Omron CX-Programmer project 新規ﾌﾟﾛｼﾞｪｸﾄ (CX-Programmer 9.20)

# PLC CP_14_0212: CJ2M CPU13
I/O table (CPU CJ2M-CPU13): rack 0 slot 0 CJ1W-ID262; rack 0 slot 1 CJ1W-OD263; rack 0 slot 2 CJ1W-ID262; rack 0 slot 3 CJ1W-OD211; rack 0 slot 4 CJ1W-ID211; rack 0 slot 5 CJ1W-OD211; rack 0 slot 6 CJ1W-CLK23

## Global symbols (name address type ; comment)
0.00 BOOL  ; SE:到着1_確認
0.01 BOOL  ; SE:到着2_確認
0.02 BOOL  ; SE:溜り_確認
0.03 BOOL  ; SE:ﾒｶｴｱｰ圧力
0.04 BOOL  ; SE:切出_引端
0.05 BOOL  ; SE:切出_出端
0.06 BOOL  ; SE:押え_動点
0.07 BOOL  ; SE:供給RBO_過負荷
0.08 BOOL  ; SE:ｽﾄｯﾊﾟｰ3_引端
0.09 BOOL  ; SE:ｽﾄｯﾊﾟｰ3_出端
0.10 BOOL  ; SE:ｽﾄｯﾊﾟｰ2_引端
0.11 BOOL  ; SE:ｽﾄｯﾊﾟｰ2_出端
0.12 BOOL  ; SE:ｽﾄｯﾊﾟｰ1_引端
0.13 BOOL  ; SE:ｽﾄｯﾊﾟｰ1_出端
0.14 BOOL  ; SE:ﾌﾟｯｼｬｰ3_引端
0.15 BOOL  ; SE:ﾌﾟｯｼｬｰ3_出端
1001 CHANNEL  ; 1CH_L_OV_SFT
1001.00 BOOL  ; 1CH_L_OV_SFT
1001.04 BOOL  ; 1CH_L_OV_SFT
1002 CHANNEL  ; 1CH_L_RV_SFT
1002.00 BOOL  ; 1CH_L_RV_SFT
1002.04 BOOL  ; 1CH_L_RV_SFT
1003 CHANNEL  ; 1CH_R_OV_SFT
1003.00 BOOL  ; 1CH_R_OV_SFT
1003.04 BOOL  ; 1CH_R_OV_SFT
1004 CHANNEL  ; 1CH_R_RV_SFT
1004.00 BOOL  ; 1CH_R_RV_SFT
1004.04 BOOL  ; 1CH_R_RV_SFT
1005 CHANNEL  ; 1CH_TSO_SFT
1005.00 BOOL  ; 1CH_TSO_SFT
1005.04 BOOL  ; 1CH_TSO_SFT
1006 CHANNEL  ; 1CH_
1006.00 BOOL  ; 1CH_OV/RV_NG_SFT_(CP1)
1006.04 BOOL  ; R_OV_Hi_(RT1)SFT
1007 CHANNEL  ; 1CH_
1007.00 BOOL  ; 1CH_OV/RV_NG_SFT_(取出)
1007.04 BOOL  ; R_RV_Low_(RT1)SFT
1008 CHANNEL  ; 1CH_
1008.04 BOOL  ; R_RV_Hi_(RT1)SFT
1009 CHANNEL  ; 1CH_
100.00 BOOL  ; PT:SW_全体1ｻｲｸﾙ
100.01 BOOL  ; 未使用
100.02 BOOL  ; 未使用
100.03 BOOL  ; 未使用
100.04 BOOL  ; 主軸_STEP_SW
100.05 BOOL  ; PT:SW_主軸1ｻｲｸﾙ
100.06 BOOL  ; PT:SW_主軸原点復帰
100.07 BOOL  ; PT:SW_全体原点復帰
100.08 BOOL  ; 手動:SW_1-9
100.09 BOOL  ; 手動:SW_1-10
100.10 BOOL  ; 手動:SW_1-11
100.11 BOOL  ; 手動:SW_1-12
100.12 BOOL  ; 手動:SW_1-13
100.13 BOOL  ; 手動:SW_1-14
100.14 BOOL  ; 手動:SW_1-15
100.15 BOOL  ; PT:FUN/RESET_SW
1011 CHANNEL  ; 2CH_L_OV_SFT
1011.01 BOOL  ; 2CH_L_OV_SFT
1011.04 BOOL  ; 2CH_L_OV_SFT
1012 CHANNEL  ; 2CH_L_RV_SFT
1012.01 BOOL  ; 2CH_L_RV_SFT
1012.04 BOOL  ; 2CH_L_RV_SFT
1013 CHANNEL  ; 2CH_R_OV_SFT
1013.01 BOOL  ; 2CH_R_OV_SFT
1013.04 BOOL  ; 2CH_R_OV_SFT
1014 CHANNEL  ; 2CH_R_RV_SFT
1014.01 BOOL  ; 2CH_R_RV_SFT
1014.04 BOOL  ; 2CH_R_RV_SFT
1015 CHANNEL  ; 2CH_TSO_SFT
1015.01 BOOL  ; 2CH_TSO_SFT
1015.04 BOOL  ; 2CH_TSO_SFT
1016 CHANNEL  ; 2CH
1016.00 BOOL  ; 2CH_OV/RV_NG_SFT_(CP2)
1016.04 BOOL  ; R_OV_Hi_(RT2)SFT
1017 CHANNEL  ; 2CH
1017.00 BOOL  ; 2CH_OV/RV_NG_SFT_(取出)
1017.04 BOOL  ; R_RV_Low_(RT2)SFT
1018 CHANNEL  ; 2CH
1018.04 BOOL  ; R_RV_Hi_(RT2)SFT
101.00 BOOL  ; PT:全体1ｻｲｸﾙ
101.01 BOOL  ; 未使用
101.02 BOOL  ; 未使用
101.03 BOOL  ; 未使用
101.04 BOOL  ; 未使用
101.05 BOOL  ; 未使用
101.06 BOOL  ; 主軸原点復帰
101.07 BOOL  ; 全体原点復帰
101.08 BOOL  ; 手動:LP_1-9
101.09 BOOL  ; 手動:LP_1-10
101.10 BOOL  ; 手動:LP_1-11
101.11 BOOL  ; 手動:LP_1-12
101.12 BOOL  ; 手動:LP_1-13
101.13 BOOL  ; 手動:LP_1-14
101.14 BOOL  ; 手動:LP_1-15
101.15 BOOL  ; 手動:LP_1-16
1021 CHANNEL  ; 3CH_L_OV_SFT
1021.03 BOOL  ; 3CH_L_OV_SFT
1021.04 BOOL  ; 3CH_L_OV_SFT
1022 CHANNEL  ; 3CH_L_RV_SFT
1022.03 BOOL  ; 3CH_L_RV_SFT
1022.04 BOOL  ; 3CH_L_RV_SFT
1023 CHANNEL  ; 3CH_R_OV_SFT
1023.03 BOOL  ; 3CH_L_RV_SFT
1023.04 BOOL  ; 3CH_R_OV_SFT
1024 CHANNEL  ; 3CH_R_RV_SFT
1024.03 BOOL  ; 3CH_R_RV_SFT
1024.04 BOOL  ; 3CH_R_RV_SFT
1025 CHANNEL  ; 3CH_TSO_SFT
1025.03 BOOL  ; 3CH_TSO_SFT
1025.04 BOOL  ; 3CH_TSO_SFT
1026 CHANNEL  ; 3CH
1026.00 BOOL  ; 3CH_OV/RN_NG_SFT_(CP3)
1026.04 BOOL  ; R_OV_Hi_(RT3)SFT
1027 CHANNEL  ; 3CH
1027.00 BOOL  ; 3CH_OV/RN_NG_SFT_(取出)
1027.04 BOOL  ; R_RV_Low_(RT3)SFT
1028 CHANNEL  ; 3CH
1028.04 BOOL  ; R_RV_Hi_(RT3)SFT
102.00 BOOL  ; PT:SW_切出1ｻｲｸﾙ
102.01 BOOL  ; PT:SW_供給1ｻｲｸﾙ
102.02 BOOL  ; 未使用
102.04 BOOL  ; PT:SW
102.05 BOOL  ; PT:SW
102.06 BOOL  ; 未使用
102.07 BOOL  ; PT:SW_供給RBO原点復帰
102.08 BOOL  ; 手動:SW_2-9
102.09 BOOL  ; 手動:SW_2-10
102.10 BOOL  ; 手動:SW_2-11
102.11 BOOL  ; 手動:SW_2-12
102.12 BOOL  ; 手動:SW_2-13
102.13 BOOL  ; 手動:SW_2-14
102.14 BOOL  ; 手動:SW_2-15
102.15 BOOL  ; 手動:SW_2-16
1031 CHANNEL  ; L_NO_(CP1)
1031.03 BOOL  ; L_acp_(CP1)
1032 CHANNEL  ; R_NO_(CP1)
1032.03 BOOL  ; R_acp_(CP1)
1033 CHANNEL  ; L_NC_(CP1)
1033.03 BOOL  ; L_bcp_(CP1)
1034 CHANNEL  ; R_NC_(CP1)
1034.03 BOOL  ; R_bcp_(CP1)
1035 CHANNEL  ; L_CG_(CP1)
1035.03 BOOL  ; L_Cg_(CP1)
1036 CHANNEL  ; R_CG_(CP1)
1036.02 BOOL  ; R_Cg_(CP2)
1036.03 BOOL  ; R_Cg_(CP1)
1037 CHANNEL  ; L_未測定_(CP1)
1037.03 BOOL  ; L_未測定_(CP1)
1038 CHANNEL  ; R_未測定_(CP1)
1038.03 BOOL  ; R_未測定_(CP1)
103.00 BOOL  ; 切出1ｻｲｸﾙ
103.01 BOOL  ; 供給1ｻｲｸﾙ
103.02 BOOL  ; 未使用
103.03 BOOL  ; M_供給ﾘﾆｱ
103.04 BOOL  ; :
103.05 BOOL  ; :
103.06 BOOL  ; 未使用
103.07 BOOL  ; 供給RBO_原点復帰
103.08 BOOL  ; 手動:LP_2-9
103.09 BOOL  ; 手動:LP_2-10
103.10 BOOL  ; 手動:LP_2-11
103.11 BOOL  ; 手動:LP_2-12
103.12 BOOL  ; 手動:LP_2-13
103.13 BOOL  ; 手動:LP_2-14
103.14 BOOL  ; 手動:LP_2-15
103.15 BOOL  ; 手動:LP_2-16
1041 CHANNEL  ; L_NO_(CP2)
1041.02 BOOL  ; L_acp_(CP2)
1042 CHANNEL  ; R_NO_(CP2)
1042.02 BOOL  ; R_acp_(CP2)
1043 CHANNEL  ; L_NC_(CP2)
1043.02 BOOL  ; L_bcp_(CP2)
1044 CHANNEL  ; R_NC_(CP2)
1044.02 BOOL  ; R_bcp_(CP2)
1045 CHANNEL  ; L_CG_(CP2)
1045.02 BOOL  ; L_Cg_(CP2)
1046 CHANNEL  ; R_CG_(CP2)
1047 CHANNEL  ; L_未測定_(CP2)
1047.02 BOOL  ; L_未測定_(CP2)
1048 CHANNEL  ; R_未測定_(CP2)
1048.02 BOOL  ; R_未測定_(CP2)
104.00 BOOL  ; PT:SW_RT1ｻｲｸﾙ
104.01 BOOL  ; :
104.02 BOOL  ; 未使用
104.03 BOOL  ; 未使用
104.04 BOOL  ; 洗浄_STEP_SW
104.05 BOOL  ; 未使用
104.06 BOOL  ; 未使用
104.07 BOOL  ; 未使用
104.08 BOOL  ; 手動:SW_3-9
104.09 BOOL  ; 手動:SW_3-10
104.10 BOOL  ; 手動:SW_3-11
104.11 BOOL  ; 手動:SW_3-12
104.12 BOOL  ; 手動:SW_3-13
104.13 BOOL  ; 手動:SW_3-14
104.14 BOOL  ; 手動:SW_3-15
104.15 BOOL  ; 手動:SW_3-16
1051 CHANNEL  ; L_NO_(CP3)
1051.00 BOOL  ; L_acp_(CP3)
1052 CHANNEL  ; R_NO_(CP3)
1052.00 BOOL  ; R_acp_(CP3)
1053 CHANNEL  ; L_NC_(CP3)
1053.00 BOOL  ; L_bcp_(CP3)
1054 CHANNEL  ; R_NC_(CP3)
1054.00 BOOL  ; R_bcp_(CP3)
1055 CHANNEL  ; L_CG_(CP3)
1055.00 BOOL  ; L_Cg_(CP3)
1056 CHANNEL  ; R_CG_(CP3)
1056.00 BOOL  ; R_Cg_(CP3)
1057 CHANNEL  ; L_未測定_(CP3)
1057.00 BOOL  ; L_未測定_(CP3)
1058 CHANNEL  ; R_未測定_(CP3)
1058.00 BOOL  ; R_未測定_(CP3)
105.00 BOOL  ; OV/RV1
105.01 BOOL  ; 未使用
105.02 BOOL  ; 未使用
105.03 BOOL  ; 未使用
105.04 BOOL  ; :
105.05 BOOL  ; 未使用
105.06 BOOL  ; 未使用
105.07 BOOL  ; 未使用
105.08 BOOL  ; 手動:LP_3-9
105.09 BOOL  ; 手動:LP_3-10
105.10 BOOL  ; 手動:LP_3-11
105.11 BOOL  ; 手動:LP_3-12
105.12 BOOL  ; 手動:LP_3-13
105.13 BOOL  ; 手動:LP_3-14
105.14 BOOL  ; 手動:LP_3-15
105.15 BOOL  ; 手動:LP_3-16
106.00 BOOL  ; PT:SW_RT_1ｻｲｸﾙ
106.01 BOOL  ; 未使用
106.02 BOOL  ; 未使用
106.03 BOOL  ; 未使用
106.04 BOOL  ; PT_SW:CP1原点復帰
106.05 BOOL  ; 未使用
106.06 BOOL  ; 未使用
106.07 BOOL  ; 未使用
106.08 BOOL  ; 手動:SW_4-9
106.09 BOOL  ; 手動:SW_4-10
106.10 BOOL  ; 手動:SW_4-11
106.11 BOOL  ; 手動:SW_4-12
106.12 BOOL  ; 手動:SW_4-13
106.13 BOOL  ; 手動:SW_4-14
106.14 BOOL  ; 手動:SW_4-15
106.15 BOOL  ; 手動:SW_4-16
107.00 BOOL  ; CP1_1ｻｲｸﾙ
107.01 BOOL  ; CP2_1ｻｲｸﾙ
107.02 BOOL  ; CP3_1ｻｲｸﾙ
107.03 BOOL  ; 未使用
107.04 BOOL  ; CP1原点復帰
107.05 BOOL  ; CP2原点復帰
107.06 BOOL  ; CP3原点復帰
107.07 BOOL  ; 未使用
107.08 BOOL  ; 手動:LP_4-9
107.09 BOOL  ; 手動:LP_4-10
107.10 BOOL  ; 手動:LP_4-11
107.11 BOOL  ; 手動:LP_4-12
107.12 BOOL  ; 手動:LP_4-13
107.13 BOOL  ; 手動:LP_4-14
107.14 BOOL  ; 手動:LP_4-15
107.15 BOOL  ; 手動:LP_4-16
108.00 BOOL  ; PT:SW_排出1ｻｲｸﾙ
108.01 BOOL  ; 未使用
108.02 BOOL  ; 未使用
108.03 BOOL  ; 未使用
108.04 BOOL  ; 未使用
108.05 BOOL  ; 未使用
108.06 BOOL  ; 未使用
108.07 BOOL  ; PT:SW_排出RBO原点復帰
108.08 BOOL  ; 手動:SW_5-9
108.09 BOOL  ; 手動:SW_5-10
108.10 BOOL  ; PT:SW
108.11 BOOL  ; :
108.12 BOOL  ; 手動:SW_5-13
108.13 BOOL  ; 手動:SW_5-14
108.14 BOOL  ; 手動:SW_5-15
108.15 BOOL  ; 手動:SW_5-16
109.00 BOOL  ; 排出1ｻｲｸﾙ
109.01 BOOL  ; 未使用
109.02 BOOL  ; 未使用
109.03 BOOL  ; CV_HOME
109.04 BOOL  ; CV_1ｻｲｸﾙ
109.05 BOOL  ; 未使用
109.06 BOOL  ; 未使用
109.07 BOOL  ; 排出RBO原点復帰
109.08 BOOL  ; 手動:LP_5-9
109.09 BOOL  ; 手動:LP_5-10
109.10 BOOL  ; :
109.11 BOOL  ; :
109.12 BOOL  ; 手動:LP_5-13
109.13 BOOL  ; 手動:LP_5-14
109.14 BOOL  ; 手動:LP_5-15
109.15 BOOL  ; 手動:LP_5-16
10.00 BOOL  ; CP2:安全位置
10.01 BOOL  ; CP3:ﾚﾃﾞｨｰ
10.02 BOOL  ; CP3:ｴﾗｰ
10.03 BOOL  ; CP3:HOME完了
10.04 BOOL  ; CP3:GO
10.05 BOOL  ; CP3:L_NOCP
10.06 BOOL  ; CP3:R_NOCP
10.07 BOOL  ; CP3:L_NCCP
10.08 BOOL  ; CP3:R_NCCP
10.09 BOOL  ; CP3:L_CG
10.10 BOOL  ; CP3:R_CG
10.11 BOOL  ; CP3:L_未測定
10.12 BOOL  ; CP3:R_未測定
10.13 BOOL  ; CP3:安全位置
10.14 BOOL  ; 次行程IF_下流満杯SE
1100 CHANNEL  ; OK_(RT1)_SFT
1100.00 BOOL  ; RT_OK(1CH)_SFT
1100.04 BOOL  ; OK_(OV/RV1)_SFT
1100.10 BOOL  ; 1CH_OK_OV/RV
1101 CHANNEL  ; OK_(RT2)_SFT
1101.01 BOOL  ; RT_OK(2CH)_SFT
1101.04 BOOL  ; OK_(RT2)_SFT
1101.10 BOOL  ; 2CH_OK_OV/RV
1102 CHANNEL  ; OK_(RT3)_SFT
1102.03 BOOL  ; RT_OK(3CH)_SFT
1102.04 BOOL  ; OK_(RT3)_SFT
1102.10 BOOL  ; 3CH_OK_OV/RV
110.00 BOOL  ; PT:SW_排出1ｻｲｸﾙ
110.01 BOOL  ; 未使用
110.02 BOOL  ; 未使用
110.03 BOOL  ; PT:SW_排出ﾘﾆｱ
110.04 BOOL  ; :
110.05 BOOL  ; 未使用
110.06 BOOL  ; :
110.07 BOOL  ; PT:SW_排出RBO原点復帰
110.08 BOOL  ; 手動:SW_6-9
110.09 BOOL  ; 手動:SW_6-10
110.10 BOOL  ; 手動:SW_6-11
110.11 BOOL  ; 手動:SW_6-12
110.12 BOOL  ; 手動:SW_6-13
110.13 BOOL  ; 手動:SW_6-14
110.14 BOOL  ; 手動:SW_6-15
110.15 BOOL  ; 手動:SW_6-16
1110 CHANNEL  ; OK_(CP1)_SFT
1110.03 BOOL  ; OK_(CP1)_SFT
1111 CHANNEL  ; OK_(CP2)_SFT
1111.02 BOOL  ; OK_(CP2)_SFT
1112 CHANNEL  ; OK_(CP3)_SFT
1112.00 BOOL  ; OK_(CP3)_SFT
111.00 BOOL  ; 排出1ｻｲｸﾙ
111.01 BOOL  ; 未使用
111.02 BOOL  ; 未使用
111.03 BOOL  ; M_排出ﾘﾆｱ
111.04 BOOL  ; :
111.05 BOOL  ; 未使用
111.06 BOOL  ; :
111.07 BOOL  ; 排出RBO原点復帰
111.08 BOOL  ; 手動:LP_6-9
111.09 BOOL  ; 手動:LP_6-10
111.10 BOOL  ; 手動:LP_6-11
111.11 BOOL  ; 手動:LP_6-12
111.12 BOOL  ; 手動:LP_6-13
111.13 BOOL  ; 手動:LP_6-14
111.14 BOOL  ; 手動:LP_6-15
111.15 BOOL  ; 手動:LP_6-16
112.00 BOOL  ; 手動:SW_7-1
112.01 BOOL  ; 手動:SW_7-2
112.02 BOOL  ; 手動:SW_7-3
112.03 BOOL  ; 手動:SW_7-4
112.04 BOOL  ; 手動:SW_7-5
112.05 BOOL  ; 手動:SW_7-6
112.06 BOOL  ; 手動:SW_7-7
112.07 BOOL  ; 手動:SW_7-8
11.00 BOOL  ; RB:HEND_供給
11.01 BOOL  ; RB:PEND_供給
11.02 BOOL  ; RB:ALM_供給
11.03 BOOL  ; RB:SV_供給
11.04 BOOL  ; RB:MOVE_供給
11.05 BOOL  ; SE:前後中間
11.09 BOOL  ; OV/RV:ﾕﾆｯﾄ2_RDY
11.10 BOOL  ; OV/RV:ﾕﾆｯﾄ2_ｴﾗｰ
11.11 BOOL  ; OV/RV_2:GO
11.12 BOOL  ; OV/RV_2:NG1
11.13 BOOL  ; OV/RV_2:NG2
11.14 BOOL  ; OV/RV_2:NG4
11.15 BOOL  ; OV/RV_2:NG8
120.00 BOOL  ; M_1-1SW
120.01 BOOL  ; M_1-2SW
120.02 BOOL  ; M_1-3SW
120.03 BOOL  ; M_1-4SW
120.04 BOOL  ; M_1-5SW
120.05 BOOL  ; M_1-6SW
120.06 BOOL  ; M_1-7SW
120.07 BOOL  ; M_1-8SW
120.08 BOOL  ; M_1-9SW
120.09 BOOL  ; M_1-10SW
120.10 BOOL  ; M_1-11SW
120.11 BOOL  ; M_1-12SW
120.12 BOOL  ; M_1-13SW
120.13 BOOL  ; M_1-14SW
120.14 BOOL  ; M_1-15SW
120.15 BOOL  ; M_1-16SW
121.00 BOOL  ; 単動:LP_搬送後退
121.01 BOOL  ; 単動:LP_搬送前進
121.02 BOOL  ; 単動:LP_搬送搬送
121.03 BOOL  ; 単動:LP_搬送戻り
121.04 BOOL  ; 単動:LP_
121.05 BOOL  ; 単動:LP_
121.06 BOOL  ; 単動:LP_1-7
121.07 BOOL  ; 単動:LP_1-8
121.08 BOOL  ; 単動:LP_押え上昇
121.09 BOOL  ; 単動:LP_押え下降
121.10 BOOL  ; 単動:LP_1-11
121.11 BOOL  ; 単動:LP_1-12
121.12 BOOL  ; 単動:LP_1-13_位置決前後
121.13 BOOL  ; 単動:LP_ﾌﾟﾛｰﾌﾞ昇降
121.14 BOOL  ; 単動:LP_1-15
121.15 BOOL  ; 単動:LP_1-16
122.00 BOOL  ; 単動:SW_2-1
122.01 BOOL  ; 単動:SW_2-2
122.02 BOOL  ; 単動:SW_2-3
122.03 BOOL  ; 単動:SW_2-4
122.04 BOOL  ; 単動:SW_2-5
122.05 BOOL  ; 単動:SW_2-6
122.06 BOOL  ; 単動:SW_2-7
122.07 BOOL  ; 単動:SW_2-8
122.08 BOOL  ; 単動:SW_2-9
122.09 BOOL  ; 単動:SW_2-10
122.10 BOOL  ; 単動:SW_2-11
122.11 BOOL  ; 単動:SW_2-12
122.12 BOOL  ; 単動:SW_2-13
122.13 BOOL  ; 単動:SW_2-14
122.14 BOOL  ; 単動:SW_2-15
122.15 BOOL  ; 単動:SW_2-16
123.00 BOOL  ; 単動:LP_切出
123.01 BOOL  ; 単動:LP_ｽﾄｯﾊﾟｰ
123.02 BOOL  ; 単動:LP_2-3
123.03 BOOL  ; 単動:LP_ﾘﾆｱ
123.04 BOOL  ; 単動:LP_ｽﾄｯﾊﾟｰ1
123.05 BOOL  ; 単動:LP_ｽﾄｯﾊﾟｰ2
123.06 BOOL  ; 単動:LP_ｽﾄｯﾊﾟｰ3
123.07 BOOL  ; 単動:LP_
123.08 BOOL  ; 単動:LP_ﾌﾟｯｼｬｰ1
123.09 BOOL  ; 単動:LP_ﾌﾟｯｼｬｰ2
123.10 BOOL  ; 単動:LP_ﾌﾟｯｼｬｰ3
123.11 BOOL  ; 単動:LP_2-12
123.12 BOOL  ; 単動:LP_
123.13 BOOL  ; 単動:LP_
123.14 BOOL  ; 単動:LP_RBO_移動
123.15 BOOL  ; 単動:LP_2-15
124.00 BOOL  ; 単動:SW_3-1
124.01 BOOL  ; 単動:SW_3-2
124.02 BOOL  ; 単動:SW_3-3
124.03 BOOL  ; 単動:SW_3-4
124.04 BOOL  ; 単動:SW_3-5
124.05 BOOL  ; 単動:SW_3-6
124.06 BOOL  ; 単動:SW_3-7
124.07 BOOL  ; 単動:SW_3-8
124.08 BOOL  ; 単動:SW_3-9
124.09 BOOL  ; 単動:SW_3-10
124.10 BOOL  ; 単動:SW_3-11
124.11 BOOL  ; 単動:SW_3-12
124.12 BOOL  ; 単動:SW_3-13
124.13 BOOL  ; 単動:SW_3-14
124.14 BOOL  ; 単動:SW_3-15
124.15 BOOL  ; 単動:SW_3-16
125.00 BOOL  ; OV/RVﾕﾆｯﾄ1
125.01 BOOL  ; OV/RVﾕﾆｯﾄ2
125.02 BOOL  ; OV/RVﾕﾆｯﾄ3
125.03 BOOL  ; M_切替3
125.04 BOOL  ; M_測定ﾕﾆｯﾄ
125.05 BOOL  ; M_
125.06 BOOL  ; 未使用
125.07 BOOL  ; 未使用
125.08 BOOL  ; M_
125.09 BOOL  ; M_
125.10 BOOL  ; M_
125.11 BOOL  ; M_
125.12 BOOL  ; M_
125.13 BOOL  ; M_
125.14 BOOL  ; M_
125.15 BOOL  ; 未使用
126.00 BOOL  ; 単動:SW_4-1
126.01 BOOL  ; 単動:SW_4-2
126.02 BOOL  ; 単動:SW_4-3
126.03 BOOL  ; 単動:SW_4-4
126.04 BOOL  ; 単動:SW_4-5
126.05 BOOL  ; 単動:SW_4-6
126.06 BOOL  ; 単動:SW_4-7
126.07 BOOL  ; 単動:SW_4-8
126.08 BOOL  ; 単動:SW_4-9
126.09 BOOL  ; 単動:SW_4-10
126.10 BOOL  ; 単動:SW_4-11
126.11 BOOL  ; 単動:SW_4-12
126.12 BOOL  ; 単動:SW_4-13
126.13 BOOL  ; 単動:SW_4-14
126.14 BOOL  ; 単動:SW_4-15
126.15 BOOL  ; 単動:SW_4-16
127.00 BOOL  ; 単動:CP1
127.01 BOOL  ; 単動:LP_
127.02 BOOL  ; 単動:LP_
127.03 BOOL  ; 単動:LP_
127.04 BOOL  ; 単動:LP_
127.05 BOOL  ; 単動:LP_
127.06 BOOL  ; 単動:LP_
127.07 BOOL  ; 単動:LP_
127.08 BOOL  ; 単動:LP_4-9
127.09 BOOL  ; 単動:LP_4-10
127.10 BOOL  ; 単動:LP_4-11
127.11 BOOL  ; 単動:LP_4-12
127.12 BOOL  ; 単動:LP_4-13
127.13 BOOL  ; 単動:LP_4-14
127.14 BOOL  ; 単動:LP_4-15
127.15 BOOL  ; 単動:LP_
128.00 BOOL  ; 単動:SW_5-1
128.01 BOOL  ; 単動:SW_5-2
128.02 BOOL  ; 単動:SW_5-3
128.03 BOOL  ; 単動:SW_5-4
128.04 BOOL  ; 単動:SW_5-5
128.05 BOOL  ; 単動:SW_5-6
128.06 BOOL  ; 単動:SW_5-7
128.07 BOOL  ; 単動:SW_5-8
128.08 BOOL  ; 単動:SW_5-9
128.09 BOOL  ; 単動:SW_5-10
128.10 BOOL  ; 単動:SW_5-11
128.11 BOOL  ; 単動:SW_5-12
128.12 BOOL  ; 単動:SW_5-13
128.13 BOOL  ; 単動:SW_5-14
128.14 BOOL  ; 単動:SW_5-15
128.15 BOOL  ; 単動:SW_5-16
129.00 BOOL  ; 単動:CP2
129.01 BOOL  ; 単動:LP_
129.02 BOOL  ; 単動:LP_5-3
129.03 BOOL  ; 単動:LP_5-4
129.04 BOOL  ; 単動:LP_5-5
129.05 BOOL  ; 単動:LP_5-6
129.06 BOOL  ; 単動:LP_5-7
129.07 BOOL  ; 単動:LP_5-8
129.08 BOOL  ; 単動:LP_5-9
129.09 BOOL  ; 単動:LP_5-10
129.10 BOOL  ; 単動:LP_5-11
129.11 BOOL  ; 単動:LP_5-12
129.12 BOOL  ; 単動:LP_5-13
129.13 BOOL  ; 単動:LP_5-14
129.14 BOOL  ; 単動:LP_5-15
129.15 BOOL  ; 単動:LP_5-16
12.00 BOOL  ; OV/RV1:ｽﾀｰﾄ
12.01 BOOL  ; OV/RV1:ﾘｾｯﾄ
12.02 BOOL  ; OV/RV:CODE1
12.03 BOOL  ; OV/RV:CODE2
12.04 BOOL  ; CP1:ｽﾀｰﾄ
12.05 BOOL  ; CP1:HOME
12.06 BOOL  ; CP2:ｽﾀｰﾄ
12.07 BOOL  ; CP2:HOME
12.08 BOOL  ; CP3:ｽﾀｰﾄ
12.09 BOOL  ; CP3:HOME
12.10 BOOL  ; CP:自動/手動
12.11 BOOL  ; CP:EMG
12.12 BOOL  ; SL:ｱｼｽﾄﾌﾞﾛｰ
130.00 BOOL  ; M_2-1SW
130.01 BOOL  ; M_2-2SW
130.02 BOOL  ; M_2-3SW
130.03 BOOL  ; M_2-4SW
130.04 BOOL  ; M_2-5SW
130.05 BOOL  ; M_2-6SW
130.06 BOOL  ; M_2-7SW
130.07 BOOL  ; M_2-8SW
130.08 BOOL  ; M_2-9SW
130.09 BOOL  ; M_2-10SW
130.10 BOOL  ; M_2-11SW
130.11 BOOL  ; M_2-12SW
130.12 BOOL  ; M_2-13SW
130.13 BOOL  ; M_2-14SW
130.14 BOOL  ; M_2-15SW
130.15 BOOL  ; M_2-16SW
131.00 BOOL  ; 単動:CP3
131.01 BOOL  ; 単動:LP_
131.02 BOOL  ; 単動:LP_
131.03 BOOL  ; 単動:LP_
131.04 BOOL  ; 単動:LP_
131.05 BOOL  ; 単動:LP_
131.06 BOOL  ; 単動:LP_
131.07 BOOL  ; 単動:LP_
131.08 BOOL  ; 単動:LP_
131.09 BOOL  ; 単動:LP_
131.10 BOOL  ; 単動:LP_6-11
131.11 BOOL  ; 単動:LP_6-12
131.12 BOOL  ; 単動:LP_6-13
131.13 BOOL  ; 単動:LP_6-14
131.14 BOOL  ; 単動:LP_6-15
131.15 BOOL  ; 単動:LP_ﾘﾆｱ(ｽﾄｯﾊﾟｰ)
132.00 BOOL  ; 単動:SW_7-1
132.01 BOOL  ; 単動:SW_7-2
132.02 BOOL  ; 単動:SW_7-3
132.03 BOOL  ; 単動:SW_7-4
132.04 BOOL  ; 単動:SW_7-5
132.05 BOOL  ; 単動:SW_7-6
132.06 BOOL  ; 単動:SW_7-7
132.07 BOOL  ; 単動:SW_7-8
132.08 BOOL  ; 単動:SW_7-9
132.09 BOOL  ; 単動:SW_7-10
132.10 BOOL  ; 単動:SW_7-11
132.11 BOOL  ; 単動:SW_7-12
132.12 BOOL  ; 単動:SW_7-13
132.13 BOOL  ; 単動:SW_7-14
132.14 BOOL  ; 単動:SW_7-15
132.15 BOOL  ; 単動:SW_7-16
133.00 BOOL  ; 単動:LP_上昇
133.01 BOOL  ; 単動:LP_下降
133.02 BOOL  ; 単動:LP_7-3
133.03 BOOL  ; 単動:LP_NGﾌﾟｯｼｬｰ
133.04 BOOL  ; 単動:排出C/V_START
133.05 BOOL  ; 単動:戻り
133.06 BOOL  ; 単動:排出
133.07 BOOL  ; 単動:払出
133.08 BOOL  ; 単動:LP_ﾁｬｯｸ1
133.09 BOOL  ; 単動:LP_ﾁｬｯｸ2
133.10 BOOL  ; 単動:LP_ﾁｬｯｸ3
133.11 BOOL  ; 単動:LP_7-12
133.12 BOOL  ; 単動:LP_7-13
133.13 BOOL  ; 単動:LP_7-14
133.14 BOOL  ; 単動:LP_RBO移動
133.15 BOOL  ; 単動:LP_7-16
135.00 BOOL  ; 単動動作中
135.01 BOOL  ; 単動1_動作中
135.02 BOOL  ; 単動2_動作中
135.03 BOOL  ; 単動3_動作中
135.04 BOOL  ; 単動4_動作中
135.05 BOOL  ; 単動5_動作中
135.06 BOOL  ; 単動6_動作中
135.07 BOOL  ; 単動7_動作中
135.10 BOOL  ; 単動動作中表示
135.11 BOOL  ; PT:SW_手動
136.00 BOOL  ; PT:No_100
136.01 BOOL  ; PT:No_101
136.02 BOOL  ; PT:No_102
136.03 BOOL  ; PT:No_103
136.04 BOOL  ; PT:No_104
136.05 BOOL  ; PT:No_105
136.06 BOOL  ; PT:No_106
136.10 BOOL  ; ｻｲｸﾙ画面中
137.00 BOOL  ; 動作中表示_1
137.01 BOOL  ; 動作中表示_2
137.02 BOOL  ; 動作中表示_3
137.03 BOOL  ; 動作中表示_4
137.04 BOOL  ; 動作中表示_5
137.05 BOOL  ; 動作中表示_6
137.06 BOOL  ; 動作中表示_7
138.00 BOOL  ; PT_No_110
138.06 BOOL  ; PT_No_116
13.00 BOOL  ; OV/RV:ﾕﾆｯﾄ3_RDY
13.01 BOOL  ; OV/RV:ﾖﾆｯﾄ3_ｴﾗｰ
13.02 BOOL  ; OV/RV3:GO
13.03 BOOL  ; OV/RV3:NG1
13.04 BOOL  ; OV/RV3:NG2
13.05 BOOL  ; OV/RV3:NG4
13.06 BOOL  ; OV/RV3:NG8
13.07 BOOL  ; 排出ﾓｰﾀ:READY/BUSY
13.08 BOOL  ; 排出ﾓｰﾀ:WARNING
13.09 BOOL  ; 排出ﾓｰﾀ:ERROR
13.10 BOOL  ; 排出ﾓｰﾀ原点ｾﾝｻ
13.11 BOOL  ; 排出ﾓｰﾀ動点ｾﾝｻ
13.12 BOOL  ; SE:CP2ﾌﾟﾛｰﾌﾞ下端
13.13 BOOL  ; SE:CP2ﾌﾟﾛｰﾌﾞ上端
13.14 BOOL  ; SE:CP3ﾌﾟﾛｰﾌﾞ下端
13.15 BOOL  ; SE:CP3ﾌﾟﾛｰﾌﾞ上端
140.08 BOOL  ; IL:搬送1ｻｲｸﾙ
14.00 BOOL  ; OV/RV3:ｽﾀｰﾄ
14.01 BOOL  ; OV/RV3:ﾘｾｯﾄ
14.02 BOOL  ; OV/RV3:CODE1
14.03 BOOL  ; OV/RV3:CODE2
14.04 BOOL  ; OV/RV3:CODE4
14.05 BOOL  ; OV/RV3:CODE8
14.06 BOOL  ; 排出ﾓｰﾀ:IN1
14.07 BOOL  ; 排出ﾓｰﾀ:IN2
14.08 BOOL  ; 排出ﾓｰﾀ:IN3
14.09 BOOL  ; 排出ﾓｰﾀ:START/STOP
14.10 BOOL  ; 排出ﾓｰﾀ:HOME
14.11 BOOL  ; 排出ﾓｰﾀ:ENABLE
14.12 BOOL  ; 排出ﾓｰﾀ:SENSOR1
14.13 BOOL  ; 排出ﾓｰﾀ:SENSOR2
14.14 BOOL  ; 排出ﾓｰﾀ:ORG_SENSOR
170.00 BOOL  ; 総合ERR
170.01 BOOL  ; 表示:ERR中
180.00 BOOL  ; ER:ﾒｲﾝ
181.00 BOOL  ; ER:ｴｱｰ圧力
182.00 BOOL  ; ER:PLC
182.01 BOOL  ; ER:電池異常
182.02 BOOL  ; ER:C/T_ｵｰﾊﾞｰ
182.03 BOOL  ; ER:I/O照合異常
182.04 BOOL  ; ER:ﾘﾓｰﾄI/O異常
183.00 BOOL  ; ER:ﾃﾞｰﾀ収集
183.01 BOOL  ; ﾃﾞｰﾀ収集_満杯
190.00 BOOL  ; ﾄｰﾀﾙｴﾗｰ
190.10 BOOL  ; ﾘｾｯﾄ
1.00 BOOL  ; SE:ﾌﾟｯｼｬｰ2_引端
1.01 BOOL  ; SE:ﾌﾟｯｼｬｰ2_出端
1.02 BOOL  ; SE:ﾌﾟｯｼｬｰ1_引端
1.03 BOOL  ; SE:ﾌﾟｯｼｬｰ1_出端
1.04 BOOL  ; SE:搬送後端
1.05 BOOL  ; SE:搬送前端
1.06 BOOL  ; RB:HEND_主軸
1.07 BOOL  ; RB:PEND_主軸
1.08 BOOL  ; RB:ALM_主軸
1.09 BOOL  ; RB:SV_主軸
1.10 BOOL  ; RB:MOVE_主軸
1.11 BOOL  ; SE:押え(OV/RV)_上端
1.12 BOOL  ; SE:押え(OV/RV)_下端
1.13 BOOL  ; SE:押え(CP1)_上端
1.14 BOOL  ; SE:押え(CP1)_下端
1.15 BOOL  ; SE:押え(CP2)_上端
201.00 BOOL  ; 搬送C/S_F(主軸)
201.01 BOOL  ; 前進_ON
201.02 BOOL  ; 位置決_解放
201.03 BOOL  ; 搬送_搬送位置_指示
201.04 BOOL  ; 搬送_搬送位置_GO_ON
201.05 BOOL  ; 搬送_搬送位置_GO_OFF
201.06 BOOL  ; 搬送_搬送位置_END
201.07 BOOL  ; 後退_ON
201.08 BOOL  ; 位置決_固定
201.09 BOOL  ; 固定確認
201.10 BOOL  ; 搬送_戻り位置_指示
201.11 BOOL  ; 搬送_戻り位置_GO_ON
201.12 BOOL  ; 搬送_戻り位置_GO_OFF
201.13 BOOL  ; 搬送_戻り位置_END
201.14 BOOL  ; 搬送C/E_F
202.00 BOOL  ; 搬送戻り_位置
202.01 BOOL  ; 搬送搬送_位置
203.00 BOOL  ; M_Pos2_指示
203.01 BOOL  ; M_Pos2_GO_ON
203.02 BOOL  ; M_Pos2_GO_OFF
203.03 BOOL  ; M_Pos2_END
203.04 BOOL  ; M_Pos2_C/E
204.00 BOOL  ; M_Pos1_指示
204.01 BOOL  ; M_Pos1_GO_ON
204.02 BOOL  ; M_Pos1_GO_OFF
204.03 BOOL  ; M_Pos1_END
204.04 BOOL  ; M_Poa1_C/E
205.00 BOOL  ; ER復帰_搬送後退_(主軸)
205.01 BOOL  ; ER復帰_位置決_(主軸)
205.02 BOOL  ; ER復帰_押え
205.03 BOOL  ; ER復帰終了_押え
206.00 BOOL  ; 復帰_搬送後退_(主軸)
206.01 BOOL  ; 復帰_押え
208.00 BOOL  ; ﾃﾞｰﾀ転送ﾄﾘｶﾞ
208.01 BOOL  ; ﾃﾞｰﾀｼﾌﾄ完了待ち
20.00 BOOL  ; DB
210.00 BOOL  ; 1CH有_保持
210.01 BOOL  ; 2CH有_保持
210.02 BOOL  ; 3CH有り_保持
211 CHANNEL  ; 1CH_供給SFT
211.00 BOOL  ; OV/RV_1CH_有り
211.01 BOOL  ; CP1_有り
211.05 BOOL  ; 排出_1CH_有り
212 CHANNEL  ; 2CH_供給SFT
212.00 BOOL  ; OV/RV_2CH_有り
212.02 BOOL  ; CP2_有り
212.05 BOOL  ; 排出_2CH_有り
213 CHANNEL  ; 3CH_供給SFT
213.00 BOOL  ; OV/RV_3CH_有り
213.04 BOOL  ; CP3_有り
213.05 BOOL  ; 排出_3CH_有り
215.00 BOOL  ; 供給ｼﾌﾄ_有
216 CHANNEL  ; 1CH_PASS_SFT
216.05 BOOL  ; 1CH_PASS_SFT
217 CHANNEL  ; 2CH_PASS_SFT
217.05 BOOL  ; 2CH_PASS_SFT
218 CHANNEL  ; 3CH_PASS_SFT
218.05 BOOL  ; 3CH_PASS_SFT
220.05 BOOL  ; 主軸_ﾓｰﾀ_ERR
250.00 BOOL  ; 主軸_ERR
250.01 BOOL  ; 主軸ER保持
250.05 BOOL  ; 前後ER_ｻｲｸﾙOFF
250.06 BOOL  ; 位置決ER_ｻｲｸﾙOFF
250.07 BOOL  ; 押えER_ｻｲｸﾙOFF
250.10 BOOL  ; 主軸部ER_ｻｲｸﾙOFF
251.00 BOOL  ; ER:搬送
251.01 BOOL  ; ER:搬送前後
251.02 BOOL  ; ER:押え1_(OV/RV)
251.03 BOOL  ; ER:押え2_(CP1)
251.04 BOOL  ; ER:押え3_(CP2)
251.05 BOOL  ; ER:押え4_(CP3)
251.06 BOOL  ; ER:位置決1
251.07 BOOL  ; ER:位置決2
252.00 BOOL  ; ER:主軸RB
252.01 BOOL  ; ER:主軸RBO_ALM
253.00 BOOL  ; ER:搬送過負荷
253.01 BOOL  ; ER:搬送過負荷
253.02 BOOL  ; 搬送過負荷_一時停止
2.00 BOOL  ; SE:押え(CP2)_下端
2.01 BOOL  ; SE:押え(CP3)_上端
2.02 BOOL  ; SE:押え(CP3)_下端
2.03 BOOL  ; SE:位置決1_出端
2.04 BOOL  ; SE:位置決1_引端
2.05 BOOL  ; SE:位置決2_出端
2.06 BOOL  ; SE:位置決2_引端
2.07 BOOL  ; SE:OV/RVﾌﾟﾛｰﾌﾞ1_下端
2.08 BOOL  ; SE:OV/RVﾌﾟﾛｰﾌﾞ1_上端
2.09 BOOL  ; SE:CP1ﾌﾟﾛｰﾌﾞ下端
2.10 BOOL  ; SE:CP1ﾌﾟﾛｰﾌﾞ上端
2.11 BOOL  ; RB:HEND_排出
2.12 BOOL  ; RB:PEND_排出
2.13 BOOL  ; RB:ALM_排出
2.14 BOOL  ; RB:SV_排出
2.15 BOOL  ; RB:MOVE_排出
300.00 BOOL  ; 上流不足_確認
300.01 BOOL  ; 溜り有_確認
300.05 BOOL  ; 下流満杯
300.06 BOOL  ; 下流満杯_警報
301.00 BOOL  ; 切出_C/S_F
301.01 BOOL  ; ｽﾄｯﾊﾟｰ_ON
301.02 BOOL  ; 切出_ON
301.03 BOOL  ; ｽﾄｯﾊﾟｰ_OFF
301.04 BOOL  ; 供給行き_指示
301.05 BOOL  ; GO_ON
301.06 BOOL  ; GO_OFF
301.07 BOOL  ; GO_END
301.08 BOOL  ; 押え_確認
301.09 BOOL  ; 供給戻り_指示
301.10 BOOL  ; GO_ON
301.11 BOOL  ; GO_OFF
301.12 BOOL  ; GO_END
301.13 BOOL  ; 供給戻り_確認
301.14 BOOL  ; 切出_OFF
301.15 BOOL  ; 切出_C/E
302.00 BOOL  ; 切出終了保持
302.05 BOOL  ; 供給行き_指示保持
303.03 BOOL  ; 切出し戻りC/E_F
304.00 BOOL  ; 切出戻りC/S_F
304.02 BOOL  ; ｽﾄｯﾊﾟｰOFF
305.00 BOOL  ; 供給(No_PASS)_C/S_F
305.01 BOOL  ; Pos2_指示
305.02 BOOL  ; Pos3_指示
305.03 BOOL  ; Pos4_指示
305.04 BOOL  ; :
305.05 BOOL  ; GO_END(3)
305.06 BOOL  ; 押え3_ON
305.07 BOOL  ; ｽﾄｯﾊﾟｰ2_ON
305.08 BOOL  ; 1_GO_ON(2)
305.09 BOOL  ; 1_GO_OFF(2)
305.10 BOOL  ; GO_END(2)
305.11 BOOL  ; 押え2_ON
305.12 BOOL  ; ｽﾄｯﾊﾟｰ1_ON
305.13 BOOL  ; 1_GO_ON(1)
305.14 BOOL  ; 1_GO_OFF(1)
305.15 BOOL  ; GO_END(1)
306.00 BOOL  ; 3_C/S_F
306.01 BOOL  ; ｽﾄｯﾊﾟｰ_ON
306.02 BOOL  ; 押え_ON
306.03 BOOL  ; 3_C/E
306.10 BOOL  ; PASS1_C/E
306.11 BOOL  ; PASS_1/3_C/E
307.00 BOOL  ; 2_C/S_F
307.01 BOOL  ; ｽﾄｯﾊﾟｰ_ON
307.02 BOOL  ; 押え_ON
307.03 BOOL  ; 2_C/E
308.00 BOOL  ; 1_C/S_F
308.01 BOOL  ; ｽﾄｯﾊﾟｰ_ON
308.02 BOOL  ; 押え_ON
308.03 BOOL  ; 1_C/E
308.04 BOOL  ; 2_GO_OFF(2)
308.05 BOOL  ; GO_END(2)
308.06 BOOL  ; 押え2_ON
308.07 BOOL  ; ｽﾄｯﾊﾟｰ1_ON
308.08 BOOL  ; 2_GO_ON(1)
308.09 BOOL  ; 2_GO_OFF(1)
308.10 BOOL  ; GO_END(1)
308.11 BOOL  ; 押え1_ON
308.12 BOOL  ; PASS3_C/E
308.15 BOOL  ; PASS1/3_C/E
309.00 BOOL  ; PASS3_供給終了保持
309.01 BOOL  ; PASS1/3_供給終了保持
310.00 BOOL  ; PASS_有
310.01 BOOL  ; PASS_指示
310.02 BOOL  ; 切出準備OK_3
310.03 BOOL  ; 3_GO_ON(1)
310.04 BOOL  ; 3_GO_OFF(1)
310.05 BOOL  ; GO_END(1)
310.06 BOOL  ; 押え1_ON
310.07 BOOL  ; PASS2/3_C/E
311.00 BOOL  ; PASS2/3_供給終了保持
315.00 BOOL  ; 供給RBO_戻り
316.00 BOOL  ; 供給戻り_C/S_F
316.01 BOOL  ; 戻り_Pos_指示
316.02 BOOL  ; 戻りGO_ON
316.03 BOOL  ; 戻りGO_OFF
316.04 BOOL  ; 戻りGO_END
316.05 BOOL  ; 供給戻り_C/E
317.00 BOOL  ; 供給戻り終了保持
320.00 BOOL  ; No_PASS_切出終了保持
320.01 BOOL  ; PASS1_切出終了保持
320.02 BOOL  ; PASS2_切出終了保持
320.03 BOOL  ; PASS1/2_切出終了保持
320.04 BOOL  ; PASS3_切出終了保持
320.05 BOOL  ; PASS1/3_切出終了保持
320.06 BOOL  ; PASS2/3_切出終了保持
323.00 BOOL  ; 切出終了保持
324.00 BOOL  ; 切出戻り_C/S_F
324.01 BOOL  ; 搬送前進端_確認
324.02 BOOL  ; ﾌﾟｯｼｬｰ/ｽﾄｯﾊﾟｰ_OFF
324.03 BOOL  ; 切出戻り_C/E
324.10 BOOL  ; 前進端保持
324.11 BOOL  ; 供給位置決_解放_保持
325.00 BOOL  ; Pos1_指示
325.01 BOOL  ; Pos2_指示
325.02 BOOL  ; Pos3_指示
325.03 BOOL  ; Pos4_指示
325.05 BOOL  ; 供給RBO_GO
350.00 BOOL  ; ER:供給部
350.01 BOOL  ; 供給ER保持
350.05 BOOL  ; 切出ER_ｻｲｸﾙOFF
350.10 BOOL  ; 供給ERｻｲｸﾙOFF
351.00 BOOL  ; ER:切出
351.01 BOOL  ; ER:切出
351.02 BOOL  ; ER:ｽﾄｯﾊﾟｰ
352.00 BOOL  ; ER:先頭未確認
352.01 BOOL  ; ER:先頭ﾜｰｸ未確認
352.02 BOOL  ; ER:二個目未確認
353.00 BOOL  ; ER:供給RBO
353.01 BOOL  ; ER:供給RBO_ALM
354.00 BOOL  ; ER:供給RBO_過負荷
354.01 BOOL  ; ER:供給RBO_過負荷
354.02 BOOL  ; 供給RBO_一時停止
355.00 BOOL  ; ER:ｽﾄｯﾊﾟｰ1
355.01 BOOL  ; ER:ｽﾄｯﾊﾟｰ1
355.02 BOOL  ; ER:ﾌﾟｯｼｬｰ1
356.00 BOOL  ; ER:ｽﾄｯﾊﾟｰ2
356.01 BOOL  ; ER:ｽﾄｯﾊﾟｰ2
356.02 BOOL  ; ER:ﾌﾟｯｼｬｰ2
357.00 BOOL  ; ER:ｽﾄｯﾊﾟｰ3
357.01 BOOL  ; ER:ｽﾄｯﾊﾟｰ3
357.02 BOOL  ; ER:ﾌﾟｯｼｬｰ3
3.00 BOOL  ; SE:ﾁｬｯｸ_上端
3.01 BOOL  ; SE:ﾁｬｯｸ_下端
3.02 BOOL  ; SE:ﾁｬｯｸ1_開
3.03 BOOL  ; SE:ﾁｬｯｸ1_閉
3.04 BOOL  ; SE:ﾁｬｯｸ2_開
3.05 BOOL  ; SE:ﾁｬｯｸ2_閉
3.06 BOOL  ; SE:ﾁｬｯｸ3_開
3.07 BOOL  ; SE:ﾁｬｯｸ3_閉
3.08 BOOL  ; NGﾌﾟｯｼｬｰ_出端
3.09 BOOL  ; NGﾌﾟｯｼｬｰ_引端
3.10 BOOL  ; SE:NG満杯
3.11 BOOL  ; SE:下流満杯
3.12 BOOL  ; SE:主軸搬送過負荷
400.00 BOOL  ; 測定動作必要
401.00 BOOL  ; 主軸_位置決終了
402.00 BOOL  ; 測定動作_C/S_F
402.01 BOOL  ; ﾌﾟﾛｰﾌﾞ上昇
402.02 BOOL  ; 測定終了
402.03 BOOL  ; ﾌﾟﾛｰﾌﾟ下降
402.04 BOOL  ; 測定動作_C/E
403.00 BOOL  ; 測定終了保持
405.00 BOOL  ; 治具洗浄動作指示
406.00 BOOL  ; 治具洗浄_C/S_F
410.00 BOOL  ; 洗浄部_ERR
4147.09 BOOL  ; CH1_PASS_ｼﾌﾄ_取出
4148.09 BOOL  ; CH2_PASS_ｼﾌﾄ_取出
4149.09 BOOL  ; CH3_PASS_ｼﾌﾄ_取出
4413.00 BOOL  ; ﾁｬｯｸ1_(閉)
4413.01 BOOL  ; ﾁｬｯｸ2_(閉)
4413.02 BOOL  ; ﾁｬｯｸ3_(閉)
450.00 BOOL  ; ER:測定部
451.00 BOOL  ; ER:ﾌﾟﾛｰﾌﾞ昇降
451.01 BOOL  ; ER:ﾌﾟﾛｰﾌﾞ昇降1
451.02 BOOL  ; ER:ﾌﾟﾛｰﾌﾞ昇降2
451.03 BOOL  ; ER:ﾌﾟﾛｰﾌﾞ昇降3
451.04 BOOL  ; ER:ﾌﾟﾛｰﾌﾞ昇降4
4.00 BOOL  ; ST:G
4.01 BOOL  ; ST:Y
4.02 BOOL  ; ST:R
4.03 BOOL  ; ST:BZ
4.04 BOOL  ; LF:供給
4.05 BOOL  ; SL:切出
4.06 BOOL  ; SL:ｽﾄｯﾊﾟｰ
4.07 BOOL  ; SL:ﾌﾟｯｼｬｰ3
4.08 BOOL  ; SL:ﾌﾟｯｼｬｰ2
4.09 BOOL  ; SL:ﾌﾟｯｼｬｰ1
4.10 BOOL  ; SL:ｽﾄｯﾊﾟｰ3
4.11 BOOL  ; SL:ｽﾄｯﾊﾟｰ2
4.12 BOOL  ; SL:ｽﾄｯﾊﾟｰ1
4.13 BOOL  ; SL:押え上昇
4.14 BOOL  ; SL:押え下降
4.15 BOOL  ; SL:搬送後退
500.00 BOOL  ; OV/RV_測定必要
501.00 BOOL  ; OV/RV_測定指示
502.00 BOOL  ; OV/RV1_C/S_F
502.01 BOOL  ; OV/RV1_ｽﾀｰﾄ
502.02 BOOL  ; OV/RV1_ｽﾄｯﾌﾟ
502.03 BOOL  ; OV/RV1_終了
502.04 BOOL  ; OV/RV1_C/E
502.05 BOOL  ; 2CH_ｽﾀｰﾄ_ON
502.06 BOOL  ; 2CH_ｽﾀｰﾄ_OFF
502.07 BOOL  ; 2CH_終了
502.08 BOOL  ; OV/RV1_C/E
503.00 BOOL  ; OV/RV1_終了保持
503.01 BOOL  ; 2CH_開始
503.02 BOOL  ; 2CH_終了
503.03 BOOL  ; 3CH_開始
503.04 BOOL  ; 3CH_終了
504.00 BOOL  ; OV/RV2_C/S_F
504.01 BOOL  ; OV/RV2_ｽﾀｰﾄ
504.02 BOOL  ; OV/RV2_ｽﾄｯﾌﾟ
504.03 BOOL  ; OV/RV2_終了
504.04 BOOL  ; OV/RV2_C/E
505.00 BOOL  ; OV/RV2_終了保持
505.04 BOOL  ; OV/RV3_C/E
505.05 BOOL  ; 3CH_PASS_C/E
506.00 BOOL  ; OV/RV3_C/S_F
506.01 BOOL  ; OV/RV3_ｽﾀｰﾄ
506.02 BOOL  ; OV/RV3_ｽﾄｯﾌﾟ
506.03 BOOL  ; OV/RV3_終了
506.04 BOOL  ; OV/RV3_C/E
507.00 BOOL  ; OV/RV3_終了保持
507.01 BOOL  ; 2CH_開始
507.02 BOOL  ; 2CH_終了
507.03 BOOL  ; 1/3CH_PASS_C/E
508.00 BOOL  ; 2/3CH_PASS_C/S_F
508.01 BOOL  ; 1CH_開始
508.02 BOOL  ; 1CH_終了
508.03 BOOL  ; 2/3CH_PAA_C/E
50.00 BOOL  ; PT:通常運転SW
50.01 BOOL  ; PT:空運転SW
50.02 BOOL  ; PT:終了運転SW
50.03 BOOL  ; PT:予備運転SW
50.04 BOOL  ; PT:ﾀﾞﾐｰ運転SW
50.10 BOOL  ; PT:RT_SW
50.11 BOOL  ; PT:CP_SW
510.00 BOOL  ; RT_終了保持
510.01 BOOL  ; RT_測定開始
511.00 BOOL  ; 1CH指示
511.01 BOOL  ; 2CH指示
511.02 BOOL  ; 3CH指示
514.00 BOOL  ; 測定開始指示
515.00 BOOL  ; RT測定_C/S_F
515.01 BOOL  ; 測定開始
515.02 BOOL  ; 測定中
515.03 BOOL  ; 測定終了
515.04 BOOL  ; RT測定_C/E
515.05 BOOL  ; 2CH_PASS_C/E
51.00 BOOL  ; PT:CH1_PASS_SW
51.01 BOOL  ; PT:PT:CH2_PASS_SW
51.02 BOOL  ; PT:CH3_PASS_SW
520.01 BOOL  ; ﾕﾆｯﾄ1:L_OV_(1)
520.02 BOOL  ; ﾕﾆｯﾄ1:L_RV_(2)
520.03 BOOL  ; ﾕﾆｯﾄ1:R_OV_(8)
520.04 BOOL  ; ﾕﾆｯﾄ1:R_RV_(9)
520.05 BOOL  ; ﾕﾆｯﾄ1:TSO_(3)
520.06 BOOL  ; R_OV_Hi(6)
520.07 BOOL  ; R_RV_Low(7)
520.08 BOOL  ; R_RV_Hi(8)
520.09 BOOL  ; 測定ER_(1)
521.05 BOOL  ; R_OV_Low
525.01 BOOL  ; ﾕﾆｯﾄ2:L_OV_(1)
525.02 BOOL  ; ﾕﾆｯﾄ2:L_RV_(2)
525.03 BOOL  ; ﾕﾆｯﾄ2:R_OV_(8)
525.04 BOOL  ; ﾕﾆｯﾄ2:R_RV_(9)
525.05 BOOL  ; ﾕﾆｯﾄ2:TSO_(3)
526.01 BOOL  ; L_OV_NG
526.02 BOOL  ; L_RV_NG
526.03 BOOL  ; R_OV_NG
526.04 BOOL  ; R_RV_NG
530.01 BOOL  ; ﾕﾆｯﾄ3:L_OV_(1)
530.02 BOOL  ; ﾕﾆｯﾄ3:L_RV_(2)
530.03 BOOL  ; ﾕﾆｯﾄ3:R_OV_(8)
530.04 BOOL  ; ﾕﾆｯﾄ3:R_RV_(9)
530.05 BOOL  ; ﾕﾆｯﾄ3:TSO_(3)
53.00 BOOL  ; PT:SW_原点ﾓﾆﾀ_1
53.01 BOOL  ; PT:SW_原点ﾓﾆﾀ_2
53.02 BOOL  ; PT:SW_原点ﾓﾆﾀ_3
53.03 BOOL  ; PT:SW_原点ﾓﾆﾀ_4
53.04 BOOL  ; PT:SW_原点ﾓﾆﾀ_5
53.05 BOOL  ; PT:SW_原点ﾓﾆﾀ_6
53.06 BOOL  ; PT:SW_原点ﾓﾆﾀ_7
550.00 BOOL  ; ER:ﾕﾆｯﾄ
551.00 BOOL  ; ER:OV/RV1
551.01 BOOL  ; ER:OV/RV1_ﾕﾆｯﾄ
551.02 BOOL  ; ER:OV/RV1_ｵｰﾊｰﾀｲﾑ
551.05 BOOL  ; OV/RV1_ERR保持
552.00 BOOL  ; ER:OV/RV2
552.01 BOOL  ; ER:OV/RV2_ﾕﾆｯﾄ
552.02 BOOL  ; ER:OV/RV2_ｵｰﾊﾞｰﾀｲﾑ
552.05 BOOL  ; OV/RV2_ERR保持
553.00 BOOL  ; ER:OV/RV3
553.01 BOOL  ; ER:OV/RV3_ﾕﾆｯﾄ
553.02 BOOL  ; ER:OV/RV3_ｵｰﾊﾞｰﾀｲﾑ
553.05 BOOL  ; OV/RV3_ERR保持
55.00 BOOL  ; 払出_開始_F
55.01 BOOL  ; 払出切替_F
55.02 BOOL  ; 通常切替_F
5.00 BOOL  ; SL:搬送前進
5.01 BOOL  ; RB:ｽﾀｰﾄ_主軸
5.02 BOOL  ; RB:一時停止_主軸
5.03 BOOL  ; RB:ﾘｾｯﾄ_主軸
5.04 BOOL  ; RB:ｻｰﾎﾞON_主軸
5.05 BOOL  ; RB:HOME_主軸
5.06 BOOL  ; RB:Pos1_主軸
5.07 BOOL  ; RB:Pos2_主軸
5.08 BOOL  ; SL:位置決
5.09 BOOL  ; SL:ﾌﾟﾛｰﾌﾞ上下
5.11 BOOL  ; RB:ｽﾀｰﾄ_排出
5.12 BOOL  ; RB:一時停止_排出
5.13 BOOL  ; RB:ﾘｾｯﾄ_排出
5.14 BOOL  ; RB:ｻｰﾎﾞON_排出
5.15 BOOL  ; RB:HOME_排出
600.00 BOOL  ; CP1_測定必要
601.00 BOOL  ; CP1_測定指示
602.00 BOOL  ; CP1_測定_C/S_F
602.01 BOOL  ; CP1_測定開始
602.02 BOOL  ; CP1_測定中
602.03 BOOL  ; CP1_測定終了
602.04 BOOL  ; CP1_測定_C/E
604.00 BOOL  ; CP1_測定終了保持
605.00 BOOL  ; CP2_測定必要
606.00 BOOL  ; CP2_測定指示
607.00 BOOL  ; CP2_測定_C/S_F
607.01 BOOL  ; CP2_測定開始
607.02 BOOL  ; CP2_測定中
607.03 BOOL  ; CP2_測定終了
607.04 BOOL  ; CP2_測定_C/E
609.00 BOOL  ; CP2_終了保持
60.00 BOOL  ; 主軸RBO_原点復帰指示
60.01 BOOL  ; 主軸RBO_原点復帰
60.02 BOOL  ; 主軸RB_原点復帰終了
60.03 BOOL  ; 主軸RB_Pos1指示
60.04 BOOL  ; 主軸RB_GO_ON
60.05 BOOL  ; 主軸RB_GO_OFF
60.06 BOOL  ; 主軸RB_Pos1_END
60.10 BOOL  ; 主軸RB_復帰終了保持
610.00 BOOL  ; CP3_測定必要
611.00 BOOL  ; CP3_測定指示
612.00 BOOL  ; CP3_測定_C/S_F
612.01 BOOL  ; CP3_測定開始
612.02 BOOL  ; CP3_測定中
612.03 BOOL  ; CP3_測定終了
612.04 BOOL  ; CP3_測定_C/E
614.00 BOOL  ; CP3_終了保持
61.00 BOOL  ; 排出RBO_原点復帰指示
61.01 BOOL  ; 排出RB_原点復帰
61.02 BOOL  ; 排出RB_原点復帰終了
61.03 BOOL  ; 排出RB_Pos1指示
61.04 BOOL  ; 排出RB_GO_ON
61.05 BOOL  ; 排出RB_GO_OFF
61.06 BOOL  ; 排出RB_Pos1_END
61.10 BOOL  ; 排出RB_復帰終了保持
620.00 BOOL  ; CP1_L_CG
620.01 BOOL  ; CP1_L_NOCP
620.02 BOOL  ; CP1_L_NCCP
620.03 BOOL  ; CP1_L_未測定
620.05 BOOL  ; CP1_R_CG
620.06 BOOL  ; CP1_R_NOCP
620.07 BOOL  ; CP1_R_NCCP
620.08 BOOL  ; CP1_R_未測定
620.10 BOOL  ; CP1_L_NG
620.11 BOOL  ; CP1_R_NG
621.00 BOOL  ; CP2_L_CG
621.01 BOOL  ; CP2_L_NOCP
621.02 BOOL  ; CP2_L_NCCP
621.03 BOOL  ; CP2_L_未測定
621.05 BOOL  ; CP2_R_CG
621.06 BOOL  ; CP2_R_NOCP
621.07 BOOL  ; CP2_R_NCCP
621.08 BOOL  ; CP2_R_未測定
621.10 BOOL  ; CP2_L_NG
621.11 BOOL  ; CP2_R_NG
622.00 BOOL  ; CP3_L_CG
622.01 BOOL  ; CP3_L_NOCP
622.02 BOOL  ; CP3_L_NCCP
622.03 BOOL  ; CP3_L_未測定
622.05 BOOL  ; CP3_R_CG
622.06 BOOL  ; CP3_R_NOCP
622.07 BOOL  ; CP3_R_NCCP
622.08 BOOL  ; CP3_R_未測定
622.10 BOOL  ; CP3_L_NG
622.11 BOOL  ; CP3_R_NG
62.00 BOOL  ; 原点復帰_搬送後退
62.01 BOOL  ; 原点復帰_押え上昇
62.02 BOOL  ; 原点復帰_ﾁｬｯｸ上昇
63.00 BOOL  ; 原点復帰_搬送後退
63.01 BOOL  ; 原点復帰_押え上昇
63.02 BOOL  ; 原点復帰_ﾁｬｯｸ上昇
64.00 BOOL  ; 供給RBO_原点復帰指示
64.01 BOOL  ; 供給RBO_原点復帰
64.02 BOOL  ; 供給RB_原点復帰終了
64.03 BOOL  ; 供給RB_Pos1指示
64.04 BOOL  ; 供給RB_GO_ON
64.05 BOOL  ; 供給RB_GO_OFF
64.06 BOOL  ; 供給RB_GO_END
64.10 BOOL  ; 供給RBO_原点復帰終了保持
650.00 BOOL  ; ER:CP
651.00 BOOL  ; ER:CP1
651.01 BOOL  ; ER:CP1ｵｰﾊﾞｰﾀｲﾑ
651.02 BOOL  ; ER:CP1ﾕﾆｯﾄER
652.00 BOOL  ; ER:CP2
652.01 BOOL  ; ER:CP2ｵｰﾊﾞｰﾀｲﾑ
652.02 BOOL  ; ER:CP2ﾕﾆｯﾄER
653.00 BOOL  ; ER:CP3
653.01 BOOL  ; ER:CP3ｵｰﾊﾞｰﾀｲﾑ
653.02 BOOL  ; ER:CP3ﾕﾆｯﾄER
654.00 BOOL  ; ER:EMG
65.00 BOOL  ; CP1_原点復帰指示
65.01 BOOL  ; CP1_原点復帰
65.02 BOOL  ; CP1_原点復帰終了
65.10 BOOL  ; CP1_原点復帰終了保持
66.00 BOOL  ; CP2_原点復帰指示
66.01 BOOL  ; CP2_原点復帰
66.02 BOOL  ; CP2_原点復帰終了
66.10 BOOL  ; CP2_原点復帰終了保持
67.00 BOOL  ; CP3_原点復帰指示
67.01 BOOL  ; CP3_:原点復帰
67.02 BOOL  ; CP3_原点復帰終了
67.10 BOOL  ; CP3_原点復帰終了保持
68.00 BOOL  ; 排出M_復帰指示
68.01 BOOL  ; 排出ﾓｰﾀ_原点復帰
68.02 BOOL  ; 排出ﾓｰﾀ_復帰終了
68.10 BOOL  ; 排出ﾓｰﾀ_復帰終了保持
6.00 BOOL  ; RB:Pos1_排出
6.01 BOOL  ; RB:Pos2_排出
6.02 BOOL  ; RB:Pos4_排出
6.03 BOOL  ; RB:Pos8_排出
6.04 BOOL  ; SL:取出ﾁｬｯｸ上昇
6.05 BOOL  ; SL:取出ﾁｬｯｸ下降
6.06 BOOL  ; SL:取出ﾁｬｯｸ3
6.07 BOOL  ; SL:取出ﾁｬｯｸ2
6.08 BOOL  ; SL:取出ﾁｬｯｸ1
6.09 BOOL  ; SL:NGﾌﾟｯｼｬｰ
6.11 BOOL  ; LF:排出
6.12 BOOL  ; RY:OV/RV切替1
6.13 BOOL  ; RY:OV/RV切替2
6.14 BOOL  ; RY:OV/RV切替3
700.00 BOOL  ; 1CH_ﾃﾞｰﾀ取込
700.01 BOOL  ; 2CH_ﾃﾞｰﾀ取込
700.02 BOOL  ; 3CH_ﾃﾞｰﾀ取込
700.05 BOOL  ; CP1_ﾃﾞｰﾀ取込
700.06 BOOL  ; CP2_ﾃﾞｰﾀ取込
700.07 BOOL  ; CP3_ﾃﾞｰﾀ取込
701.00 BOOL  ; ﾃﾞｰﾀ_ｼﾌﾄ
701.01 BOOL  ; ﾃﾞｰﾀ_OFF
701.05 BOOL  ; ｼﾌﾄﾃﾞｰﾀ_ｸﾘｱ
70.00 BOOL  ; ORG:TTL
710.01 BOOL  ; 1CH_L_OV_保持
710.02 BOOL  ; 1CH_L_RV_保持
710.03 BOOL  ; 1CH_R_OV_保持
710.04 BOOL  ; 1CH_R_RV_保持
710.05 BOOL  ; 1CH_TSO_保持
710.06 BOOL  ; 1CH_
710.07 BOOL  ; 1CH_
710.08 BOOL  ; 1CH_
710.09 BOOL  ; 1CH_
711.01 BOOL  ; 2CH_L_OV_保持
711.02 BOOL  ; 2CH_L_RV_保持
711.03 BOOL  ; 2CH_R_OV_保持
711.04 BOOL  ; 2CH_R_RV_保持
711.05 BOOL  ; 2CH_TSO_保持
711.06 BOOL  ; 2CH_
711.07 BOOL  ; 2CH_
711.08 BOOL  ; 2CH__
712.01 BOOL  ; 3CH_L_OV_保持
712.02 BOOL  ; 3CH_L_RV_保持
712.03 BOOL  ; 3CH_R_OV_保持
712.04 BOOL  ; 3CH_R_RV_保持
712.05 BOOL  ; 3CH_TSO保持
712.06 BOOL  ; 3CH_
712.07 BOOL  ; 3CH_
712.08 BOOL  ; 3CH_
715.00 BOOL  ; 1CH_OV/RV_OK
716.00 BOOL  ; 2CH_OV/RV_OK
717.00 BOOL  ; 3CH_OV/RV_OK保持
71.00 BOOL  ; ORG:主軸
71.01 BOOL  ; ORG:搬送
71.02 BOOL  ; ORG:位置決
71.03 BOOL  ; ORG:ﾌﾟﾛｰﾌﾞ昇降
71.04 BOOL  ; ORG:押え
71.05 BOOL  ; 押え_動点
71.06 BOOL  ; 押え_動点↓
71.07 BOOL  ; 押え_原点
71.08 BOOL  ; 押え:原点↓
720.01 BOOL  ; 1CH_L_NO_(CP1)
720.02 BOOL  ; 1CH_R_NO_(CP1)
720.03 BOOL  ; 1CH_L_NC_(CP1)
720.04 BOOL  ; 1CH_R_NC_(CP1)
720.05 BOOL  ; 1CH_L_CG_(CP1)
720.06 BOOL  ; 1CH_R_CG_(CP1)
720.07 BOOL  ; 1CH_L_未測定_(CP1)
720.08 BOOL  ; 1CH_R_未測定_(CP1)
721.01 BOOL  ; 2CH_L_NO_(CP2)
721.02 BOOL  ; 2CH_R_NO_(CP2)
721.03 BOOL  ; 2CH_L_NC_(CP2)
721.04 BOOL  ; 2CH_R_NC_(CP2)
721.05 BOOL  ; 2CH_L_CG_(CP2)
721.06 BOOL  ; 2CH_R_CG_(CP2)
721.07 BOOL  ; 2CH_L_未測定_(CP2)
721.08 BOOL  ; 2CH_R_未測定_(CP2)
722.01 BOOL  ; 3CH_L_NO_(CP3)
722.02 BOOL  ; 3CH_R_NO_(CP3)
722.03 BOOL  ; 3CH_L_NC_(CP3)
722.04 BOOL  ; 3CH_R_NC_(CP3)
722.05 BOOL  ; 3CH_L_CG_(CP3)
722.06 BOOL  ; 3CH_R_CG_(CP3)
722.07 BOOL  ; 3CH_L_未測定_(CP3)
722.08 BOOL  ; 3CH_R_未測定_(CP3)
725.00 BOOL  ; 1CH_OK_(CP1)
726.00 BOOL  ; 2CH_OK_(CP2)
727.00 BOOL  ; 3CH_OK_(CP3)
72.00 BOOL  ; ORG:供給
72.01 BOOL  ; ORG:切出
72.02 BOOL  ; 切出中
72.05 BOOL  ; ORG:ｴｽｹｰﾌﾟ
72.06 BOOL  ; ORG:ｽﾄｯﾊﾟｰ
72.08 BOOL  ; ORG:ﾌﾟｯｼｬｰ
730.00 BOOL  ; 1CH_排出ﾃﾞｰﾀ_取込
730.01 BOOL  ; 2CH_ﾃﾞｰﾀ取込
730.02 BOOL  ; 3CH_ﾃﾞｰﾀ取込
730.05 BOOL  ; 1CH_排出ﾃﾞｰﾀ_ｸﾘｱ
730.06 BOOL  ; 2CH_排出ﾃﾞｰﾀ_ｸﾘｱ
730.07 BOOL  ; 3CH_排出ﾃﾞｰﾀ_ｸﾘｱ
731.01 BOOL  ; ER:ｽﾄｯﾊﾟｰ
731.02 BOOL  ; ER:反転
731.03 BOOL  ; ER:ﾌﾟｯｼﾔｰ
735.00 BOOL  ; OK_(1CH)
735.01 BOOL  ; OK_(2CH)
735.02 BOOL  ; OK_(3CH)
736.03 BOOL  ; NGﾚｰﾝ1_(1CH)
736.04 BOOL  ; NGﾚｰﾝ2_(1CH)
736.05 BOOL  ; NGﾚｰﾝ3_(1CH)
736.06 BOOL  ; NGﾚｰﾝ4_(1CH)
736.07 BOOL  ; NGﾚｰﾝ5_(1CH)
736.08 BOOL  ; NGﾚｰﾝ6_(1CH)
736.09 BOOL  ; NGﾚｰﾝ7_(1CH)
736.10 BOOL  ; 1CH_NG排出ﾜｰｸ_有り
737.03 BOOL  ; 未検査1_(2CH)
737.04 BOOL  ; NGﾚｰﾝ2_(2CH)
737.05 BOOL  ; NGﾚｰﾝ3_(2CH)
737.06 BOOL  ; NGﾚｰﾝ4_(2CH)
737.07 BOOL  ; NGﾚｰﾝ5_(2CH)
737.08 BOOL  ; NGﾚｰﾝ6_(2CH)
737.09 BOOL  ; NGﾚｰﾝ7_(2CH)
737.10 BOOL  ; 2CH_NG排出ﾜｰｸ_有り
738.03 BOOL  ; 未検査1_(3CH)
738.04 BOOL  ; NGﾚｰﾝ2_(3CH)
738.05 BOOL  ; NGﾚｰﾝ3_(3CH)
738.06 BOOL  ; NGﾚｰﾝ4_(3CH)
738.07 BOOL  ; NGﾚｰﾝ5_(3CH)
738.08 BOOL  ; NGﾚｰﾝ6_(3CH)
738.09 BOOL  ; NGﾚｰﾝ7_(3CH)
738.10 BOOL  ; 3CH_NG排出ﾜｰｸ_有り
73.00 BOOL  ; ORG:OV/RV
740.01 BOOL  ; 排出先_1ヶ所
740.02 BOOL  ; 排出先_2ヶ所
740.03 BOOL  ; 排出先_3ヶ所
74.00 BOOL  ; ORG:CP測定
74.01 BOOL  ; ORG:CP1
74.02 BOOL  ; ORG:CP2
74.03 BOOL  ; ORG:CP3
750.00 BOOL  ; ﾃﾞｰﾀ_有
751.00 BOOL  ; 1CH_L_OV/RV_OK
751.01 BOOL  ; 1CH_L_OV/RV_NG
751.02 BOOL  ; 1CH_L_OV/RV_未測定
751.03 BOOL  ; 1CH_R_OV/RV_OK
751.04 BOOL  ; 1CH_R_OV/RV_NG
751.05 BOOL  ; 1CH_R_OV/RV_未測定
751.06 BOOL  ; 1CH_L_CP_OK
751.07 BOOL  ; 1CH_L_CP_NO
751.08 BOOL  ; 1CH_L_CP_NC
751.09 BOOL  ; 1CH_L_CP_CG
751.10 BOOL  ; 1CH_L_CP_未測定
751.11 BOOL  ; 1CH_R_CP_OK
751.12 BOOL  ; 1CH_R_CP_NO
751.13 BOOL  ; 1CH_R_CP_NC
751.14 BOOL  ; 1CH_R_CP_CG
751.15 BOOL  ; 1CH_R_CP_未測定
752.00 BOOL  ; 2CH_L_OV_OK
752.01 BOOL  ; 2CH_L_OV_NG
752.02 BOOL  ; 2CH_L_OV_未測定
752.03 BOOL  ; 2CH_R_OV_OK
752.04 BOOL  ; 2CH_R_OV_NG
752.05 BOOL  ; 2CH_R_OV_未測定
752.06 BOOL  ; 2CH_L_CP_OK
752.07 BOOL  ; 2CH_L_CP_NO
752.08 BOOL  ; 2CH_L_CP_NC
752.09 BOOL  ; 2CH_L_CP_CG
752.10 BOOL  ; 2CH_L_CP_未測定
752.11 BOOL  ; 2CH_R_CP_OK
752.12 BOOL  ; 2CH_R_CP_NO
752.13 BOOL  ; 2CH_R_CP_NC
752.14 BOOL  ; 2CH_R_CP_CG
752.15 BOOL  ; 2CH_R_CP_未測定
753.00 BOOL  ; 3CH_L_OV_OK
753.01 BOOL  ; 3CH_L_OV_NG
753.02 BOOL  ; 3CH_L_OV_未測定
753.03 BOOL  ; 3CH_R_OV_OK
753.04 BOOL  ; 3CH_R_OV_NG
753.05 BOOL  ; 3CH_R_OV_未測定
753.06 BOOL  ; 3CH_L_CP_OK
753.07 BOOL  ; 3CH_L_CP_NO
753.08 BOOL  ; 3CH_L_CP_NC
753.09 BOOL  ; 3CH_L_CP_CG
753.10 BOOL  ; 3CH_L_CP_未測定
753.11 BOOL  ; 3CH_R_CP_OK
753.12 BOOL  ; 3CH_R_CP_NO
753.13 BOOL  ; 3CH_R_CP_NC
753.14 BOOL  ; 3CH_R_CP_CG
753.15 BOOL  ; 3CH_R_CP_未測定
75.00 BOOL  ; ORG:排出
75.01 BOOL  ; 排出:ORG
75.05 BOOL  ; ORG:排出ｺﾝﾍﾞｱ
76.00 BOOL  ; ORG:ﾃﾞｰﾀ収集
76.01 BOOL  ; RDY:ﾃﾞｰﾀ収集
7.00 BOOL  ; RB:ｽﾀｰﾄ_供給
7.01 BOOL  ; RB:一時停止_供給
7.02 BOOL  ; RB:ﾘｾｯﾄ_供給
7.03 BOOL  ; RB:ｻｰﾎﾞON_供給
7.04 BOOL  ; RB:HOME_供給
7.05 BOOL  ; RB:Pos1_供給
7.06 BOOL  ; RB:Pos2_供給
7.07 BOOL  ; RB:Pos4_供給
7.10 BOOL  ; OV/RV2:ｽﾀｰﾄ
7.11 BOOL  ; OV/RV2:ﾘｾｯﾄ
7.12 BOOL  ; OV/RV2:CODE1
7.13 BOOL  ; OV/RV2:CODE2
7.14 BOOL  ; OV/RV2:CODE4
7.15 BOOL  ; OV/RV2:CODE8
800.00 BOOL  ; 排出必要
800.02 BOOL  ; 排出必要_予約
801.00 BOOL  ; DB_SW:仮
805.00 BOOL  ; 排出C/S_F
805.01 BOOL  ; 下降_ON
805.02 BOOL  ; ﾁｬｯｸ_閉
805.03 BOOL  ; 上昇_ON
805.04 BOOL  ; 排出1_GO_ON
805.05 BOOL  ; 排出1_GO_OFF
805.06 BOOL  ; 排出1_GO_END
805.07 BOOL  ; 下降_ON
805.08 BOOL  ; ﾁｬｯｸ_開
805.09 BOOL  ; 上昇_ON
805.10 BOOL  ; 排出2_GO_ON
805.11 BOOL  ; 排出2_GO_OFF
805.12 BOOL  ; 排出2_GO_END
805.13 BOOL  ; 下降_ON
805.14 BOOL  ; ﾁｬｯｸ_開
805.15 BOOL  ; 上昇_ON
806.00 BOOL  ; 排出3_GO_ON
806.01 BOOL  ; 排出3_GO_OFF
806.02 BOOL  ; 排出3_GO_END
806.03 BOOL  ; 下降_ON
806.04 BOOL  ; ﾁｬｯｸ_開
806.05 BOOL  ; 上昇_ON
807.00 BOOL  ; 排出戻り_Pos_指示
807.01 BOOL  ; 排出戻り_GO_ON
807.02 BOOL  ; 排出戻り_GO_OFF
807.03 BOOL  ; 排出戻り_GO_END
807.04 BOOL  ; ﾁｬｯｸ開ﾁｪｯｸ
807.05 BOOL  ; 排出C/E_F
808.00 BOOL  ; DB_排出
80.00 BOOL  ; PT:運転SW
80.05 BOOL  ; PT:停止SW
810.00 BOOL  ; 排出済_搬送許可
815.01 BOOL  ; 排出_Pos1
815.02 BOOL  ; 排出_Pos2
815.03 BOOL  ; 排出_Pos3
815.04 BOOL  ; 排出_Pos4
815.05 BOOL  ; 排出_Pos5
815.06 BOOL  ; 排出_Pos6
815.07 BOOL  ; 排出_Pos7
815.08 BOOL  ; 排出_Pos8
815.09 BOOL  ; 排出_Pos9
816.00 BOOL  ; 排出RBO_Pos指示
816.01 BOOL  ; 排出RBO_GO
816.02 BOOL  ; 排出RBO_Pos1
816.03 BOOL  ; 排出RBO_Pos2
816.04 BOOL  ; 排出RBO_Pos4
816.05 BOOL  ; 排出RBO_Pos8
816.10 BOOL  ; ﾁｬｯｸ開_ﾀｲﾐﾝｸﾞ
817.01 BOOL  ; 取出_位置
817.02 BOOL  ; OK_位置
817.03 BOOL  ; NGﾚｰﾝ1
817.04 BOOL  ; NGﾚｰﾝ2
817.05 BOOL  ; NGﾚｰﾝ3
817.06 BOOL  ; NGｹｰﾝ4
817.07 BOOL  ; NGﾚｰﾝ5
817.08 BOOL  ; NGﾚｰﾝ6
817.09 BOOL  ; NGﾚｰﾝ7
817.10 BOOL  ; 移動禁止
818.01 BOOL  ; ﾁｬｯｸ1_閉
818.02 BOOL  ; ﾁｬｯｸ2_閉
818.03 BOOL  ; ﾁｬｯｸ3_閉
819.01 BOOL  ; ﾁｬｯｸ1_開
819.02 BOOL  ; ﾁｬｯｸ2_開
819.03 BOOL  ; ﾁｬｯｸ3_開
819.10 BOOL  ; ﾁｬｯｸ1_開確認
81.00 BOOL  ; 運転_F
81.05 BOOL  ; 運転連絡
820.00 BOOL  ; NG_排出ﾜｰｸ有
821.00 BOOL  ; NG_排出C/S_F
821.01 BOOL  ; ﾌﾟｯｼｬｰ_ON
821.02 BOOL  ; ﾌﾟｯｼｬｰ_OFF
821.03 BOOL  ; NG排出_C/E
822.00 BOOL  ; NGﾌﾟｯｼｬｰ_ON
823.00 BOOL  ; CP_測定中
823.01 BOOL  ; CP_RDY
825.00 BOOL  ; ER復帰_上昇
825.01 BOOL  ; ER復帰_ﾁｬｯｸ
826.00 BOOL  ; 復帰_上昇
826.01 BOOL  ; 復帰_ﾁｬｯｸ
82.00 BOOL  ; 停止_F
82.05 BOOL  ; 停止ﾗﾝﾌﾟ
830.00 BOOL  ; 排出_必要
831.00 BOOL  ; 排出ｺﾝﾍﾞｱ_C/S_F
831.01 BOOL  ; 排出_指示
831.02 BOOL  ; 搬送_ON
831.03 BOOL  ; 搬送_END
831.04 BOOL  ; 戻り_指示
831.05 BOOL  ; 戻り_ON
831.06 BOOL  ; 戻り_END
831.07 BOOL  ; 原点確認
831.08 BOOL  ; 排出ｺﾝﾍﾞｱ_C/E
831.10 BOOL  ; 払出_指示
831.11 BOOL  ; 払出_ON
831.12 BOOL  ; 払出_END
831.13 BOOL  ; 次行程IF_脱磁停止
83.00 BOOL  ; ﾄｰﾀﾙ_C/S_F
84.00 BOOL  ; ﾄｰﾀﾙ_待機ﾌﾗｸﾞ
84.01 BOOL  ; ﾊﾟｰﾂ情報_1
84.02 BOOL  ; ﾊﾟｰﾂ情報_2
84.03 BOOL  ; ﾊﾟｰﾂ情報_3
84.04 BOOL  ; ﾊﾟｰﾂ情報_4
84.05 BOOL  ; ﾊﾟｰﾂ情報_5
84.06 BOOL  ; ﾊﾟｰﾂ情報_6
84.07 BOOL  ; ﾊﾟｰﾂ情報_7
850.00 BOOL  ; 排出部_ER:排出部
850.01 BOOL  ; 排出ER保持
850.05 BOOL  ; 昇降ER_ｻｲｸﾙOFF
850.06 BOOL  ; ﾁｬｯｸ_1ER_ｻｲｸﾙOFF
850.07 BOOL  ; ﾁｬｯｸ_2ER_ｻｲｸﾙOFF
850.08 BOOL  ; ﾁｬｯｸ_3ER_ｻｲｸﾙOFF
850.10 BOOL  ; 排出部ER_ｻｲｸﾙOFF
851.00 BOOL  ; ER:排出RBO
851.01 BOOL  ; ER:排出RBO_ALM
851.02 BOOL  ; ER:排出RBO_ｵｰﾊﾞｰﾀｲﾑ
852.00 BOOL  ; ER:排出
852.01 BOOL  ; ER:排出昇降
852.02 BOOL  ; ER:NGﾌﾟｯｼｬｰ
853.00 BOOL  ; ER:ﾁｬｯｸ1
853.01 BOOL  ; ER:ﾁｬｯｸ1
854.00 BOOL  ; ER:ﾁｬｯｸ2
854.01 BOOL  ; ER:ﾁｬｯｸ2
855.00 BOOL  ; ER:ﾁｬｯｸ3
855.01 BOOL  ; ER:ﾁｬｯｸ3
856.00 BOOL  ; 排出NG満杯
856.01 BOOL  ; 排出NG満杯
857.00 BOOL  ; ER:排出ﾓｰﾀ
857.01 BOOL  ; ER:RDY_OFF
857.02 BOOL  ; ER:WARNING
857.03 BOOL  ; ER:ERROR
857.04 BOOL  ; ER:ｵｰﾊﾞｰﾀｲﾑ
85.00 BOOL  ; ﾄｰﾀﾙ_警報ﾌﾗｸﾞ
85.01 BOOL  ; 警報_1
85.02 BOOL  ; 警報_2
85.03 BOOL  ; 警報_3
85.04 BOOL  ; 警報_4
85.05 BOOL  ; 警報_5
85.06 BOOL  ; 警報_6
86.00 BOOL  ; PT:SW_ﾌﾞｻﾞｰｵﾌ
86.05 BOOL  ; ﾌﾞｻﾞｰｵﾌ
87.00 BOOL  ; 手動
87.01 BOOL  ; MAIN
87.05 BOOL  ; 手動
87.06 BOOL  ; 単動
87.10 BOOL  ; MAIN_指示
87.11 BOOL  ; MAIN_指示保持
88.00 BOOL  ; ﾁｮｺ停CNT_CLR_SW
88.05 BOOL  ; 生産ｶｳﾝﾄ_CLR_SW
88.10 BOOL  ; ｻｲｸﾙﾀｲﾑｵｰﾊﾞｰ
89.00 BOOL  ; ERR_CNT条件
89.05 BOOL  ; PT:SW_ERR_CNT_CLR
89.06 BOOL  ; PT:SW_ERR_ST
89.07 BOOL  ; PT:SW_NGｶｳﾝﾄ
89.09 BOOL  ; DB:SW_ER無効
89.10 BOOL  ; ｴﾗｰ検出条件
8.00 BOOL  ; OV/RV:ﾕﾆｯﾄ1_RDY
8.01 BOOL  ; OV/RV:ﾕﾆｯﾄ1_ｴﾗｰ
8.02 BOOL  ; OV/RV_1:GO
8.03 BOOL  ; OV/RV_1:NG1
8.04 BOOL  ; OV/RV_1:NG2
8.05 BOOL  ; OV/RV_1:NG4
8.06 BOOL  ; OV/RV_1:NG8
8.07 BOOL  ; CP1:ﾚﾃﾞｨｰ
8.08 BOOL  ; CP1:ｴﾗｰ
8.09 BOOL  ; CP1:HOME完了
8.10 BOOL  ; CP1:GO
8.11 BOOL  ; CP1:L_NOCP
8.12 BOOL  ; CP1:R_NOCP
8.13 BOOL  ; CP1:L_NCCP
8.14 BOOL  ; CP1:R_NCCP
8.15 BOOL  ; CP1:L_CG
90.00 BOOL  ; IL:全体1ｻｲｸﾙ
90.01 BOOL  ; IL:
90.02 BOOL  ; IL:
90.03 BOOL  ; IL:
90.04 BOOL  ; IL:
90.05 BOOL  ; IL:
90.06 BOOL  ; IL:主軸RBO原点復帰
90.07 BOOL  ; IL:全体原点復帰
90.08 BOOL  ; IL:切出1ｻｲｸﾙ
90.09 BOOL  ; IL:供給1ｻｲｸﾙ
90.10 BOOL  ; IL:
90.11 BOOL  ; IL:ﾘﾆｱ_ｵﾌ
90.12 BOOL  ; IL:
90.13 BOOL  ; IL:
90.14 BOOL  ; IL:
90.15 BOOL  ; IL:供給RBO_HOME
91.00 BOOL  ; IL:OV/RV_1ｻｲｸﾙ
91.01 BOOL  ; IL:
91.02 BOOL  ; IL:
91.03 BOOL  ; IL:
91.04 BOOL  ; IL:
91.05 BOOL  ; IL:
91.06 BOOL  ; IL:
91.07 BOOL  ; IL:
91.08 BOOL  ; IL:CP1_1ｻｲｸﾙ
91.09 BOOL  ; IL:CP2_1ｻｲｸﾙ
91.10 BOOL  ; IL:CP3_1ｻｲｸﾙ
91.11 BOOL  ; IL:
91.12 BOOL  ; IL:CP1原点復帰
91.13 BOOL  ; IL:CP2原点復帰
91.14 BOOL  ; IL:CP3原点復帰
91.15 BOOL  ; IL:
92.00 BOOL  ; IL:排出1ｻｲｸﾙ
92.01 BOOL  ; IL:
92.02 BOOL  ; IL:
92.03 BOOL  ; IL:C/V_HOME
92.04 BOOL  ; IL:
92.05 BOOL  ; IL:
92.06 BOOL  ; IL:
92.07 BOOL  ; IL:排出ROB原点復帰
93.00 BOOL  ; IL:搬送後退
93.01 BOOL  ; IL:搬送前進
93.02 BOOL  ; IL:搬送搬送
93.03 BOOL  ; IL:搬送戻り
93.04 BOOL  ; IL:
93.05 BOOL  ; IL:
93.06 BOOL  ; IL:
93.07 BOOL  ; IL:
93.08 BOOL  ; IL:押え上昇
93.09 BOOL  ; IL:押え下降
93.12 BOOL  ; IL:位置決前後
93.13 BOOL  ; IL:ﾌﾟﾛｰﾌﾞ上下
93.14 BOOL  ; IL:
93.15 BOOL  ; IL:
94.00 BOOL  ; IL:切出
94.01 BOOL  ; IL:ｽﾄｯﾊﾟｰ
94.02 BOOL  ; IL:ｽﾄｯﾊﾟｰ1
94.03 BOOL  ; IL:
94.04 BOOL  ; IL:ｽﾄｯﾊﾟｰ1
94.05 BOOL  ; IL:ｽﾄｯﾊﾟｰ2
94.06 BOOL  ; IL:ｽﾄｯﾊﾟｰ6
94.07 BOOL  ; IL:
94.08 BOOL  ; IL:ﾌﾟｯｼｬｰ1
94.09 BOOL  ; IL:ﾌﾟｯｼｬｰ2
94.10 BOOL  ; IL:ﾌﾟｯｼｬｰ3
94.11 BOOL  ; IL:
94.12 BOOL  ; IL:
94.13 BOOL  ; IL:
94.14 BOOL  ; IL:供給RBO
94.15 BOOL  ; IL:
95.00 BOOL  ; IL:ﾕﾆｯﾄ1_(OV/RV)
95.01 BOOL  ; IL:ﾕﾆｯﾄ2_(OV/RV)
95.02 BOOL  ; IL:ﾕﾆｯﾄ3_(OV/RV)
95.03 BOOL  ; IL:
95.04 BOOL  ; IL:
96.00 BOOL  ; IL:CP1
97.00 BOOL  ; IL:CP2
98.00 BOOL  ; IL:CP3
99.00 BOOL  ; IL:上昇
99.01 BOOL  ; IL:下降
99.02 BOOL  ; IL:
99.03 BOOL  ; IL:NGﾌﾟｯｼｬｰ
99.04 BOOL  ; IL:排出CV_START
99.05 BOOL  ; IL:戻り
99.06 BOOL  ; IL:排出
99.07 BOOL  ; IL:払出
99.08 BOOL  ; IL:ﾁｬｯｸ1
99.09 BOOL  ; IL:ﾁｬｯｸ2
99.10 BOOL  ; IL:ﾁｬｯｸ3
99.11 BOOL  ; IL:
99.12 BOOL  ; IL:
99.13 BOOL  ; IL:
99.14 BOOL  ; IL:排出RBO移動
99.15 BOOL  ; IL:
9.00 BOOL  ; CP1:R_CG
9.01 BOOL  ; CP1:L_未測定
9.02 BOOL  ; CP1:R_未測定
9.03 BOOL  ; CP1:安全位置
9.04 BOOL  ; CP2:ﾚﾃﾞｨｰ
9.05 BOOL  ; CP2:ｴﾗｰ
9.06 BOOL  ; CP2:HOME完了
9.07 BOOL  ; CP2:GO
9.08 BOOL  ; CP2:L_NOCP
9.09 BOOL  ; CP2:R_NOCP
9.10 BOOL  ; CP2:L_NCCP
9.11 BOOL  ; CP2:R_NCCP
9.12 BOOL  ; CP2:L_CG
9.13 BOOL  ; CP2:R_CG
9.14 BOOL  ; CP2:L_未測定
9.15 BOOL  ; CP2:R_未測定
A402.05 BOOL  ; ﾘﾓｰﾄI/O異常
C0010 BOOL  ; 6sec
D10 CHANNEL  ; PT:画面切替
D1000 CHANNEL  ; 長押し_時間
D10000.00 BOOL  ; 収集PLCﾄﾘｶﾞ
D10000.03 BOOL  ; 払出運転
D10001.00 BOOL  ; 収集RT1検査ﾌﾗｸﾞ
D10001.01 BOOL  ; 収集RT2検査ﾌﾗｸﾞ
D10001.02 BOOL  ; 収集RT3検査ﾌﾗｸﾞ
D10001.03 BOOL  ; 収集CP1検査ﾌﾗｸﾞ
D10001.04 BOOL  ; 収集CP2検査ﾌﾗｸﾞ
D10001.05 BOOL  ; 収集CP3検査ﾌﾗｸﾞ
D10002.00 BOOL  ; 収集検査開始ﾄﾘｶﾞ
D10007 CHANNEL  ; 1st：ﾜｰｸ有り
D10008 CHANNEL  ; 2st：ﾜｰｸ有り
D10009 CHANNEL  ; 3st：ﾜｰｸ有り
D10010 CHANNEL  ; 1CH_OV_L
D10011 CHANNEL  ; 1CH_OV_R
D10012 CHANNEL  ; 1CH_RV_L
D10013 CHANNEL  ; 1CH_RV_R
D10014 CHANNEL  ; 1CH_TS_L
D10015 CHANNEL  ; 1CH_TS_R
D10016 CHANNEL  ; 2CH_OV_L
D10017 CHANNEL  ; 2CH_OV_R
D10018 CHANNEL  ; 2CH_RV_L
D10019 CHANNEL  ; 2CH_RV_R
D10020 CHANNEL  ; 2CH_TS_L
D10021 CHANNEL  ; 2CH_TS_R
D10022 CHANNEL  ; 3CH_OV_L
D10023 CHANNEL  ; 3CH_OV_R
D10024 CHANNEL  ; 3CH_RV_L
D10025 CHANNEL  ; 3CH_RV_R
D10026 CHANNEL  ; 3CH_TS_L
D10027 CHANNEL  ; 3CH_TS_R
D10028 CHANNEL  ; 1CH_NO_L
D10029 CHANNEL  ; 1CH_NO_R
D10030 CHANNEL  ; 1CH_NC_L
D10031 CHANNEL  ; 1CH_NC_R
D10032 CHANNEL  ; 1CH_CG_L
D10033 CHANNEL  ; 1CH_CG_R
D10034 CHANNEL  ; 2CH_NO_L
D10035 CHANNEL  ; 2CH_NO_R
D10036 CHANNEL  ; 2CH_NC_L
D10037 CHANNEL  ; 2CH_NC_R
D10038 CHANNEL  ; 2CH_CG_L
D10039 CHANNEL  ; 2CH_CG_R
D10040 CHANNEL  ; 3CH_NO_L
D10041 CHANNEL  ; 3CH_NO_R
D10042 CHANNEL  ; 3CH_NC_L
D10043 CHANNEL  ; 3CH_NC_R
D10044 CHANNEL  ; 3CH_CG_L
D10045 CHANNEL  ; 3CH_CG_R
D10050 CHANNEL  ; 3CH_L_OV_Low
D10051 CHANNEL  ; 3CH_L_OV_Hi
D10052 CHANNEL  ; 3CH_R_OV_Low
D10053 CHANNEL  ; 3CH_R_OV_Hi
D10054 CHANNEL  ; 3CH_L_RV_Low
D10055 CHANNEL  ; 3CH_L_RV_Hi
D10056 CHANNEL  ; 3CH_R_RV_Low
D10057 CHANNEL  ; 3CH_R_RV_Hi
D10058 CHANNEL  ; 3CH_L_acp
D10059 CHANNEL  ; 3CH_R_acp
D10060 CHANNEL  ; 3CH_L_bcp
D10061 CHANNEL  ; 3CH_R_bcp
D10062 CHANNEL  ; 3CH_L_cg
D10063 CHANNEL  ; 3CH_R_cg
D1010 CHANNEL  ; PT:画面No.
D10990 CHANNEL  ; NGｺｰﾄﾞ
D10991 CHANNEL  ; OKｺｰﾄﾞ
D10992 CHANNEL  ; 未側ｺｰﾄﾞ
D11994.00 BOOL  ; ﾃﾞｰﾀ収集Busy
D11997 CHANNEL  ; RDY:ﾃﾞｰﾀ収集
D11997.00 BOOL  ; RDY:ﾃﾞｰﾀ収集
D1600 CHANNEL  ; 1CH_排出先ﾃﾞｰﾀ
D1610 CHANNEL  ; 2CH_排出先ﾃﾞｰﾀ
D1620 CHANNEL  ; 3CH_排出先ﾃﾞｰﾀ
D1650 CHANNEL  ; 排出RBO_現在位置
D202 CHANNEL  ; 投入数
D204 CHANNEL  ; 生産数
D206 CHANNEL  ; 不良数
D208 CHANNEL  ; 歩留り
D210 CHANNEL  ; 稼働率
D220 CHANNEL  ; 全体_C/T
D221 CHANNEL  ; 主軸_C/T
D222 CHANNEL  ; 切出_C/T
D223 CHANNEL  ; 測定_C/T
D224 CHANNEL  ; RT_C/T
D225 CHANNEL  ; CP1_C/T
D226 CHANNEL  ; CP2_C/T
D227 CHANNEL  ; CP3_C/T
D228 CHANNEL  ; 排出_C/T
D240 CHANNEL  ; ERR:MAIN
D241 CHANNEL  ; ERR:主軸部
D242 CHANNEL  ; ERR:ﾍﾞｰｽ供給部
D243 CHANNEL  ; ERR:測定部
D244 CHANNEL  ; ERR:RT
D245 CHANNEL  ; ERR:CP1
D246 CHANNEL  ; ERR:CP2
D247 CHANNEL  ; ERR:CP3
D248 CHANNEL  ; ERR:排出部
D250 CHANNEL  ; 生産数×1000
D260 CHANNEL  ; 生産数×1000
D3000 CHANNEL  ; 指示Pos_CNT
D400 CHANNEL  ; 1CH_L_OV
D401 CHANNEL  ; 1CH_L_RV
D402 CHANNEL  ; 1CH_TSO
D403 CHANNEL  ; 1CH_L_RV_Hi
D404 CHANNEL  ; 1CH_R_OV
D405 CHANNEL  ; 1CH_R_RV
D406 CHANNEL  ; 1CH_R_TSO
D407 CHANNEL  ; 1CH_R_RV_Hi
D408 CHANNEL  ; 1CH_L_NO
D409 CHANNEL  ; 1CH_L_NC
D410 CHANNEL  ; 1CH_L_CG
D411 CHANNEL  ; 1CH_L_未測定
D412 CHANNEL  ; 1CH_R_NO
D413 CHANNEL  ; 1CH_R_NC
D414 CHANNEL  ; 1CH_R_CG
D415 CHANNEL  ; 1CH_R_未測定
D420 CHANNEL  ; 2CH_L_OV
D421 CHANNEL  ; 2CH_L_RV
D422 CHANNEL  ; 2CH_TSO
D423 CHANNEL  ; 2CH_L_RV_Hi
D424 CHANNEL  ; 2CH_R_OV
D425 CHANNEL  ; 2CH_R_RV
D426 CHANNEL  ; 2CH_R_RV_Low
D427 CHANNEL  ; 2CH_R_RV_Hi
D428 CHANNEL  ; 2CH_L_NO
D429 CHANNEL  ; 2CH_L_NC
D430 CHANNEL  ; 2CH_L_CG
D431 CHANNEL  ; 2CH_L_未測定
D432 CHANNEL  ; 2CH_R_NO
D433 CHANNEL  ; 2CH_R_NC
D434 CHANNEL  ; 2CH_R_CG
D435 CHANNEL  ; 2CH_R_未測定
D440 CHANNEL  ; 3CH_L_OV
D441 CHANNEL  ; 3CH_L_RV
D442 CHANNEL  ; 3CH_TSO
D443 CHANNEL  ; 3CH_L_RV_Hi
D444 CHANNEL  ; 3CH_R_OV
D445 CHANNEL  ; 3CH_R_RV
D446 CHANNEL  ; 3CH_R_RV_Low
D447 CHANNEL  ; 3CH_R_RV_Hi
D448 CHANNEL  ; 3CH_L_NO
D449 CHANNEL  ; 3CH_L_NC
D450 CHANNEL  ; 3CH_L_CG
D451 CHANNEL  ; 3CH_L_未測定
D452 CHANNEL  ; 3CH_R_NO
D453 CHANNEL  ; 3CH_R_NC
D454 CHANNEL  ; 3CH_R_CG
D455 CHANNEL  ; 3CH_R_未測定
D601 CHANNEL  ; C/T_比較値
D92 CHANNEL  ; MODE
H10.00 BOOL  ; 通常運転
H10.01 BOOL  ; 終了運転
H10.02 BOOL  ; 払出運転
H10.03 BOOL  ; 予備運転
H10.04 BOOL  ; ﾀﾞﾐｰ運転
H10.05 BOOL  ; 指定無し
H10.10 BOOL  ; RT_選択
H10.11 BOOL  ; CP_選択
H11.00 BOOL  ; CH1_PASS
H11.01 BOOL  ; CH2_PASS
H11.02 BOOL  ; CH3_PASS
H11.05 BOOL  ; CH1_PASSﾌﾞﾛｯｸ
H11.06 BOOL  ; CH2_PASS_ﾌﾞﾛｯｸ
H11.07 BOOL  ; CH3_PASS_ﾌﾞﾛｯｸ
H12.00 BOOL  ; 1_PASS
H12.01 BOOL  ; 2_PASS
H12.02 BOOL  ; 3_PASS
H12.03 BOOL  ; 1/2_PASS
H12.04 BOOL  ; 1/3_PASS
H12.05 BOOL  ; 2/3_PASS
H12.15 BOOL  ; NO_PASS
H90.04 BOOL  ; DB:TTL_OK
H90.08 BOOL  ; DB:ﾃﾞｰﾀ収集無効
T0000 BOOL  ; 電源ON DRY
T0001 BOOL  ; 主軸RB_ｻｰﾎﾞON
T0002 BOOL  ; 主軸RB_HOME
T0003 BOOL  ; 排出RB_ｻｰﾎﾞON
T0004 BOOL  ; 排出RB_HOME
T0005 BOOL  ; 供給RB_ｻｰﾎﾞON
T0006 BOOL  ; 供給RB_HOME
T0042 BOOL  ; 供給RBO_復帰確認
T0060 BOOL  ; SW:ｽﾀｰﾄUP↑
T0081 BOOL  ; ERR_CNT_CLR
T0175 BOOL  ; 総合ERR_遅延
T0180 BOOL  ; :
T0201 BOOL  ; 位置決解放_確認
T0202 BOOL  ; 搬送前端_確認
T0203 BOOL  ; 搬送_Pos2指示
T0206 BOOL  ; 位置決固定確認
T0300 BOOL  ; 先頭_有確認
T0302 BOOL  ; 二個目_有確認
T0304 BOOL  ; 上流有り_確認
T0306 BOOL  ; 上流無し_確認
T0314 BOOL  ; GO_END_確認
T0316 BOOL  ; :
T0317 BOOL  ; :
T0319 BOOL  ; :
T0320 BOOL  ; :
T0323 BOOL  ; :
T0330 BOOL  ; 供給ﾘﾆｱ
T0340 BOOL  ; 供給ﾜｰｸ無確認
T0345 BOOL  ; 先頭未確認
T0346 BOOL  ; 二個目未確認
T0400 BOOL  ; :
T0401 BOOL  ; :
T0402 BOOL  ; :
T0500 BOOL  ; :
T0501 BOOL  ; :
T0502 BOOL  ; :
T0505 BOOL  ; :
T0816 BOOL  ; 排出1_上端確認
T0820 BOOL  ; 排出2_上端確認
T0825 BOOL  ; 排出3_上端確認
T0845 BOOL  ; 排出ﾘﾆｱ
T0861 BOOL  ; :
T1000 BOOL  ; 遅延_1-1
T1001 BOOL  ; 遅延_1-2
T1002 BOOL  ; 遅延_1-3
T1003 BOOL  ; 遅延_1-4
T1004 BOOL  ; 遅延_1-5
T1005 BOOL  ; 遅延_1-6
T1006 BOOL  ; 遅延_1-7
T1007 BOOL  ; 遅延_1-8
T1010 BOOL  ; 遅延_2-1
T1011 BOOL  ; 遅延_2-2
T1012 BOOL  ; 遅延_2-3
T1013 BOOL  ; 遅延_2-4
T1014 BOOL  ; 遅延_2-5
T1015 BOOL  ; 遅延_2-6
T1016 BOOL  ; 遅延_2-7
T1017 BOOL  ; 遅延_2-8
T1020 BOOL  ; 遅延_3-1
T1021 BOOL  ; 遅延_3-2
T1022 BOOL  ; 遅延_3-3
T1023 BOOL  ; 遅延_3-4
T1024 BOOL  ; 遅延_3-5
T1025 BOOL  ; 遅延_3-6
T1026 BOOL  ; 遅延_3-7
T1027 BOOL  ; 遅延_3-8
T1030 BOOL  ; 遅延_4-1
T1031 BOOL  ; 遅延_4-2
T1032 BOOL  ; 遅延_4-3
T1033 BOOL  ; 遅延_4-4
T1034 BOOL  ; 遅延_4-5
T1035 BOOL  ; 遅延_4-6
T1036 BOOL  ; 遅延_4-7
T1037 BOOL  ; 遅延_4-8
T1040 BOOL  ; 遅延_5-1
T1041 BOOL  ; 遅延_5-2
T1042 BOOL  ; 遅延_5-3
T1043 BOOL  ; 遅延_5-4
T1044 BOOL  ; 遅延_5-5
T1045 BOOL  ; 遅延_5-6
T1046 BOOL  ; 遅延_5-7
T1047 BOOL  ; 遅延_5-8
T1050 BOOL  ; 遅延_6-1
T1051 BOOL  ; 遅延_6-2
T1052 BOOL  ; 遅延_6-3
T1053 BOOL  ; 遅延_6-4
T1054 BOOL  ; 遅延_6-5
T1055 BOOL  ; 遅延_6-6
T1056 BOOL  ; 遅延_6-7
T1057 BOOL  ; 遅延_6-8
T1060 BOOL  ; 遅延_7-1
T1061 BOOL  ; 遅延_7-2
T1062 BOOL  ; 遅延_7-3
T1063 BOOL  ; 遅延_7-4
T1064 BOOL  ; 遅延_7-5
T1065 BOOL  ; 遅延_7-6
T1066 BOOL  ; 遅延_7-7
T1067 BOOL  ; 遅延_7-8
T1309 BOOL  ; 1CH_未検査排出判定
T2000 BOOL  ; 収集PLCﾄﾘｶﾞON時間
T2001 BOOL  ; ﾃﾞｰﾀｼﾌﾄ待ち時間
T72 CHANNEL  ; :
W147 CHANNEL  ; 1st：ﾜｰｸ有り
W148 CHANNEL  ; 2st：ﾜｰｸ有り
W149 CHANNEL  ; 3st：ﾜｰｸ有り
W50.00 BOOL  ; PT:SW_#80
W50.01 BOOL  ; PT:SW_#81
W50.02 BOOL  ; PT:SW_#82
W50.03 BOOL  ; PT:SW_#83
W50.04 BOOL  ; PT:SW_#84
W50.05 BOOL  ; PT:SW_#90
W50.06 BOOL  ; PT:SW_#85
W50.07 BOOL  ; PT:SW_#86
W511.09 BOOL  ; DEBUG_EM1_2nd_ﾁｬｯｸ開確認
W511.10 BOOL  ; DEBUG
W511.11 BOOL  ; DEBUG_EM1_2nd_次行程満杯
W511.12 BOOL  ; DEBUG_EM1_2nd_未検査判定ﾀｲﾐﾝｸﾞ変更
W511.13 BOOL  ; DEBUG_EM1_2nd_先頭ﾜｰｸ未確認ER変更
W511.14 BOOL  ; DEBUG_EM1_2nd_排出CV
W511.15 BOOL  ; DEBUG_EM1_2nd_排出順番変更

## Program MAIN (cyclic task 0)

### Section MAIN

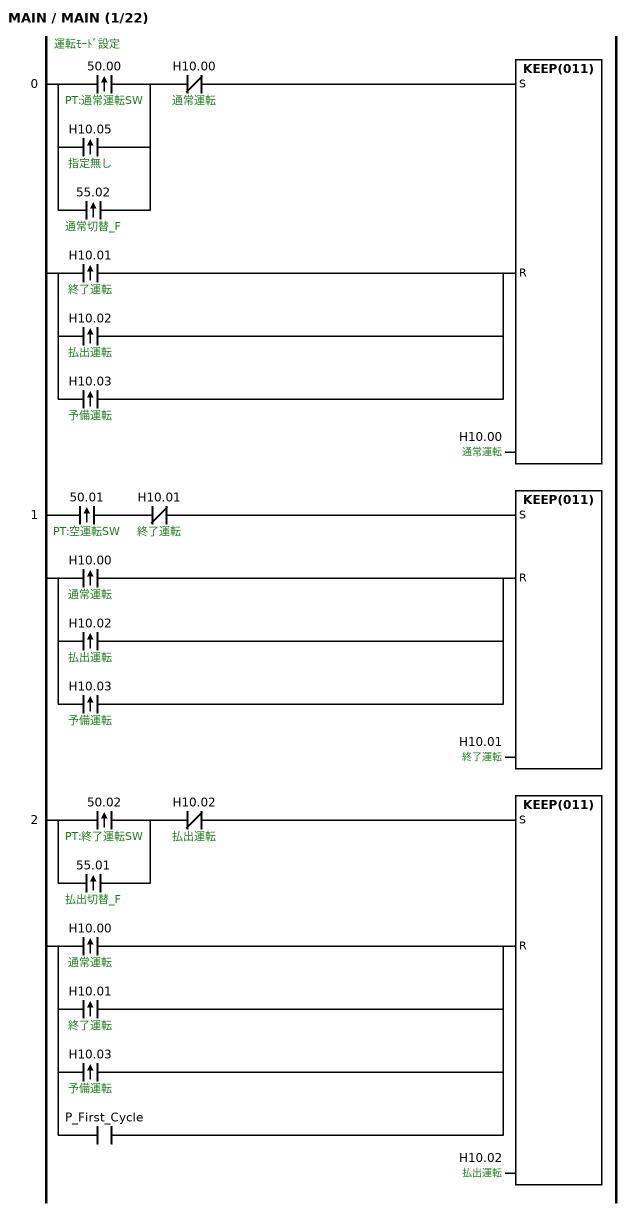
; rung 0: 運転ﾓｰﾄﾞ設定
@LD 50.00  ; PT:通常運転SW
@OR H10.05  ; 指定無し
@OR 55.02  ; 通常切替_F
ANDNOT H10.00  ; 通常運転
@LD H10.01  ; 終了運転
@OR H10.02  ; 払出運転
@OR H10.03  ; 予備運転
KEEP(011) H10.00  ; 通常運転
; rung 1
@LD 50.01  ; PT:空運転SW
ANDNOT H10.01  ; 終了運転
@LD H10.00  ; 通常運転
@OR H10.02  ; 払出運転
@OR H10.03  ; 予備運転
KEEP(011) H10.01  ; 終了運転
; rung 2
@LD 50.02  ; PT:終了運転SW
@OR 55.01  ; 払出切替_F
ANDNOT H10.02  ; 払出運転
@LD H10.00  ; 通常運転
@OR H10.01  ; 終了運転
@OR H10.03  ; 予備運転
OR P_First_Cycle
KEEP(011) H10.02  ; 払出運転

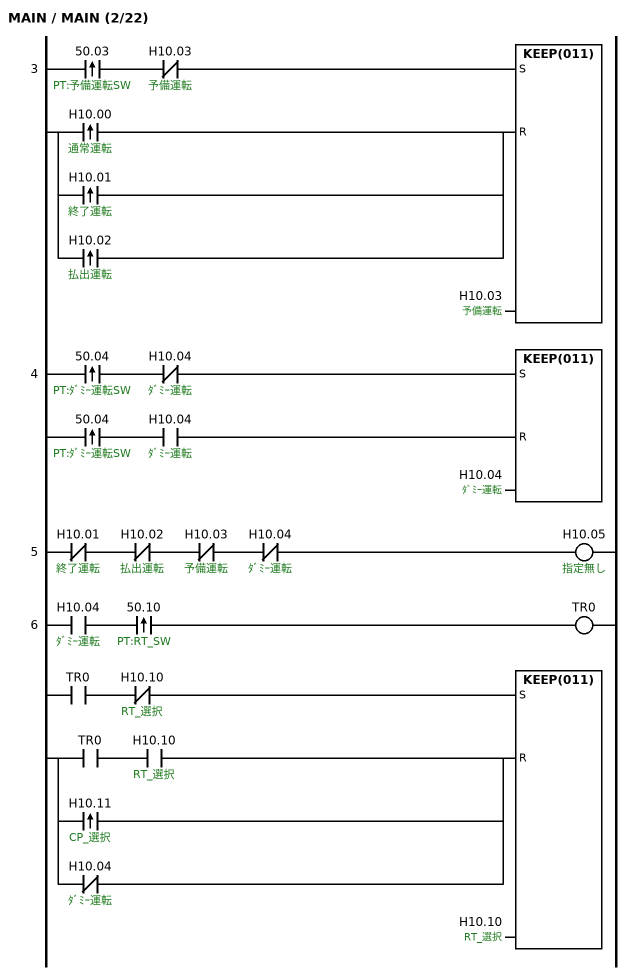
; rung 3
@LD 50.03  ; PT:予備運転SW
ANDNOT H10.03  ; 予備運転
@LD H10.00  ; 通常運転
@OR H10.01  ; 終了運転
@OR H10.02  ; 払出運転
KEEP(011) H10.03  ; 予備運転
; rung 4
@LD 50.04  ; PT:ﾀﾞﾐｰ運転SW
ANDNOT H10.04  ; ﾀﾞﾐｰ運転
@LD 50.04  ; PT:ﾀﾞﾐｰ運転SW
AND H10.04  ; ﾀﾞﾐｰ運転
KEEP(011) H10.04  ; ﾀﾞﾐｰ運転
; rung 5
LDNOT H10.01  ; 終了運転
ANDNOT H10.02  ; 払出運転
ANDNOT H10.03  ; 予備運転
ANDNOT H10.04  ; ﾀﾞﾐｰ運転
OUT H10.05  ; 指定無し
; rung 6
LD H10.04  ; ﾀﾞﾐｰ運転
@AND 50.10  ; PT:RT_SW
OUT TR0
ANDNOT H10.10  ; RT_選択
LD TR0
AND H10.10  ; RT_選択
@LD H10.11  ; CP_選択
ORNOT H10.04  ; ﾀﾞﾐｰ運転
ORLD
KEEP(011) H10.10  ; RT_選択

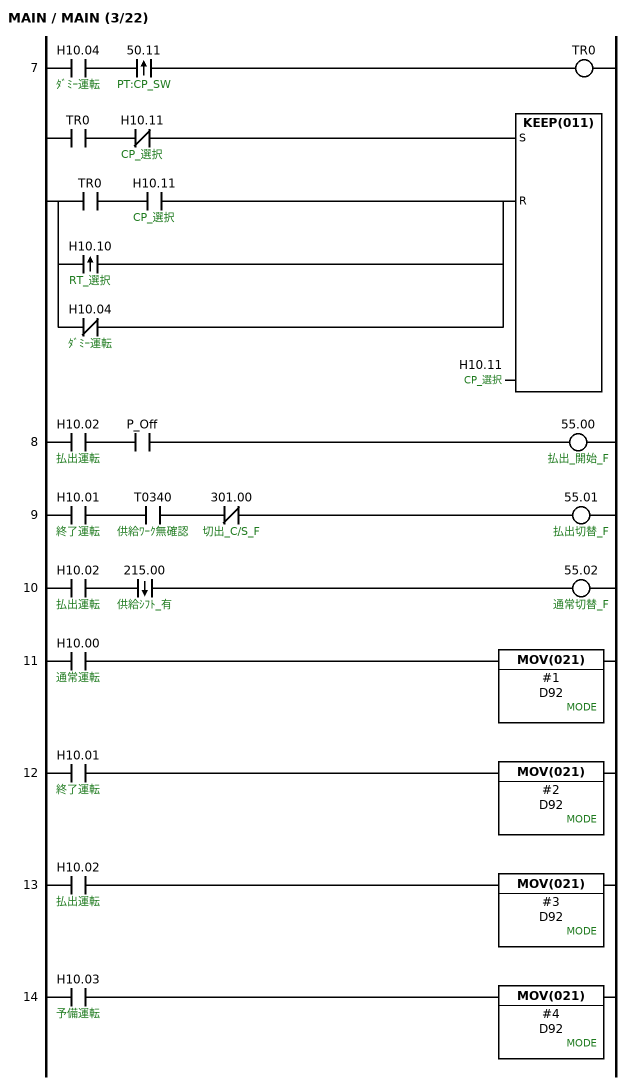
; rung 7
LD H10.04  ; ﾀﾞﾐｰ運転
@AND 50.11  ; PT:CP_SW
OUT TR0
ANDNOT H10.11  ; CP_選択
LD TR0
AND H10.11  ; CP_選択
@LD H10.10  ; RT_選択
ORNOT H10.04  ; ﾀﾞﾐｰ運転
ORLD
KEEP(011) H10.11  ; CP_選択
; rung 8
LD H10.02  ; 払出運転
AND P_Off
OUT 55.00  ; 払出_開始_F
; rung 9
LD H10.01  ; 終了運転
AND T0340  ; 供給ﾜｰｸ無確認
ANDNOT 301.00  ; 切出_C/S_F
OUT 55.01  ; 払出切替_F
; rung 10
LD H10.02  ; 払出運転
%AND 215.00  ; 供給ｼﾌﾄ_有
OUT 55.02  ; 通常切替_F
; rung 11
LD H10.00  ; 通常運転
MOV(021) #1 D92  ; MODE
; rung 12
LD H10.01  ; 終了運転
MOV(021) #2 D92  ; MODE
; rung 13
LD H10.02  ; 払出運転
MOV(021) #3 D92  ; MODE
; rung 14
LD H10.03  ; 予備運転
MOV(021) #4 D92  ; MODE

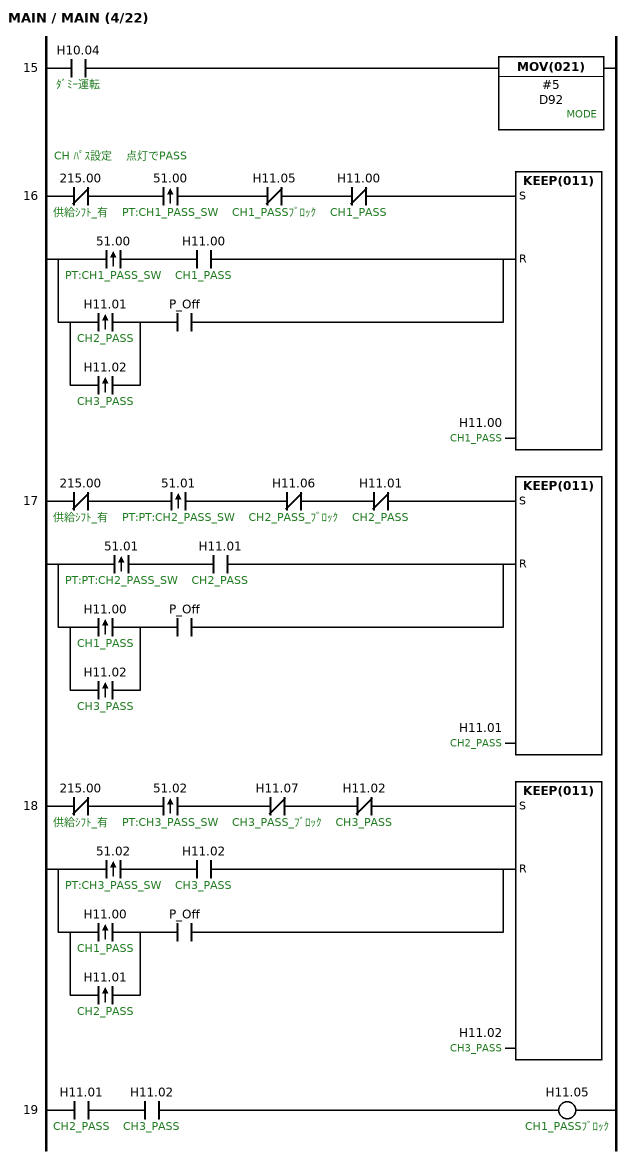
; rung 15
LD H10.04  ; ﾀﾞﾐｰ運転
MOV(021) #5 D92  ; MODE
; rung 16: CH ﾊﾟｽ設定    点灯でPASS
LDNOT 215.00  ; 供給ｼﾌﾄ_有
@AND 51.00  ; PT:CH1_PASS_SW
ANDNOT H11.05  ; CH1_PASSﾌﾞﾛｯｸ
ANDNOT H11.00  ; CH1_PASS
@LD 51.00  ; PT:CH1_PASS_SW
AND H11.00  ; CH1_PASS
@LD H11.01  ; CH2_PASS
@OR H11.02  ; CH3_PASS
AND P_Off
ORLD
KEEP(011) H11.00  ; CH1_PASS
; rung 17
LDNOT 215.00  ; 供給ｼﾌﾄ_有
@AND 51.01  ; PT:PT:CH2_PASS_SW
ANDNOT H11.06  ; CH2_PASS_ﾌﾞﾛｯｸ
ANDNOT H11.01  ; CH2_PASS
@LD 51.01  ; PT:PT:CH2_PASS_SW
AND H11.01  ; CH2_PASS
@LD H11.00  ; CH1_PASS
@OR H11.02  ; CH3_PASS
AND P_Off
ORLD
KEEP(011) H11.01  ; CH2_PASS
; rung 18
LDNOT 215.00  ; 供給ｼﾌﾄ_有
@AND 51.02  ; PT:CH3_PASS_SW
ANDNOT H11.07  ; CH3_PASS_ﾌﾞﾛｯｸ
ANDNOT H11.02  ; CH3_PASS
@LD 51.02  ; PT:CH3_PASS_SW
AND H11.02  ; CH3_PASS
@LD H11.00  ; CH1_PASS
@OR H11.01  ; CH2_PASS
AND P_Off
ORLD
KEEP(011) H11.02  ; CH3_PASS
; rung 19
LD H11.01  ; CH2_PASS
AND H11.02  ; CH3_PASS
OUT H11.05  ; CH1_PASSﾌﾞﾛｯｸ

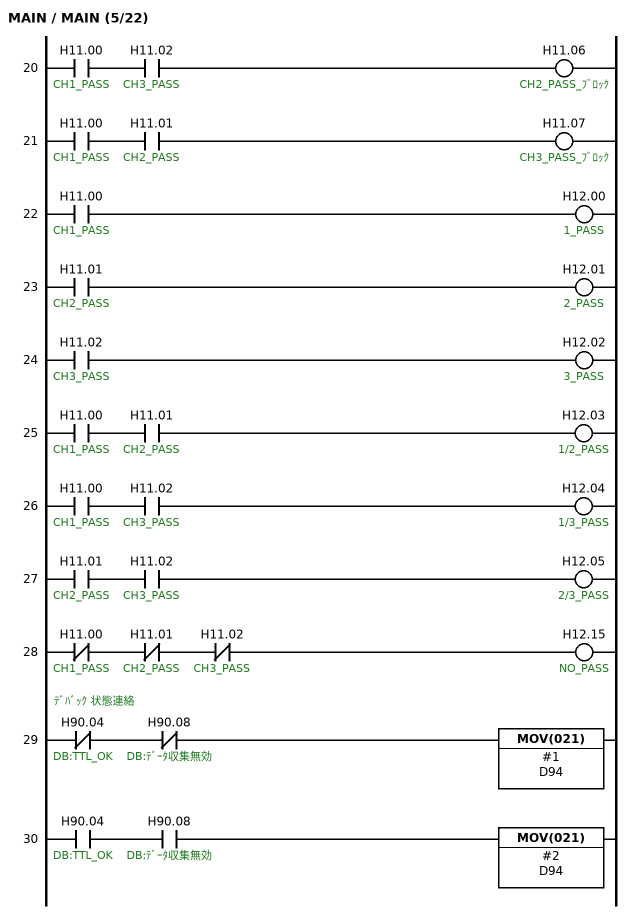
; rung 20
LD H11.00  ; CH1_PASS
AND H11.02  ; CH3_PASS
OUT H11.06  ; CH2_PASS_ﾌﾞﾛｯｸ
; rung 21
LD H11.00  ; CH1_PASS
AND H11.01  ; CH2_PASS
OUT H11.07  ; CH3_PASS_ﾌﾞﾛｯｸ
; rung 22
LD H11.00  ; CH1_PASS
OUT H12.00  ; 1_PASS
; rung 23
LD H11.01  ; CH2_PASS
OUT H12.01  ; 2_PASS
; rung 24
LD H11.02  ; CH3_PASS
OUT H12.02  ; 3_PASS
; rung 25
LD H11.00  ; CH1_PASS
AND H11.01  ; CH2_PASS
OUT H12.03  ; 1/2_PASS
; rung 26
LD H11.00  ; CH1_PASS
AND H11.02  ; CH3_PASS
OUT H12.04  ; 1/3_PASS
; rung 27
LD H11.01  ; CH2_PASS
AND H11.02  ; CH3_PASS
OUT H12.05  ; 2/3_PASS
; rung 28
LDNOT H11.00  ; CH1_PASS
ANDNOT H11.01  ; CH2_PASS
ANDNOT H11.02  ; CH3_PASS
OUT H12.15  ; NO_PASS
; rung 29: ﾃﾞﾊﾞｯｸ 状態連絡
LDNOT H90.04  ; DB:TTL_OK
ANDNOT H90.08  ; DB:ﾃﾞｰﾀ収集無効
MOV(021) #1 D94
; rung 30
LD H90.04  ; DB:TTL_OK
AND H90.08  ; DB:ﾃﾞｰﾀ収集無効
MOV(021) #2 D94

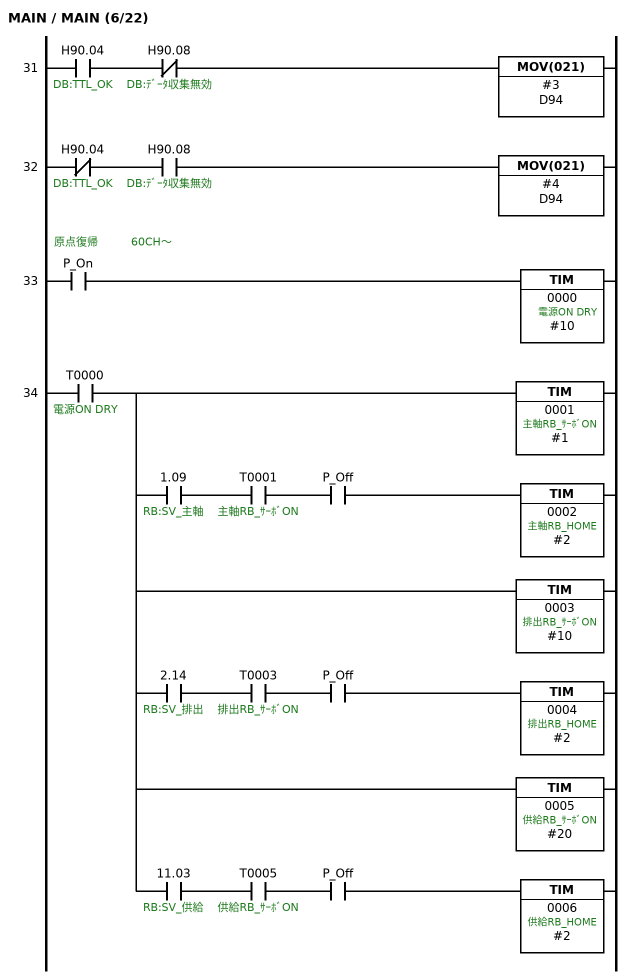
; rung 31
LD H90.04  ; DB:TTL_OK
ANDNOT H90.08  ; DB:ﾃﾞｰﾀ収集無効
MOV(021) #3 D94
; rung 32
LDNOT H90.04  ; DB:TTL_OK
AND H90.08  ; DB:ﾃﾞｰﾀ収集無効
MOV(021) #4 D94
; rung 33: 原点復帰　　　60CH～
LD P_On
TIM 0000 #10  ; 電源ON DRY
; rung 34
LD T0000  ; 電源ON DRY
OUT TR0
TIM 0001 #1  ; 主軸RB_ｻｰﾎﾞON
AND 1.09  ; RB:SV_主軸
AND T0001  ; 主軸RB_ｻｰﾎﾞON
AND P_Off
TIM 0002 #2  ; 主軸RB_HOME
LD TR0
TIM 0003 #10  ; 排出RB_ｻｰﾎﾞON
AND 2.14  ; RB:SV_排出
AND T0003  ; 排出RB_ｻｰﾎﾞON
AND P_Off
TIM 0004 #2  ; 排出RB_HOME
LD TR0
TIM 0005 #20  ; 供給RB_ｻｰﾎﾞON
AND 11.03  ; RB:SV_供給
AND T0005  ; 供給RB_ｻｰﾎﾞON
AND P_Off
TIM 0006 #2  ; 供給RB_HOME

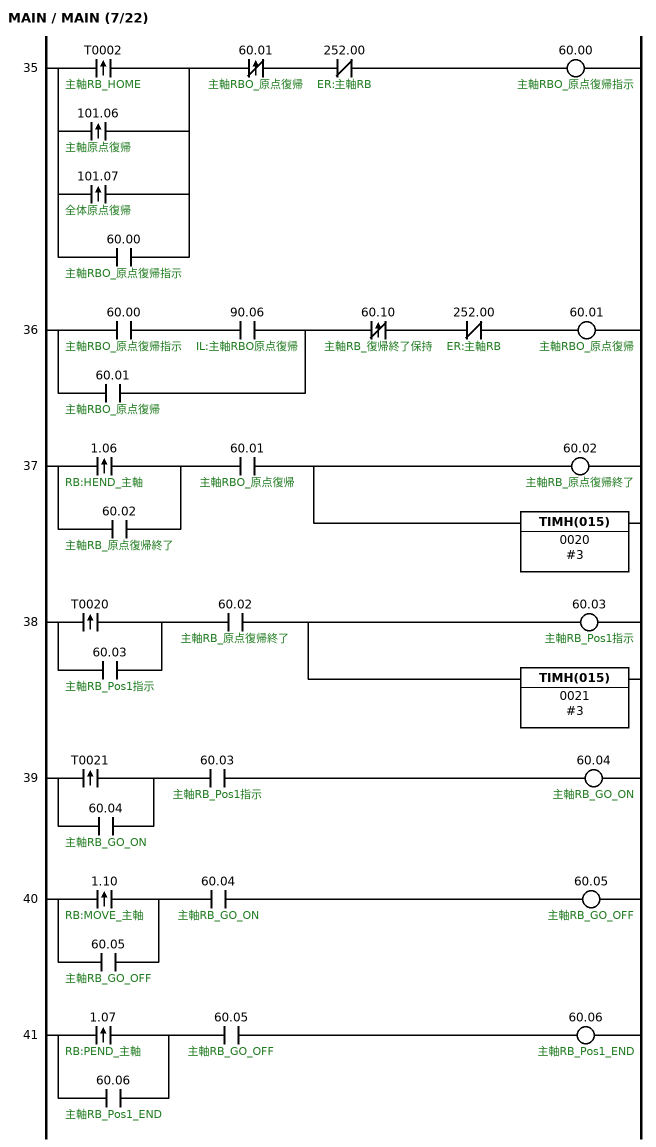
; rung 35
@LD T0002  ; 主軸RB_HOME
@OR 101.06  ; 主軸原点復帰
@OR 101.07  ; 全体原点復帰
OR 60.00  ; 主軸RBO_原点復帰指示
@ANDNOT 60.01  ; 主軸RBO_原点復帰
ANDNOT 252.00  ; ER:主軸RB
OUT 60.00  ; 主軸RBO_原点復帰指示
; rung 36
LD 60.00  ; 主軸RBO_原点復帰指示
AND 90.06  ; IL:主軸RBO原点復帰
OR 60.01  ; 主軸RBO_原点復帰
@ANDNOT 60.10  ; 主軸RB_復帰終了保持
ANDNOT 252.00  ; ER:主軸RB
OUT 60.01  ; 主軸RBO_原点復帰
; rung 37
@LD 1.06  ; RB:HEND_主軸
OR 60.02  ; 主軸RB_原点復帰終了
AND 60.01  ; 主軸RBO_原点復帰
OUT 60.02  ; 主軸RB_原点復帰終了
TIMH(015) 0020 #3
; rung 38
@LD T0020
OR 60.03  ; 主軸RB_Pos1指示
AND 60.02  ; 主軸RB_原点復帰終了
OUT 60.03  ; 主軸RB_Pos1指示
TIMH(015) 0021 #3
; rung 39
@LD T0021
OR 60.04  ; 主軸RB_GO_ON
AND 60.03  ; 主軸RB_Pos1指示
OUT 60.04  ; 主軸RB_GO_ON
; rung 40
@LD 1.10  ; RB:MOVE_主軸
OR 60.05  ; 主軸RB_GO_OFF
AND 60.04  ; 主軸RB_GO_ON
OUT 60.05  ; 主軸RB_GO_OFF
; rung 41
@LD 1.07  ; RB:PEND_主軸
OR 60.06  ; 主軸RB_Pos1_END
AND 60.05  ; 主軸RB_GO_OFF
OUT 60.06  ; 主軸RB_Pos1_END

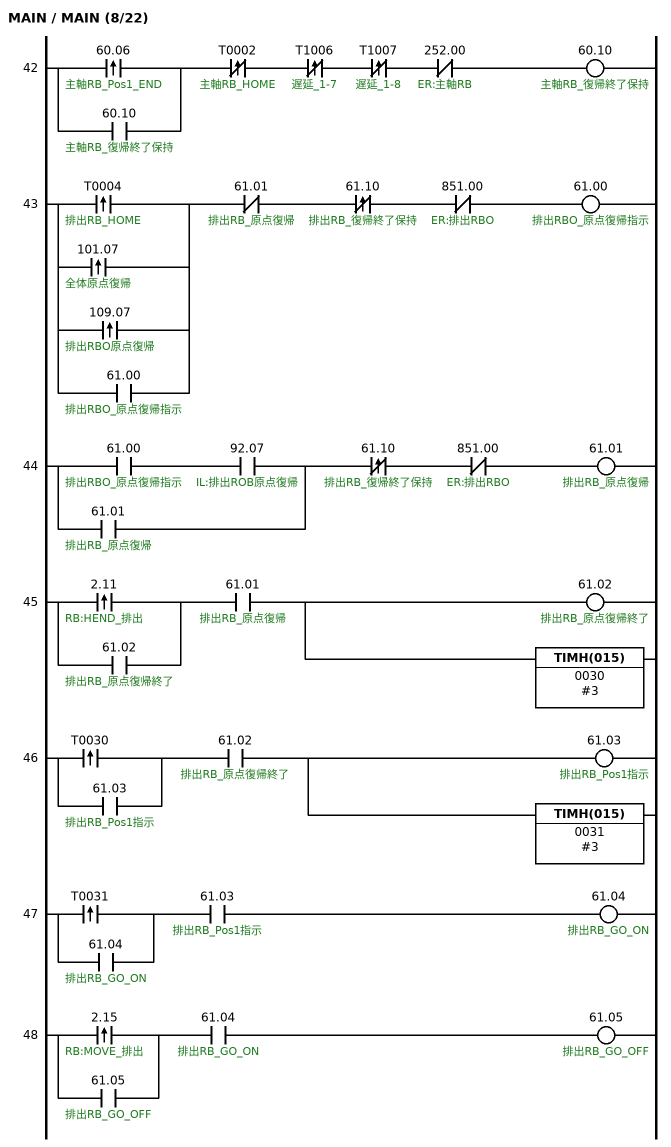
; rung 42
@LD 60.06  ; 主軸RB_Pos1_END
OR 60.10  ; 主軸RB_復帰終了保持
@ANDNOT T0002  ; 主軸RB_HOME
@ANDNOT T1006  ; 遅延_1-7
@ANDNOT T1007  ; 遅延_1-8
ANDNOT 252.00  ; ER:主軸RB
OUT 60.10  ; 主軸RB_復帰終了保持
; rung 43
@LD T0004  ; 排出RB_HOME
@OR 101.07  ; 全体原点復帰
@OR 109.07  ; 排出RBO原点復帰
OR 61.00  ; 排出RBO_原点復帰指示
ANDNOT 61.01  ; 排出RB_原点復帰
@ANDNOT 61.10  ; 排出RB_復帰終了保持
ANDNOT 851.00  ; ER:排出RBO
OUT 61.00  ; 排出RBO_原点復帰指示
; rung 44
LD 61.00  ; 排出RBO_原点復帰指示
AND 92.07  ; IL:排出ROB原点復帰
OR 61.01  ; 排出RB_原点復帰
@ANDNOT 61.10  ; 排出RB_復帰終了保持
ANDNOT 851.00  ; ER:排出RBO
OUT 61.01  ; 排出RB_原点復帰
; rung 45
@LD 2.11  ; RB:HEND_排出
OR 61.02  ; 排出RB_原点復帰終了
AND 61.01  ; 排出RB_原点復帰
OUT 61.02  ; 排出RB_原点復帰終了
TIMH(015) 0030 #3
; rung 46
@LD T0030
OR 61.03  ; 排出RB_Pos1指示
AND 61.02  ; 排出RB_原点復帰終了
OUT 61.03  ; 排出RB_Pos1指示
TIMH(015) 0031 #3
; rung 47
@LD T0031
OR 61.04  ; 排出RB_GO_ON
AND 61.03  ; 排出RB_Pos1指示
OUT 61.04  ; 排出RB_GO_ON
; rung 48
@LD 2.15  ; RB:MOVE_排出
OR 61.05  ; 排出RB_GO_OFF
AND 61.04  ; 排出RB_GO_ON
OUT 61.05  ; 排出RB_GO_OFF

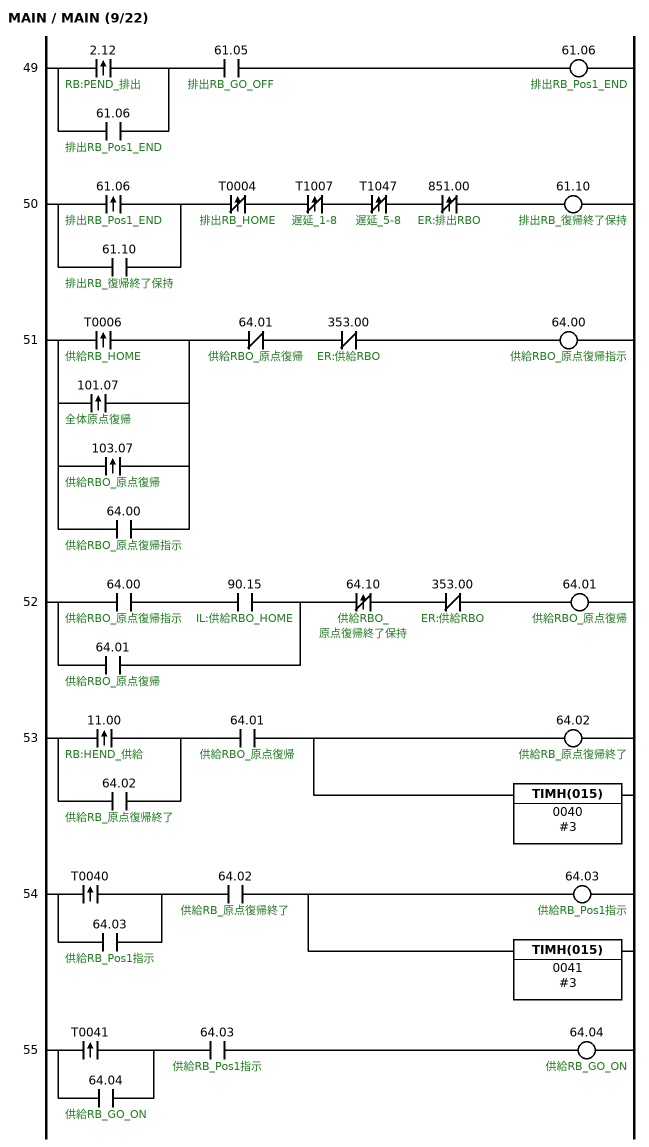
; rung 49
@LD 2.12  ; RB:PEND_排出
OR 61.06  ; 排出RB_Pos1_END
AND 61.05  ; 排出RB_GO_OFF
OUT 61.06  ; 排出RB_Pos1_END
; rung 50
@LD 61.06  ; 排出RB_Pos1_END
OR 61.10  ; 排出RB_復帰終了保持
@ANDNOT T0004  ; 排出RB_HOME
@ANDNOT T1007  ; 遅延_1-8
@ANDNOT T1047  ; 遅延_5-8
@ANDNOT 851.00  ; ER:排出RBO
OUT 61.10  ; 排出RB_復帰終了保持
; rung 51
@LD T0006  ; 供給RB_HOME
@OR 101.07  ; 全体原点復帰
@OR 103.07  ; 供給RBO_原点復帰
OR 64.00  ; 供給RBO_原点復帰指示
ANDNOT 64.01  ; 供給RBO_原点復帰
ANDNOT 353.00  ; ER:供給RBO
OUT 64.00  ; 供給RBO_原点復帰指示
; rung 52
LD 64.00  ; 供給RBO_原点復帰指示
AND 90.15  ; IL:供給RBO_HOME
OR 64.01  ; 供給RBO_原点復帰
@ANDNOT 64.10  ; 供給RBO_原点復帰終了保持
ANDNOT 353.00  ; ER:供給RBO
OUT 64.01  ; 供給RBO_原点復帰
; rung 53
@LD 11.00  ; RB:HEND_供給
OR 64.02  ; 供給RB_原点復帰終了
AND 64.01  ; 供給RBO_原点復帰
OUT 64.02  ; 供給RB_原点復帰終了
TIMH(015) 0040 #3
; rung 54
@LD T0040
OR 64.03  ; 供給RB_Pos1指示
AND 64.02  ; 供給RB_原点復帰終了
OUT 64.03  ; 供給RB_Pos1指示
TIMH(015) 0041 #3
; rung 55
@LD T0041
OR 64.04  ; 供給RB_GO_ON
AND 64.03  ; 供給RB_Pos1指示
OUT 64.04  ; 供給RB_GO_ON

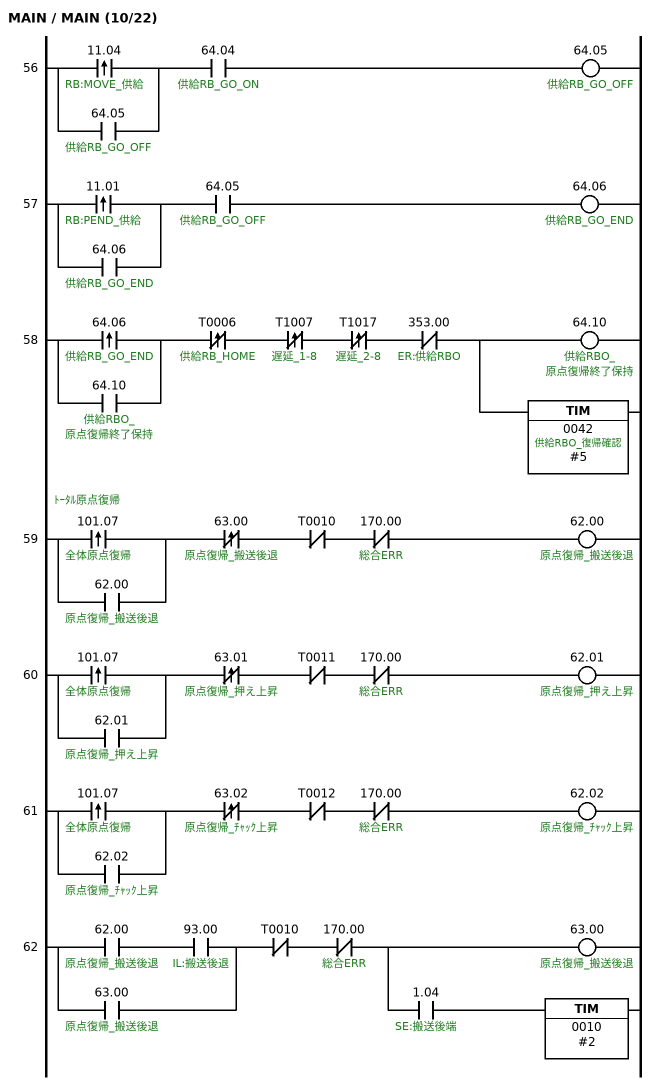
; rung 56
@LD 11.04  ; RB:MOVE_供給
OR 64.05  ; 供給RB_GO_OFF
AND 64.04  ; 供給RB_GO_ON
OUT 64.05  ; 供給RB_GO_OFF
; rung 57
@LD 11.01  ; RB:PEND_供給
OR 64.06  ; 供給RB_GO_END
AND 64.05  ; 供給RB_GO_OFF
OUT 64.06  ; 供給RB_GO_END
; rung 58
@LD 64.06  ; 供給RB_GO_END
OR 64.10  ; 供給RBO_原点復帰終了保持
@ANDNOT T0006  ; 供給RB_HOME
@ANDNOT T1007  ; 遅延_1-8
@ANDNOT T1017  ; 遅延_2-8
ANDNOT 353.00  ; ER:供給RBO
OUT 64.10  ; 供給RBO_原点復帰終了保持
TIM 0042 #5  ; 供給RBO_復帰確認
; rung 59: ﾄｰﾀﾙ原点復帰
@LD 101.07  ; 全体原点復帰
OR 62.00  ; 原点復帰_搬送後退
@ANDNOT 63.00  ; 原点復帰_搬送後退
ANDNOT T0010
ANDNOT 170.00  ; 総合ERR
OUT 62.00  ; 原点復帰_搬送後退
; rung 60
@LD 101.07  ; 全体原点復帰
OR 62.01  ; 原点復帰_押え上昇
@ANDNOT 63.01  ; 原点復帰_押え上昇
ANDNOT T0011
ANDNOT 170.00  ; 総合ERR
OUT 62.01  ; 原点復帰_押え上昇
; rung 61
@LD 101.07  ; 全体原点復帰
OR 62.02  ; 原点復帰_ﾁｬｯｸ上昇
@ANDNOT 63.02  ; 原点復帰_ﾁｬｯｸ上昇
ANDNOT T0012
ANDNOT 170.00  ; 総合ERR
OUT 62.02  ; 原点復帰_ﾁｬｯｸ上昇
; rung 62
LD 62.00  ; 原点復帰_搬送後退
AND 93.00  ; IL:搬送後退
OR 63.00  ; 原点復帰_搬送後退
ANDNOT T0010
ANDNOT 170.00  ; 総合ERR
OUT 63.00  ; 原点復帰_搬送後退
AND 1.04  ; SE:搬送後端
TIM 0010 #2

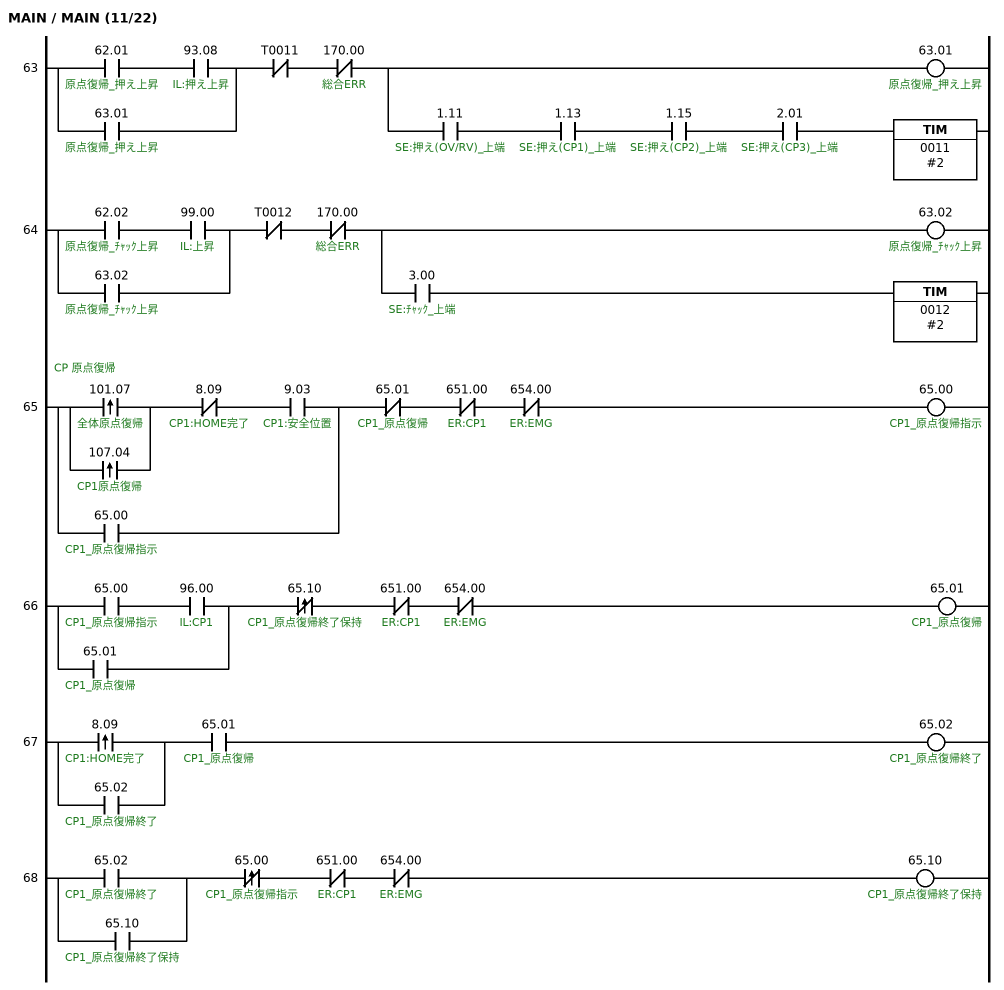
; rung 63
LD 62.01  ; 原点復帰_押え上昇
AND 93.08  ; IL:押え上昇
OR 63.01  ; 原点復帰_押え上昇
ANDNOT T0011
ANDNOT 170.00  ; 総合ERR
OUT 63.01  ; 原点復帰_押え上昇
AND 1.11  ; SE:押え(OV/RV)_上端
AND 1.13  ; SE:押え(CP1)_上端
AND 1.15  ; SE:押え(CP2)_上端
AND 2.01  ; SE:押え(CP3)_上端
TIM 0011 #2
; rung 64
LD 62.02  ; 原点復帰_ﾁｬｯｸ上昇
AND 99.00  ; IL:上昇
OR 63.02  ; 原点復帰_ﾁｬｯｸ上昇
ANDNOT T0012
ANDNOT 170.00  ; 総合ERR
OUT 63.02  ; 原点復帰_ﾁｬｯｸ上昇
AND 3.00  ; SE:ﾁｬｯｸ_上端
TIM 0012 #2
; rung 65: CP 原点復帰
@LD 101.07  ; 全体原点復帰
@OR 107.04  ; CP1原点復帰
ANDNOT 8.09  ; CP1:HOME完了
AND 9.03  ; CP1:安全位置
OR 65.00  ; CP1_原点復帰指示
ANDNOT 65.01  ; CP1_原点復帰
ANDNOT 651.00  ; ER:CP1
ANDNOT 654.00  ; ER:EMG
OUT 65.00  ; CP1_原点復帰指示
; rung 66
LD 65.00  ; CP1_原点復帰指示
AND 96.00  ; IL:CP1
OR 65.01  ; CP1_原点復帰
@ANDNOT 65.10  ; CP1_原点復帰終了保持
ANDNOT 651.00  ; ER:CP1
ANDNOT 654.00  ; ER:EMG
OUT 65.01  ; CP1_原点復帰
; rung 67
@LD 8.09  ; CP1:HOME完了
OR 65.02  ; CP1_原点復帰終了
AND 65.01  ; CP1_原点復帰
OUT 65.02  ; CP1_原点復帰終了
; rung 68
LD 65.02  ; CP1_原点復帰終了
OR 65.10  ; CP1_原点復帰終了保持
@ANDNOT 65.00  ; CP1_原点復帰指示
ANDNOT 651.00  ; ER:CP1
ANDNOT 654.00  ; ER:EMG
OUT 65.10  ; CP1_原点復帰終了保持

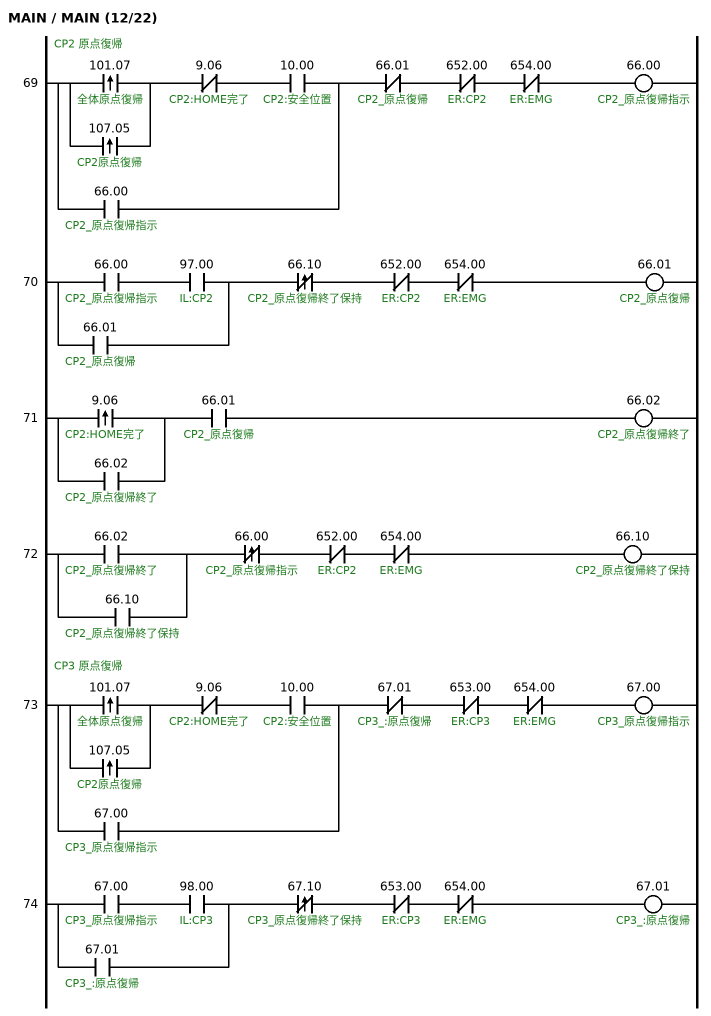
; rung 69: CP2 原点復帰
@LD 101.07  ; 全体原点復帰
@OR 107.05  ; CP2原点復帰
ANDNOT 9.06  ; CP2:HOME完了
AND 10.00  ; CP2:安全位置
OR 66.00  ; CP2_原点復帰指示
ANDNOT 66.01  ; CP2_原点復帰
ANDNOT 652.00  ; ER:CP2
ANDNOT 654.00  ; ER:EMG
OUT 66.00  ; CP2_原点復帰指示
; rung 70
LD 66.00  ; CP2_原点復帰指示
AND 97.00  ; IL:CP2
OR 66.01  ; CP2_原点復帰
@ANDNOT 66.10  ; CP2_原点復帰終了保持
ANDNOT 652.00  ; ER:CP2
ANDNOT 654.00  ; ER:EMG
OUT 66.01  ; CP2_原点復帰
; rung 71
@LD 9.06  ; CP2:HOME完了
OR 66.02  ; CP2_原点復帰終了
AND 66.01  ; CP2_原点復帰
OUT 66.02  ; CP2_原点復帰終了
; rung 72
LD 66.02  ; CP2_原点復帰終了
OR 66.10  ; CP2_原点復帰終了保持
@ANDNOT 66.00  ; CP2_原点復帰指示
ANDNOT 652.00  ; ER:CP2
ANDNOT 654.00  ; ER:EMG
OUT 66.10  ; CP2_原点復帰終了保持
; rung 73: CP3 原点復帰
@LD 101.07  ; 全体原点復帰
@OR 107.05  ; CP2原点復帰
ANDNOT 9.06  ; CP2:HOME完了
AND 10.00  ; CP2:安全位置
OR 67.00  ; CP3_原点復帰指示
ANDNOT 67.01  ; CP3_:原点復帰
ANDNOT 653.00  ; ER:CP3
ANDNOT 654.00  ; ER:EMG
OUT 67.00  ; CP3_原点復帰指示
; rung 74
LD 67.00  ; CP3_原点復帰指示
AND 98.00  ; IL:CP3
OR 67.01  ; CP3_:原点復帰
@ANDNOT 67.10  ; CP3_原点復帰終了保持
ANDNOT 653.00  ; ER:CP3
ANDNOT 654.00  ; ER:EMG
OUT 67.01  ; CP3_:原点復帰

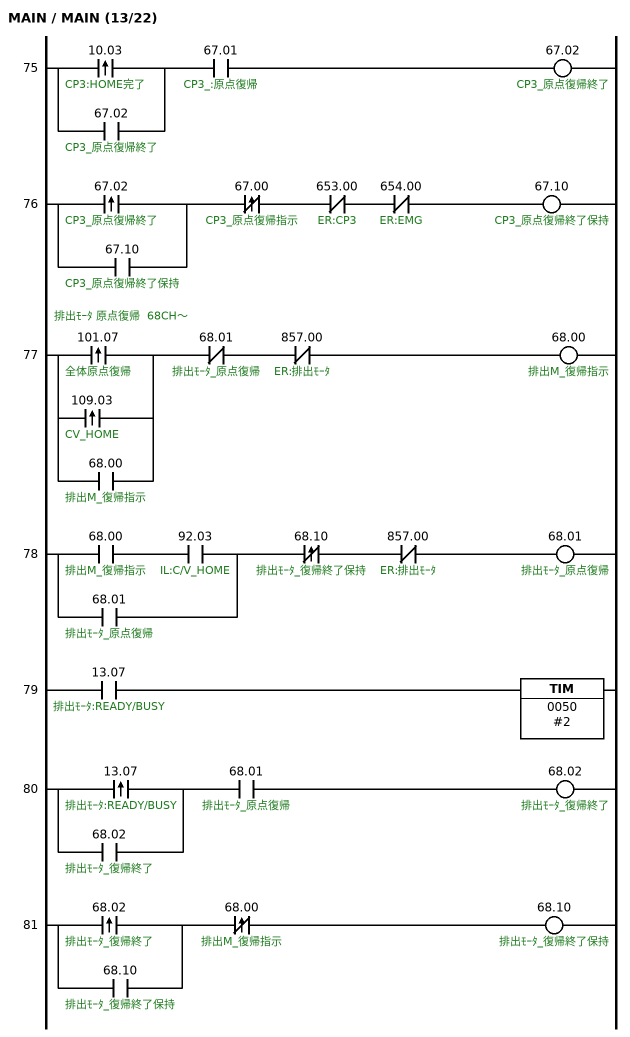
; rung 75
@LD 10.03  ; CP3:HOME完了
OR 67.02  ; CP3_原点復帰終了
AND 67.01  ; CP3_:原点復帰
OUT 67.02  ; CP3_原点復帰終了
; rung 76
@LD 67.02  ; CP3_原点復帰終了
OR 67.10  ; CP3_原点復帰終了保持
@ANDNOT 67.00  ; CP3_原点復帰指示
ANDNOT 653.00  ; ER:CP3
ANDNOT 654.00  ; ER:EMG
OUT 67.10  ; CP3_原点復帰終了保持
; rung 77: 排出ﾓｰﾀ 原点復帰  68CH～
@LD 101.07  ; 全体原点復帰
@OR 109.03  ; CV_HOME
OR 68.00  ; 排出M_復帰指示
ANDNOT 68.01  ; 排出ﾓｰﾀ_原点復帰
ANDNOT 857.00  ; ER:排出ﾓｰﾀ
OUT 68.00  ; 排出M_復帰指示
; rung 78
LD 68.00  ; 排出M_復帰指示
AND 92.03  ; IL:C/V_HOME
OR 68.01  ; 排出ﾓｰﾀ_原点復帰
@ANDNOT 68.10  ; 排出ﾓｰﾀ_復帰終了保持
ANDNOT 857.00  ; ER:排出ﾓｰﾀ
OUT 68.01  ; 排出ﾓｰﾀ_原点復帰
; rung 79
LD 13.07  ; 排出ﾓｰﾀ:READY/BUSY
TIM 0050 #2
; rung 80
@LD 13.07  ; 排出ﾓｰﾀ:READY/BUSY
OR 68.02  ; 排出ﾓｰﾀ_復帰終了
AND 68.01  ; 排出ﾓｰﾀ_原点復帰
OUT 68.02  ; 排出ﾓｰﾀ_復帰終了
; rung 81
@LD 68.02  ; 排出ﾓｰﾀ_復帰終了
OR 68.10  ; 排出ﾓｰﾀ_復帰終了保持
@ANDNOT 68.00  ; 排出M_復帰指示
OUT 68.10  ; 排出ﾓｰﾀ_復帰終了保持

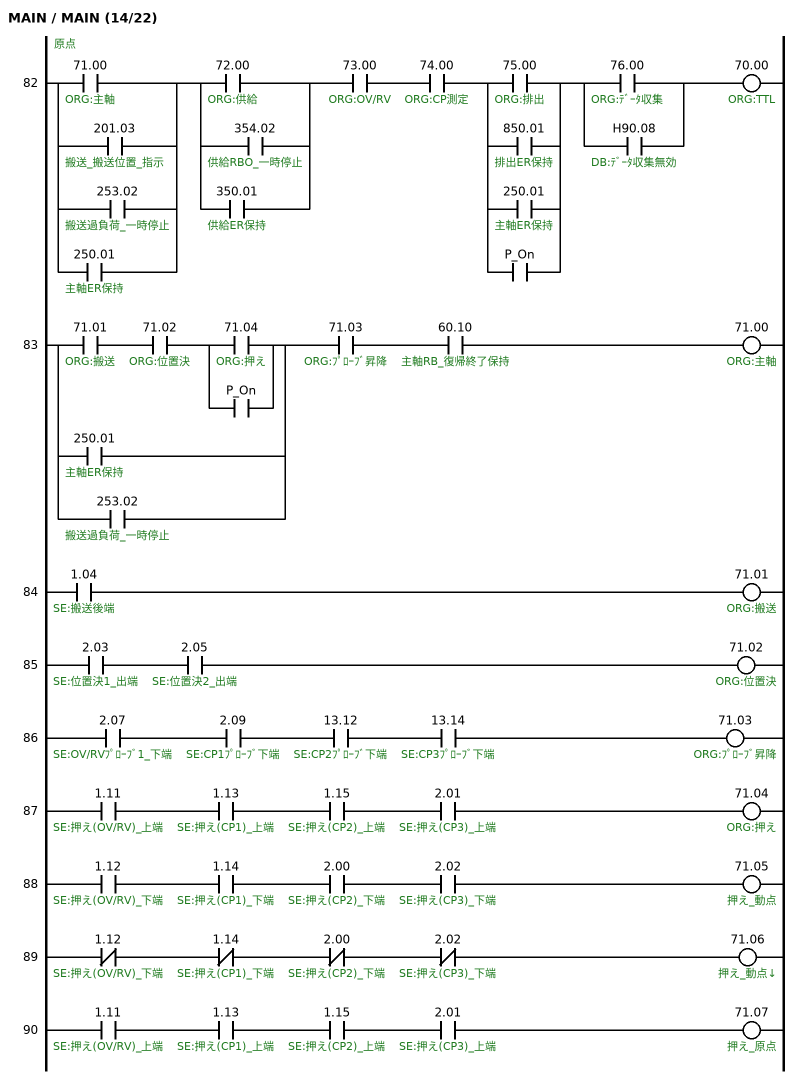
; rung 82: 原点
LD 71.00  ; ORG:主軸
OR 201.03  ; 搬送_搬送位置_指示
OR 253.02  ; 搬送過負荷_一時停止
OR 250.01  ; 主軸ER保持
LD 72.00  ; ORG:供給
OR 354.02  ; 供給RBO_一時停止
OR 350.01  ; 供給ER保持
ANDLD
AND 73.00  ; ORG:OV/RV
AND 74.00  ; ORG:CP測定
LD 75.00  ; ORG:排出
OR 850.01  ; 排出ER保持
OR 250.01  ; 主軸ER保持
OR P_On
ANDLD
LD 76.00  ; ORG:ﾃﾞｰﾀ収集
OR H90.08  ; DB:ﾃﾞｰﾀ収集無効
ANDLD
OUT 70.00  ; ORG:TTL
; rung 83
LD 71.01  ; ORG:搬送
AND 71.02  ; ORG:位置決
LD 71.04  ; ORG:押え
OR P_On
ANDLD
OR 250.01  ; 主軸ER保持
OR 253.02  ; 搬送過負荷_一時停止
AND 71.03  ; ORG:ﾌﾟﾛｰﾌﾞ昇降
AND 60.10  ; 主軸RB_復帰終了保持
OUT 71.00  ; ORG:主軸
; rung 84
LD 1.04  ; SE:搬送後端
OUT 71.01  ; ORG:搬送
; rung 85
LD 2.03  ; SE:位置決1_出端
AND 2.05  ; SE:位置決2_出端
OUT 71.02  ; ORG:位置決
; rung 86
LD 2.07  ; SE:OV/RVﾌﾟﾛｰﾌﾞ1_下端
AND 2.09  ; SE:CP1ﾌﾟﾛｰﾌﾞ下端
AND 13.12  ; SE:CP2ﾌﾟﾛｰﾌﾞ下端
AND 13.14  ; SE:CP3ﾌﾟﾛｰﾌﾞ下端
OUT 71.03  ; ORG:ﾌﾟﾛｰﾌﾞ昇降
; rung 87
LD 1.11  ; SE:押え(OV/RV)_上端
AND 1.13  ; SE:押え(CP1)_上端
AND 1.15  ; SE:押え(CP2)_上端
AND 2.01  ; SE:押え(CP3)_上端
OUT 71.04  ; ORG:押え
; rung 88
LD 1.12  ; SE:押え(OV/RV)_下端
AND 1.14  ; SE:押え(CP1)_下端
AND 2.00  ; SE:押え(CP2)_下端
AND 2.02  ; SE:押え(CP3)_下端
OUT 71.05  ; 押え_動点
; rung 89
LDNOT 1.12  ; SE:押え(OV/RV)_下端
ANDNOT 1.14  ; SE:押え(CP1)_下端
ANDNOT 2.00  ; SE:押え(CP2)_下端
ANDNOT 2.02  ; SE:押え(CP3)_下端
OUT 71.06  ; 押え_動点↓
; rung 90
LD 1.11  ; SE:押え(OV/RV)_上端
AND 1.13  ; SE:押え(CP1)_上端
AND 1.15  ; SE:押え(CP2)_上端
AND 2.01  ; SE:押え(CP3)_上端
OUT 71.07  ; 押え_原点

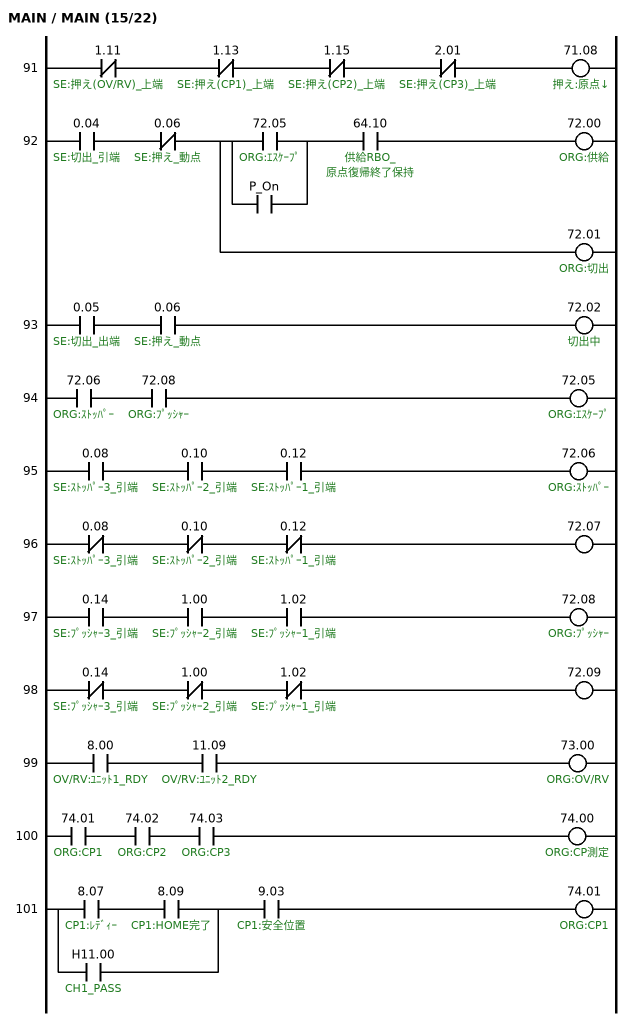
; rung 91
LDNOT 1.11  ; SE:押え(OV/RV)_上端
ANDNOT 1.13  ; SE:押え(CP1)_上端
ANDNOT 1.15  ; SE:押え(CP2)_上端
ANDNOT 2.01  ; SE:押え(CP3)_上端
OUT 71.08  ; 押え:原点↓
; rung 92
LD 0.04  ; SE:切出_引端
ANDNOT 0.06  ; SE:押え_動点
OUT TR0
LD 72.05  ; ORG:ｴｽｹｰﾌﾟ
OR P_On
ANDLD
AND 64.10  ; 供給RBO_原点復帰終了保持
OUT 72.00  ; ORG:供給
LD TR0
OUT 72.01  ; ORG:切出
; rung 93
LD 0.05  ; SE:切出_出端
AND 0.06  ; SE:押え_動点
OUT 72.02  ; 切出中
; rung 94
LD 72.06  ; ORG:ｽﾄｯﾊﾟｰ
AND 72.08  ; ORG:ﾌﾟｯｼｬｰ
OUT 72.05  ; ORG:ｴｽｹｰﾌﾟ
; rung 95
LD 0.08  ; SE:ｽﾄｯﾊﾟｰ3_引端
AND 0.10  ; SE:ｽﾄｯﾊﾟｰ2_引端
AND 0.12  ; SE:ｽﾄｯﾊﾟｰ1_引端
OUT 72.06  ; ORG:ｽﾄｯﾊﾟｰ
; rung 96
LDNOT 0.08  ; SE:ｽﾄｯﾊﾟｰ3_引端
ANDNOT 0.10  ; SE:ｽﾄｯﾊﾟｰ2_引端
ANDNOT 0.12  ; SE:ｽﾄｯﾊﾟｰ1_引端
OUT 72.07
; rung 97
LD 0.14  ; SE:ﾌﾟｯｼｬｰ3_引端
AND 1.00  ; SE:ﾌﾟｯｼｬｰ2_引端
AND 1.02  ; SE:ﾌﾟｯｼｬｰ1_引端
OUT 72.08  ; ORG:ﾌﾟｯｼｬｰ
; rung 98
LDNOT 0.14  ; SE:ﾌﾟｯｼｬｰ3_引端
ANDNOT 1.00  ; SE:ﾌﾟｯｼｬｰ2_引端
ANDNOT 1.02  ; SE:ﾌﾟｯｼｬｰ1_引端
OUT 72.09
; rung 99
LD 8.00  ; OV/RV:ﾕﾆｯﾄ1_RDY
AND 11.09  ; OV/RV:ﾕﾆｯﾄ2_RDY
OUT 73.00  ; ORG:OV/RV
; rung 100
LD 74.01  ; ORG:CP1
AND 74.02  ; ORG:CP2
AND 74.03  ; ORG:CP3
OUT 74.00  ; ORG:CP測定
; rung 101
LD 8.07  ; CP1:ﾚﾃﾞｨｰ
AND 8.09  ; CP1:HOME完了
OR H11.00  ; CH1_PASS
AND 9.03  ; CP1:安全位置
OUT 74.01  ; ORG:CP1

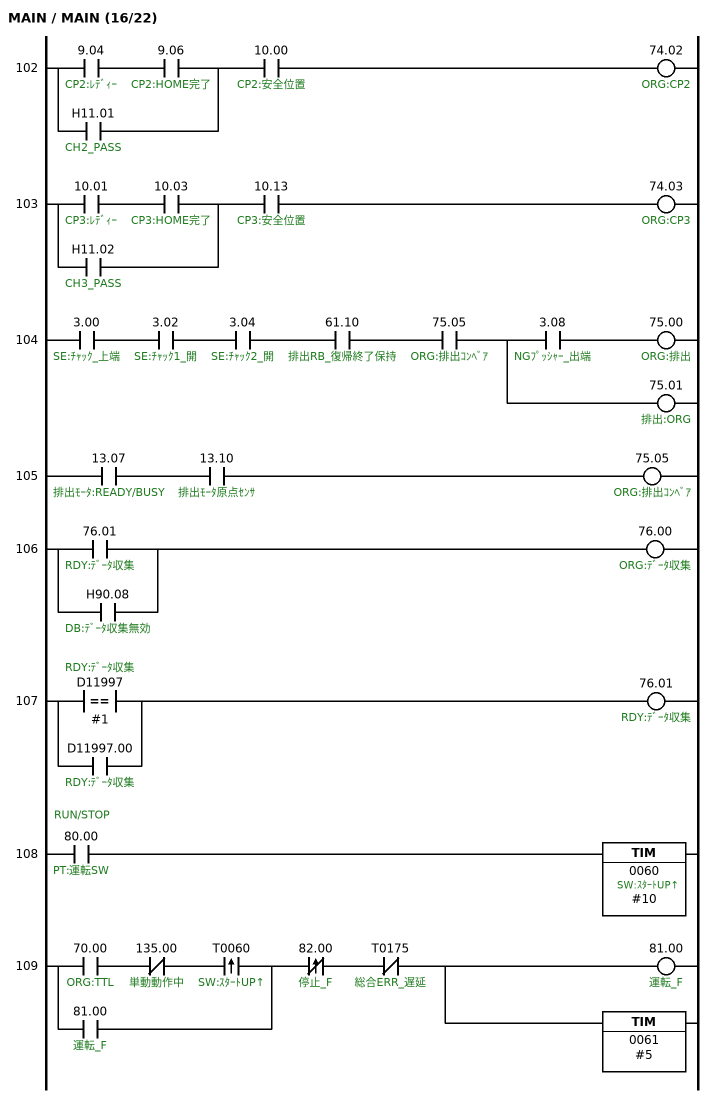
; rung 102
LD 9.04  ; CP2:ﾚﾃﾞｨｰ
AND 9.06  ; CP2:HOME完了
OR H11.01  ; CH2_PASS
AND 10.00  ; CP2:安全位置
OUT 74.02  ; ORG:CP2
; rung 103
LD 10.01  ; CP3:ﾚﾃﾞｨｰ
AND 10.03  ; CP3:HOME完了
OR H11.02  ; CH3_PASS
AND 10.13  ; CP3:安全位置
OUT 74.03  ; ORG:CP3
; rung 104
LD 3.00  ; SE:ﾁｬｯｸ_上端
AND 3.02  ; SE:ﾁｬｯｸ1_開
AND 3.04  ; SE:ﾁｬｯｸ2_開
AND 61.10  ; 排出RB_復帰終了保持
AND 75.05  ; ORG:排出ｺﾝﾍﾞｱ
OUT TR0
AND 3.08  ; NGﾌﾟｯｼｬｰ_出端
OUT 75.00  ; ORG:排出
LD TR0
OUT 75.01  ; 排出:ORG
; rung 105
LD 13.07  ; 排出ﾓｰﾀ:READY/BUSY
AND 13.10  ; 排出ﾓｰﾀ原点ｾﾝｻ
OUT 75.05  ; ORG:排出ｺﾝﾍﾞｱ
; rung 106
LD 76.01  ; RDY:ﾃﾞｰﾀ収集
OR H90.08  ; DB:ﾃﾞｰﾀ収集無効
OUT 76.00  ; ORG:ﾃﾞｰﾀ収集
; rung 107
LD=(300) D11997 #1  ; RDY:ﾃﾞｰﾀ収集
OR D11997.00  ; RDY:ﾃﾞｰﾀ収集
OUT 76.01  ; RDY:ﾃﾞｰﾀ収集
; rung 108: RUN/STOP
LD 80.00  ; PT:運転SW
TIM 0060 #10  ; SW:ｽﾀｰﾄUP↑
; rung 109
LD 70.00  ; ORG:TTL
ANDNOT 135.00  ; 単動動作中
@AND T0060  ; SW:ｽﾀｰﾄUP↑
OR 81.00  ; 運転_F
@ANDNOT 82.00  ; 停止_F
ANDNOT T0175  ; 総合ERR_遅延
OUT 81.00  ; 運転_F
TIM 0061 #5

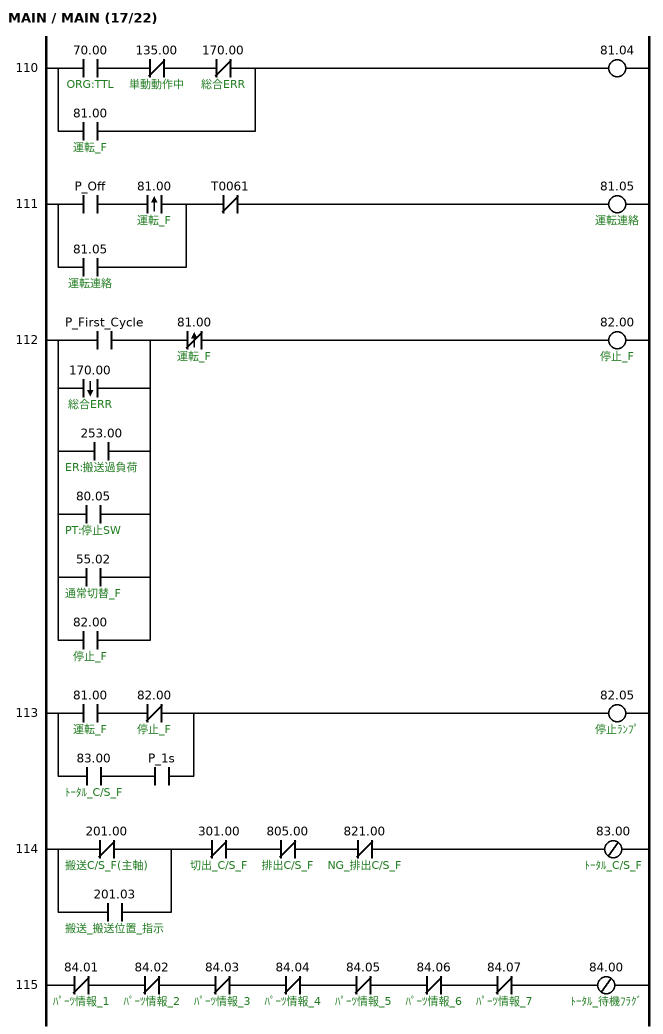
; rung 110
LD 70.00  ; ORG:TTL
ANDNOT 135.00  ; 単動動作中
ANDNOT 170.00  ; 総合ERR
OR 81.00  ; 運転_F
OUT 81.04
; rung 111
LD P_Off
@AND 81.00  ; 運転_F
OR 81.05  ; 運転連絡
ANDNOT T0061
OUT 81.05  ; 運転連絡
; rung 112
LD P_First_Cycle
%OR 170.00  ; 総合ERR
OR 253.00  ; ER:搬送過負荷
OR 80.05  ; PT:停止SW
OR 55.02  ; 通常切替_F
OR 82.00  ; 停止_F
@ANDNOT 81.00  ; 運転_F
OUT 82.00  ; 停止_F
; rung 113
LD 81.00  ; 運転_F
ANDNOT 82.00  ; 停止_F
LD 83.00  ; ﾄｰﾀﾙ_C/S_F
AND P_1s
ORLD
OUT 82.05  ; 停止ﾗﾝﾌﾟ
; rung 114
LDNOT 201.00  ; 搬送C/S_F(主軸)
OR 201.03  ; 搬送_搬送位置_指示
ANDNOT 301.00  ; 切出_C/S_F
ANDNOT 805.00  ; 排出C/S_F
ANDNOT 821.00  ; NG_排出C/S_F
OUTNOT 83.00  ; ﾄｰﾀﾙ_C/S_F
; rung 115
LDNOT 84.01  ; ﾊﾟｰﾂ情報_1
ANDNOT 84.02  ; ﾊﾟｰﾂ情報_2
ANDNOT 84.03  ; ﾊﾟｰﾂ情報_3
ANDNOT 84.04  ; ﾊﾟｰﾂ情報_4
ANDNOT 84.05  ; ﾊﾟｰﾂ情報_5
ANDNOT 84.06  ; ﾊﾟｰﾂ情報_6
ANDNOT 84.07  ; ﾊﾟｰﾂ情報_7
OUTNOT 84.00  ; ﾄｰﾀﾙ_待機ﾌﾗｸﾞ

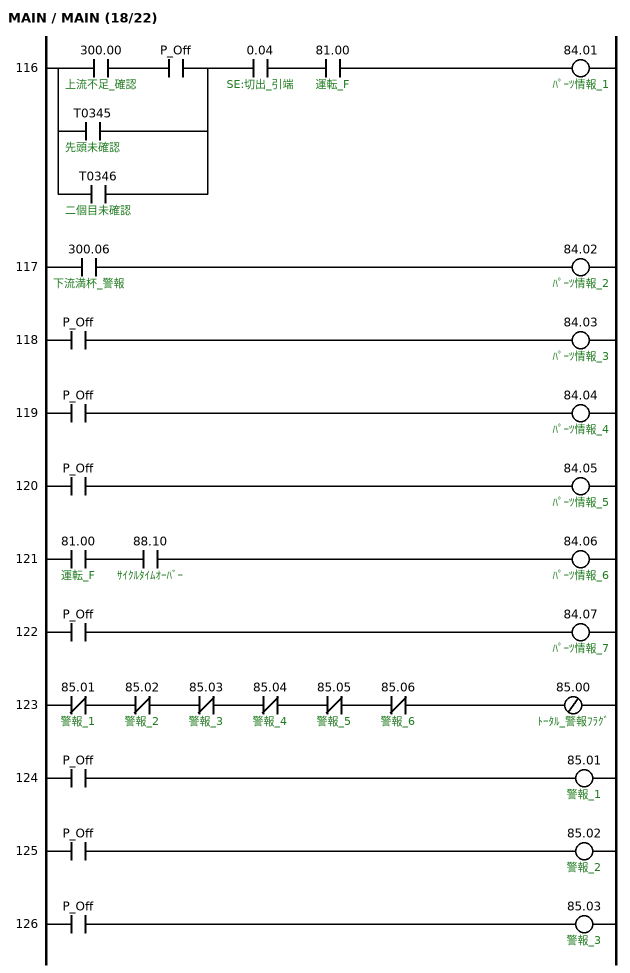
; rung 116
LD 300.00  ; 上流不足_確認
AND P_Off
OR T0345  ; 先頭未確認
OR T0346  ; 二個目未確認
AND 0.04  ; SE:切出_引端
AND 81.00  ; 運転_F
OUT 84.01  ; ﾊﾟｰﾂ情報_1
; rung 117
LD 300.06  ; 下流満杯_警報
OUT 84.02  ; ﾊﾟｰﾂ情報_2
; rung 118
LD P_Off
OUT 84.03  ; ﾊﾟｰﾂ情報_3
; rung 119
LD P_Off
OUT 84.04  ; ﾊﾟｰﾂ情報_4
; rung 120
LD P_Off
OUT 84.05  ; ﾊﾟｰﾂ情報_5
; rung 121
LD 81.00  ; 運転_F
AND 88.10  ; ｻｲｸﾙﾀｲﾑｵｰﾊﾞｰ
OUT 84.06  ; ﾊﾟｰﾂ情報_6
; rung 122
LD P_Off
OUT 84.07  ; ﾊﾟｰﾂ情報_7
; rung 123
LDNOT 85.01  ; 警報_1
ANDNOT 85.02  ; 警報_2
ANDNOT 85.03  ; 警報_3
ANDNOT 85.04  ; 警報_4
ANDNOT 85.05  ; 警報_5
ANDNOT 85.06  ; 警報_6
OUTNOT 85.00  ; ﾄｰﾀﾙ_警報ﾌﾗｸﾞ
; rung 124
LD P_Off
OUT 85.01  ; 警報_1
; rung 125
LD P_Off
OUT 85.02  ; 警報_2
; rung 126
LD P_Off
OUT 85.03  ; 警報_3

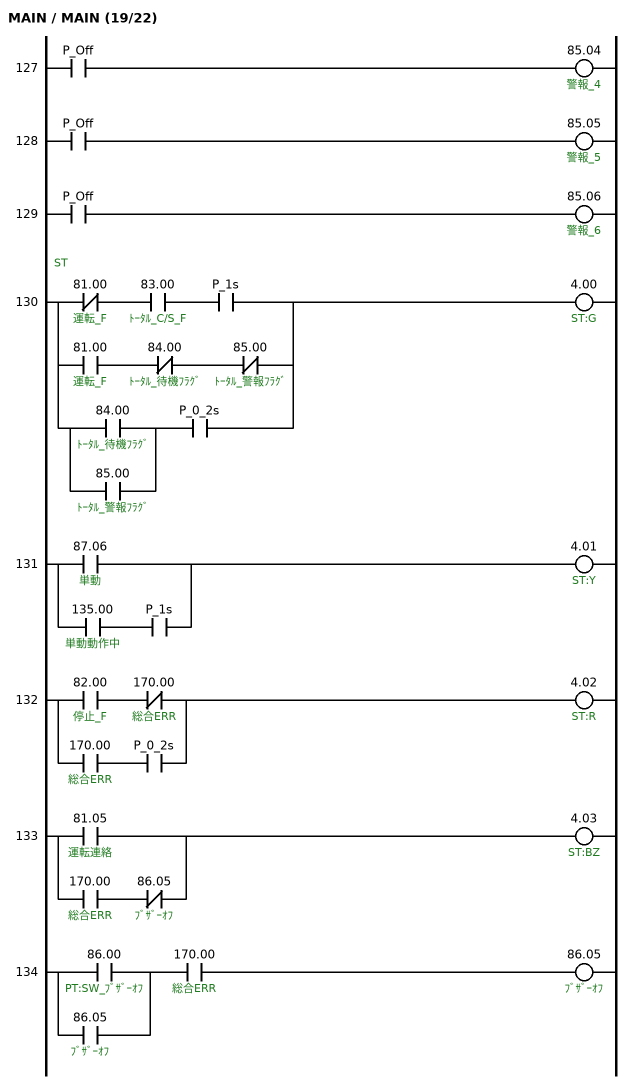
; rung 127
LD P_Off
OUT 85.04  ; 警報_4
; rung 128
LD P_Off
OUT 85.05  ; 警報_5
; rung 129
LD P_Off
OUT 85.06  ; 警報_6
; rung 130: ST
LDNOT 81.00  ; 運転_F
AND 83.00  ; ﾄｰﾀﾙ_C/S_F
AND P_1s
LD 81.00  ; 運転_F
ANDNOT 84.00  ; ﾄｰﾀﾙ_待機ﾌﾗｸﾞ
ANDNOT 85.00  ; ﾄｰﾀﾙ_警報ﾌﾗｸﾞ
ORLD
LD 84.00  ; ﾄｰﾀﾙ_待機ﾌﾗｸﾞ
OR 85.00  ; ﾄｰﾀﾙ_警報ﾌﾗｸﾞ
AND P_0_2s
ORLD
OUT 4.00  ; ST:G
; rung 131
LD 87.06  ; 単動
LD 135.00  ; 単動動作中
AND P_1s
ORLD
OUT 4.01  ; ST:Y
; rung 132
LD 82.00  ; 停止_F
ANDNOT 170.00  ; 総合ERR
LD 170.00  ; 総合ERR
AND P_0_2s
ORLD
OUT 4.02  ; ST:R
; rung 133
LD 81.05  ; 運転連絡
LD 170.00  ; 総合ERR
ANDNOT 86.05  ; ﾌﾞｻﾞｰｵﾌ
ORLD
OUT 4.03  ; ST:BZ
; rung 134
LD 86.00  ; PT:SW_ﾌﾞｻﾞｰｵﾌ
OR 86.05  ; ﾌﾞｻﾞｰｵﾌ
AND 170.00  ; 総合ERR
OUT 86.05  ; ﾌﾞｻﾞｰｵﾌ

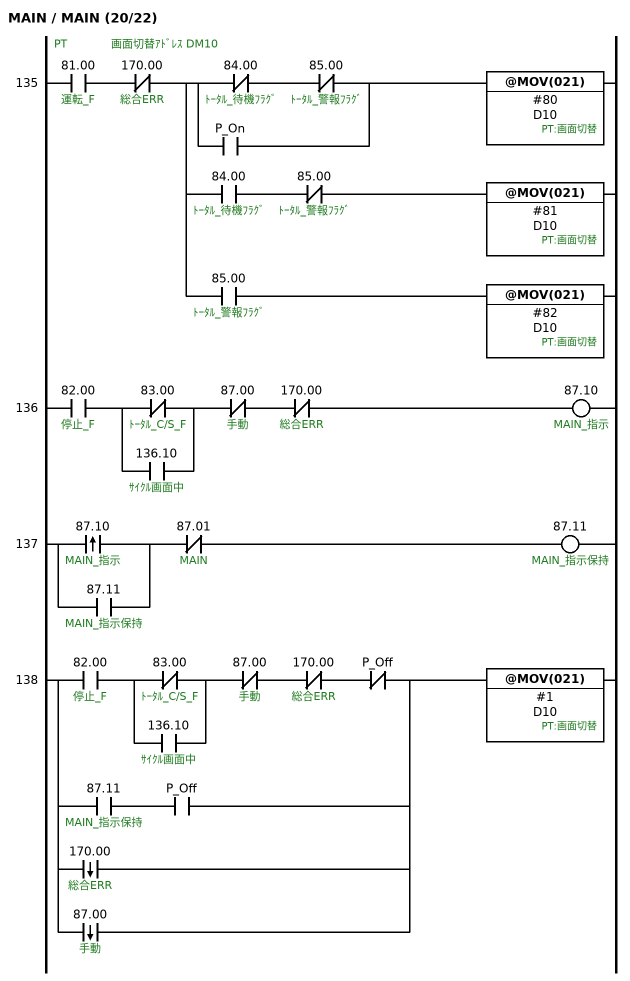
; rung 135: PT　　　　画面切替ｱﾄﾞﾚｽ DM10
LD 81.00  ; 運転_F
ANDNOT 170.00  ; 総合ERR
OUT TR0
LDNOT 84.00  ; ﾄｰﾀﾙ_待機ﾌﾗｸﾞ
ANDNOT 85.00  ; ﾄｰﾀﾙ_警報ﾌﾗｸﾞ
OR P_On
ANDLD
@MOV(021) #80 D10  ; PT:画面切替
LD TR0
AND 84.00  ; ﾄｰﾀﾙ_待機ﾌﾗｸﾞ
ANDNOT 85.00  ; ﾄｰﾀﾙ_警報ﾌﾗｸﾞ
@MOV(021) #81 D10  ; PT:画面切替
LD TR0
AND 85.00  ; ﾄｰﾀﾙ_警報ﾌﾗｸﾞ
@MOV(021) #82 D10  ; PT:画面切替
; rung 136
LD 82.00  ; 停止_F
LDNOT 83.00  ; ﾄｰﾀﾙ_C/S_F
OR 136.10  ; ｻｲｸﾙ画面中
ANDLD
ANDNOT 87.00  ; 手動
ANDNOT 170.00  ; 総合ERR
OUT 87.10  ; MAIN_指示
; rung 137
@LD 87.10  ; MAIN_指示
OR 87.11  ; MAIN_指示保持
ANDNOT 87.01  ; MAIN
OUT 87.11  ; MAIN_指示保持
; rung 138
LD 82.00  ; 停止_F
LDNOT 83.00  ; ﾄｰﾀﾙ_C/S_F
OR 136.10  ; ｻｲｸﾙ画面中
ANDLD
ANDNOT 87.00  ; 手動
ANDNOT 170.00  ; 総合ERR
ANDNOT P_Off
LD 87.11  ; MAIN_指示保持
AND P_Off
ORLD
%OR 170.00  ; 総合ERR
%OR 87.00  ; 手動
@MOV(021) #1 D10  ; PT:画面切替

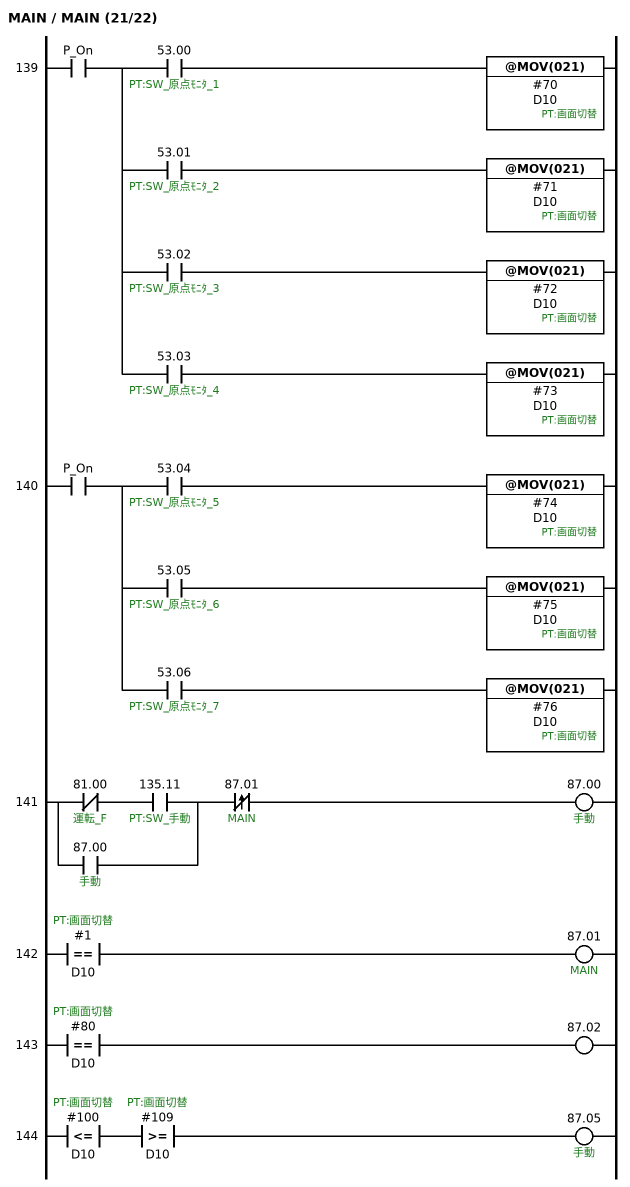
; rung 139
LD P_On
OUT TR0
AND 53.00  ; PT:SW_原点ﾓﾆﾀ_1
@MOV(021) #70 D10  ; PT:画面切替
LD TR0
AND 53.01  ; PT:SW_原点ﾓﾆﾀ_2
@MOV(021) #71 D10  ; PT:画面切替
LD TR0
AND 53.02  ; PT:SW_原点ﾓﾆﾀ_3
@MOV(021) #72 D10  ; PT:画面切替
LD TR0
AND 53.03  ; PT:SW_原点ﾓﾆﾀ_4
@MOV(021) #73 D10  ; PT:画面切替
; rung 140
LD P_On
OUT TR0
AND 53.04  ; PT:SW_原点ﾓﾆﾀ_5
@MOV(021) #74 D10  ; PT:画面切替
LD TR0
AND 53.05  ; PT:SW_原点ﾓﾆﾀ_6
@MOV(021) #75 D10  ; PT:画面切替
LD TR0
AND 53.06  ; PT:SW_原点ﾓﾆﾀ_7
@MOV(021) #76 D10  ; PT:画面切替
; rung 141
LDNOT 81.00  ; 運転_F
AND 135.11  ; PT:SW_手動
OR 87.00  ; 手動
@ANDNOT 87.01  ; MAIN
OUT 87.00  ; 手動
; rung 142
LD=(300) #1 D10  ; PT:画面切替
OUT 87.01  ; MAIN
; rung 143
LD=(300) #80 D10  ; PT:画面切替
OUT 87.02
; rung 144
LD<=(315) #100 D10  ; PT:画面切替
AND>=(325) #109 D10  ; PT:画面切替
OUT 87.05  ; 手動

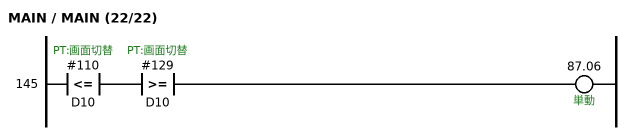
; rung 145
LD<=(315) #110 D10  ; PT:画面切替
AND>=(325) #129 D10  ; PT:画面切替
OUT 87.06  ; 単動

### Section 生産管理

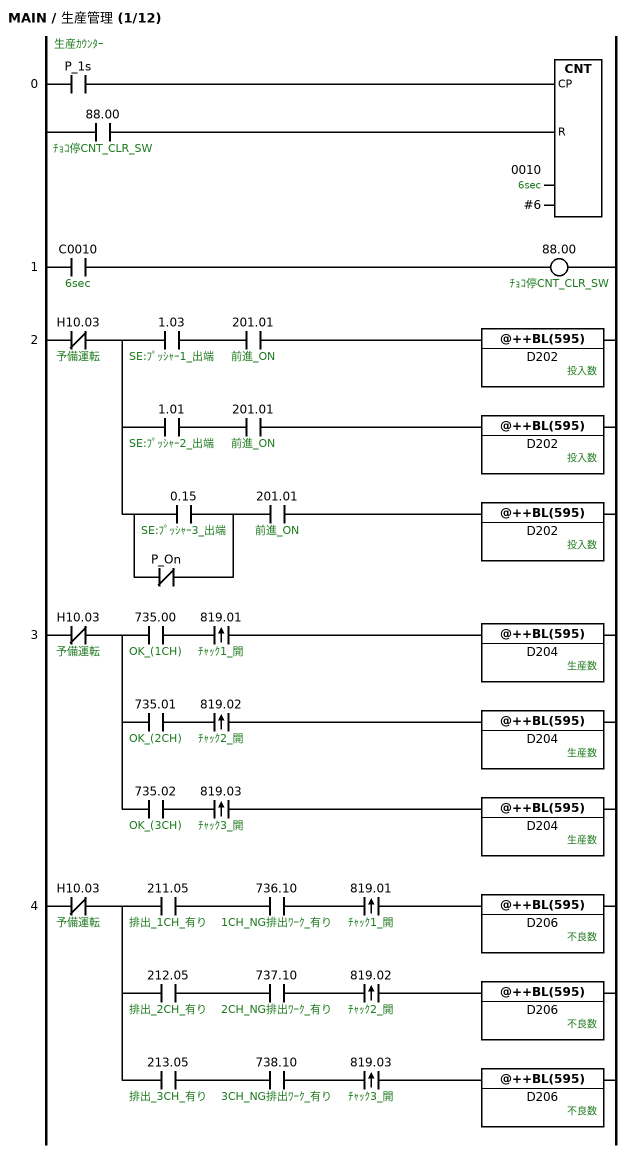
; rung 0: 生産ｶｳﾝﾀｰ
LD P_1s
LD 88.00  ; ﾁｮｺ停CNT_CLR_SW
CNT 0010 #6  ; 6sec
; rung 1
LD C0010  ; 6sec
OUT 88.00  ; ﾁｮｺ停CNT_CLR_SW
; rung 2
LDNOT H10.03  ; 予備運転
OUT TR0
AND 1.03  ; SE:ﾌﾟｯｼｬｰ1_出端
AND 201.01  ; 前進_ON
@++BL(595) D202  ; 投入数
LD TR0
AND 1.01  ; SE:ﾌﾟｯｼｬｰ2_出端
AND 201.01  ; 前進_ON
@++BL(595) D202  ; 投入数
LD TR0
LD 0.15  ; SE:ﾌﾟｯｼｬｰ3_出端
ORNOT P_On
ANDLD
AND 201.01  ; 前進_ON
@++BL(595) D202  ; 投入数
; rung 3
LDNOT H10.03  ; 予備運転
OUT TR0
AND 735.00  ; OK_(1CH)
@AND 819.01  ; ﾁｬｯｸ1_開
@++BL(595) D204  ; 生産数
LD TR0
AND 735.01  ; OK_(2CH)
@AND 819.02  ; ﾁｬｯｸ2_開
@++BL(595) D204  ; 生産数
LD TR0
AND 735.02  ; OK_(3CH)
@AND 819.03  ; ﾁｬｯｸ3_開
@++BL(595) D204  ; 生産数
; rung 4
LDNOT H10.03  ; 予備運転
OUT TR0
AND 211.05  ; 排出_1CH_有り
AND 736.10  ; 1CH_NG排出ﾜｰｸ_有り
@AND 819.01  ; ﾁｬｯｸ1_開
@++BL(595) D206  ; 不良数
LD TR0
AND 212.05  ; 排出_2CH_有り
AND 737.10  ; 2CH_NG排出ﾜｰｸ_有り
@AND 819.02  ; ﾁｬｯｸ2_開
@++BL(595) D206  ; 不良数
LD TR0
AND 213.05  ; 排出_3CH_有り
AND 738.10  ; 3CH_NG排出ﾜｰｸ_有り
@AND 819.03  ; ﾁｬｯｸ3_開
@++BL(595) D206  ; 不良数

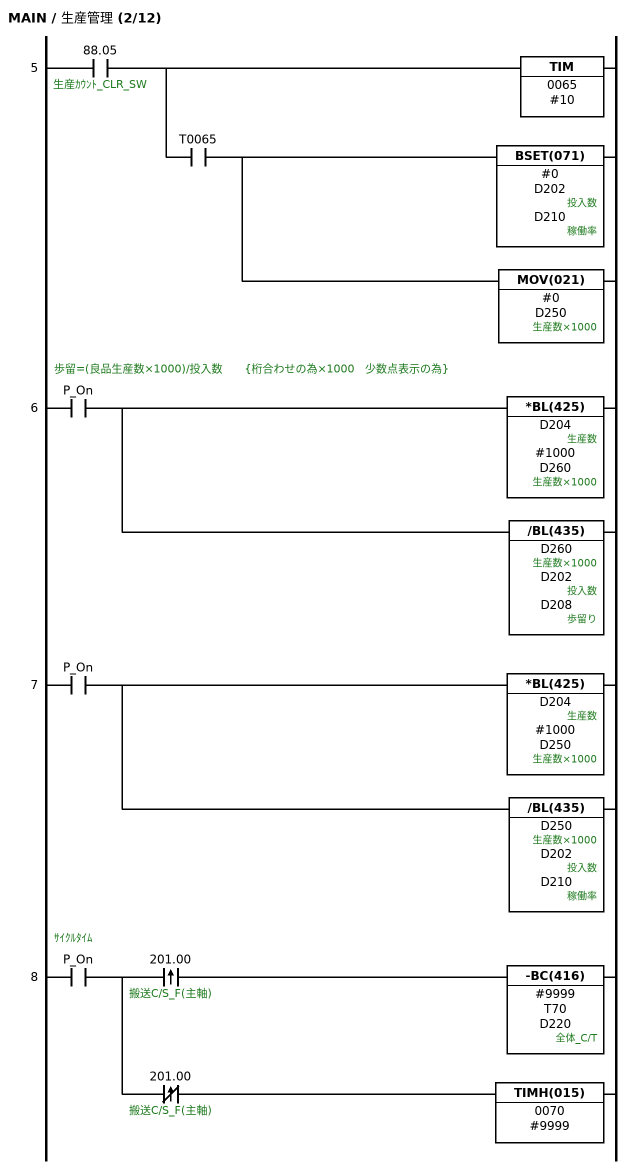
; rung 5
LD 88.05  ; 生産ｶｳﾝﾄ_CLR_SW
TIM 0065 #10
AND T0065
BSET(071) #0 D202 D210  ; 投入数, 稼働率
MOV(021) #0 D250  ; 生産数×1000
; rung 6: 歩留=(良品生産数×1000)/投入数　　{桁合わせの為×1000   少数点表示の為}
LD P_On
*BL(425) D204 #1000 D260  ; 生産数, 生産数×1000
/BL(435) D260 D202 D208  ; 生産数×1000, 投入数, 歩留り
; rung 7
LD P_On
*BL(425) D204 #1000 D250  ; 生産数, 生産数×1000
/BL(435) D250 D202 D210  ; 生産数×1000, 投入数, 稼働率
; rung 8: ｻｲｸﾙﾀｲﾑ
LD P_On
OUT TR0
@AND 201.00  ; 搬送C/S_F(主軸)
-BC(416) #9999 T70 D220  ; 全体_C/T
LD TR0
@ANDNOT 201.00  ; 搬送C/S_F(主軸)
TIMH(015) 0070 #9999

